REGION Network 46: FIT-508 LOW / HIGH
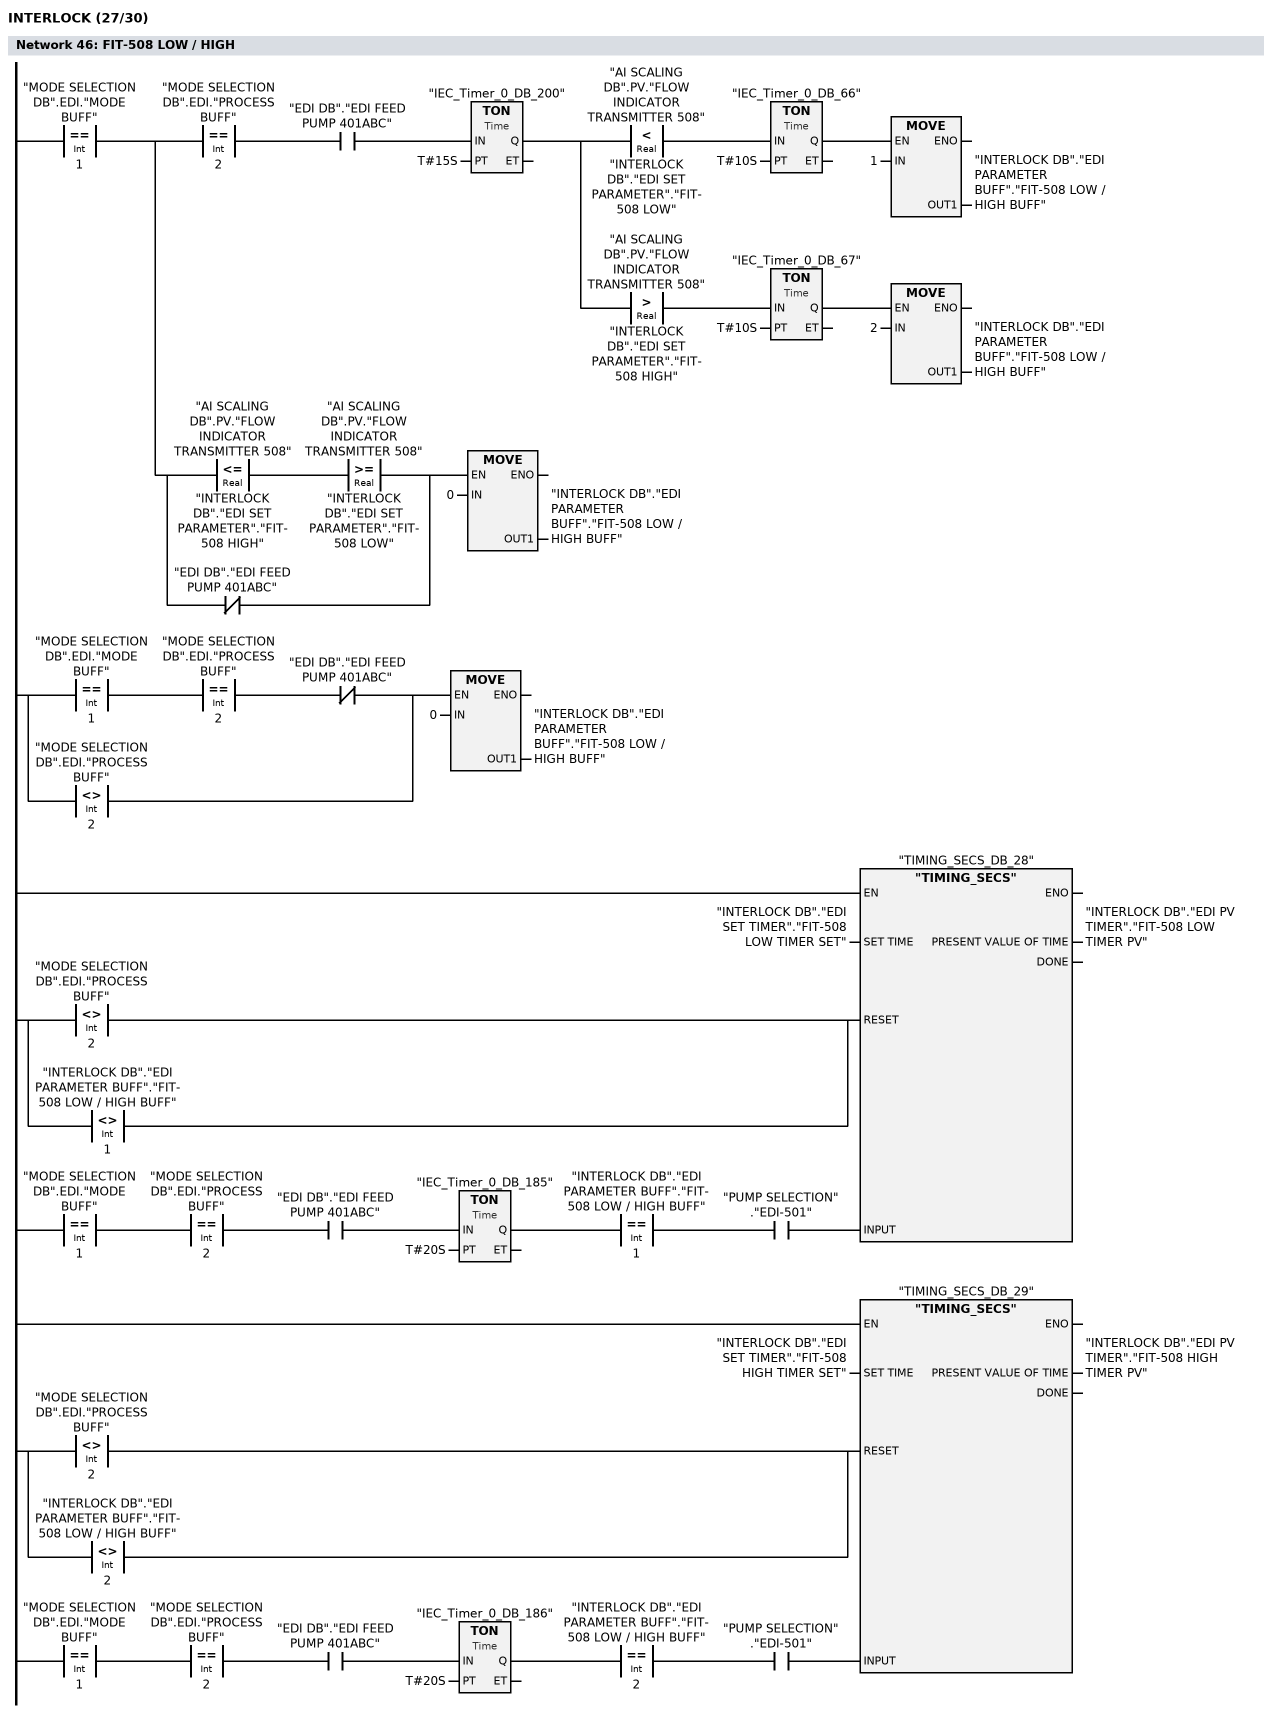
   RUNG wire#powerrail
      { S7_Templates := "SrcType := Int" } EQ_Contact(in1 := "MODE SELECTION DB".EDI."MODE BUFF", in2 := 1)
      wire#w1
      { S7_Templates := "SrcType := Int" } EQ_Contact(in1 := "MODE SELECTION DB".EDI."PROCESS BUFF", in2 := 2)
      Contact( "EDI DB"."EDI FEED PUMP 401ABC" )
      { S7_Templates := "time_type := Time" } "IEC_Timer_0_DB_200".TON(pt := T#15S, et =>)
      wire#w2
      { S7_Templates := "SrcType := Real" } LT_Contact(in1 := "AI SCALING DB".PV."FLOW INDICATOR TRANSMITTER 508", in2 := "INTERLOCK DB"."EDI SET PARAMETER"."FIT-508 LOW")
      { S7_Templates := "time_type := Time" } "IEC_Timer_0_DB_66".TON(pt := T#10S, et =>)
      Move(in := 1, out1 => "INTERLOCK DB"."EDI PARAMETER BUFF"."FIT-508 LOW / HIGH BUFF")
   END_RUNG
   RUNG wire#w2
      { S7_Templates := "SrcType := Real" } GT_Contact(in1 := "AI SCALING DB".PV."FLOW INDICATOR TRANSMITTER 508", in2 := "INTERLOCK DB"."EDI SET PARAMETER"."FIT-508 HIGH")
      { S7_Templates := "time_type := Time" } "IEC_Timer_0_DB_67".TON(pt := T#10S, et =>)
      Move(in := 2, out1 => "INTERLOCK DB"."EDI PARAMETER BUFF"."FIT-508 LOW / HIGH BUFF")
   END_RUNG
   RUNG wire#w1
      { S7_Templates := "SrcType := Real" } LE_Contact(in1 := "AI SCALING DB".PV."FLOW INDICATOR TRANSMITTER 508", in2 := "INTERLOCK DB"."EDI SET PARAMETER"."FIT-508 HIGH")
      { S7_Templates := "SrcType := Real" } GE_Contact(in1 := "AI SCALING DB".PV."FLOW INDICATOR TRANSMITTER 508", in2 := "INTERLOCK DB"."EDI SET PARAMETER"."FIT-508 LOW")
      wire#w3
      Move(in := 0, out1 => "INTERLOCK DB"."EDI PARAMETER BUFF"."FIT-508 LOW / HIGH BUFF")
   END_RUNG
   RUNG wire#w1
      I_Contact( "EDI DB"."EDI FEED PUMP 401ABC" )
   END_RUNG wire#w3
   RUNG wire#powerrail
      { S7_Templates := "SrcType := Int" } EQ_Contact(in1 := "MODE SELECTION DB".EDI."MODE BUFF", in2 := 1)
      { S7_Templates := "SrcType := Int" } EQ_Contact(in1 := "MODE SELECTION DB".EDI."PROCESS BUFF", in2 := 2)
      I_Contact( "EDI DB"."EDI FEED PUMP 401ABC" )
      wire#w4
      Move(in := 0, out1 => "INTERLOCK DB"."EDI PARAMETER BUFF"."FIT-508 LOW / HIGH BUFF")
   END_RUNG
   RUNG wire#powerrail
      { S7_Templates := "SrcType := Int" } NE_Contact(in1 := "MODE SELECTION DB".EDI."PROCESS BUFF", in2 := 2)
   END_RUNG wire#w4
   RUNG wire#powerrail
      "TIMING_SECS_DB_28"(RESET := wire#w5, INPUT := wire#w6, "SET TIME" := "INTERLOCK DB"."EDI SET TIMER"."FIT-508 LOW TIMER SET", "PRESENT VALUE OF TIME" => "INTERLOCK DB"."EDI PV TIMER"."FIT-508 LOW TIMER PV", DONE =>)
   END_RUNG
   RUNG wire#powerrail
      { S7_Templates := "SrcType := Int" } NE_Contact(in1 := "MODE SELECTION DB".EDI."PROCESS BUFF", in2 := 2)
   END_RUNG wire#w5
   RUNG wire#powerrail
      { S7_Templates := "SrcType := Int" } NE_Contact(in1 := "INTERLOCK DB"."EDI PARAMETER BUFF"."FIT-508 LOW / HIGH BUFF", in2 := 1)
   END_RUNG wire#w5
   RUNG wire#powerrail
      { S7_Templates := "SrcType := Int" } EQ_Contact(in1 := "MODE SELECTION DB".EDI."MODE BUFF", in2 := 1)
      { S7_Templates := "SrcType := Int" } EQ_Contact(in1 := "MODE SELECTION DB".EDI."PROCESS BUFF", in2 := 2)
      Contact( "EDI DB"."EDI FEED PUMP 401ABC" )
      { S7_Templates := "time_type := Time" } "IEC_Timer_0_DB_185".TON(pt := T#20S, et =>)
      { S7_Templates := "SrcType := Int" } EQ_Contact(in1 := "INTERLOCK DB"."EDI PARAMETER BUFF"."FIT-508 LOW / HIGH BUFF", in2 := 1)
      Contact( "PUMP SELECTION"."EDI-501" )
   END_RUNG wire#w6
   RUNG wire#powerrail
      "TIMING_SECS_DB_29"(RESET := wire#w7, INPUT := wire#w8, "SET TIME" := "INTERLOCK DB"."EDI SET TIMER"."FIT-508 HIGH TIMER SET", "PRESENT VALUE OF TIME" => "INTERLOCK DB"."EDI PV TIMER"."FIT-508 HIGH TIMER PV", DONE =>)
   END_RUNG
   RUNG wire#powerrail
      { S7_Templates := "SrcType := Int" } NE_Contact(in1 := "MODE SELECTION DB".EDI."PROCESS BUFF", in2 := 2)
   END_RUNG wire#w7
   RUNG wire#powerrail
      { S7_Templates := "SrcType := Int" } NE_Contact(in1 := "INTERLOCK DB"."EDI PARAMETER BUFF"."FIT-508 LOW / HIGH BUFF", in2 := 2)
   END_RUNG wire#w7
   RUNG wire#powerrail
      { S7_Templates := "SrcType := Int" } EQ_Contact(in1 := "MODE SELECTION DB".EDI."MODE BUFF", in2 := 1)
      { S7_Templates := "SrcType := Int" } EQ_Contact(in1 := "MODE SELECTION DB".EDI."PROCESS BUFF", in2 := 2)
      Contact( "EDI DB"."EDI FEED PUMP 401ABC" )
      { S7_Templates := "time_type := Time" } "IEC_Timer_0_DB_186".TON(pt := T#20S, et =>)
      { S7_Templates := "SrcType := Int" } EQ_Contact(in1 := "INTERLOCK DB"."EDI PARAMETER BUFF"."FIT-508 LOW / HIGH BUFF", in2 := 2)
      Contact( "PUMP SELECTION"."EDI-501" )
   END_RUNG wire#w8
   // the same network as SCL:
   #_w1 := "MODE SELECTION DB".EDI."MODE BUFF" = 1;
   "IEC_Timer_0_DB_200".TON(IN := #_w1 AND ("MODE SELECTION DB".EDI."PROCESS BUFF" = 2) AND "EDI DB"."EDI FEED PUMP 401ABC",
                           PT := T#15S);
   "IEC_Timer_0_DB_66".TON(IN := "IEC_Timer_0_DB_200".Q AND ("AI SCALING DB".PV."FLOW INDICATOR TRANSMITTER 508" < "INTERLOCK DB"."EDI SET PARAMETER"."FIT-508 LOW"),
                           PT := T#10S);
   IF "IEC_Timer_0_DB_66".Q THEN "INTERLOCK DB"."EDI PARAMETER BUFF"."FIT-508 LOW / HIGH BUFF" := 1; END_IF;
   "IEC_Timer_0_DB_67".TON(IN := "IEC_Timer_0_DB_200".Q AND ("AI SCALING DB".PV."FLOW INDICATOR TRANSMITTER 508" > "INTERLOCK DB"."EDI SET PARAMETER"."FIT-508 HIGH"),
                           PT := T#10S);
   IF "IEC_Timer_0_DB_67".Q THEN "INTERLOCK DB"."EDI PARAMETER BUFF"."FIT-508 LOW / HIGH BUFF" := 2; END_IF;
   IF #_w1 AND ((("AI SCALING DB".PV."FLOW INDICATOR TRANSMITTER 508" <= "INTERLOCK DB"."EDI SET PARAMETER"."FIT-508 HIGH") AND ("AI SCALING DB".PV."FLOW INDICATOR TRANSMITTER 508" >= "INTERLOCK DB"."EDI SET PARAMETER"."FIT-508 LOW")) OR NOT "EDI DB"."EDI FEED PUMP 401ABC") THEN
       "INTERLOCK DB"."EDI PARAMETER BUFF"."FIT-508 LOW / HIGH BUFF" := 0;
   END_IF;
   IF (("MODE SELECTION DB".EDI."MODE BUFF" = 1) AND ("MODE SELECTION DB".EDI."PROCESS BUFF" = 2) AND NOT "EDI DB"."EDI FEED PUMP 401ABC") OR ("MODE SELECTION DB".EDI."PROCESS BUFF" <> 2) THEN
       "INTERLOCK DB"."EDI PARAMETER BUFF"."FIT-508 LOW / HIGH BUFF" := 0;
   END_IF;
   "IEC_Timer_0_DB_185".TON(IN := ("MODE SELECTION DB".EDI."MODE BUFF" = 1) AND ("MODE SELECTION DB".EDI."PROCESS BUFF" = 2) AND "EDI DB"."EDI FEED PUMP 401ABC",
                           PT := T#20S);
   "TIMING_SECS_DB_28"("SET TIME" := "INTERLOCK DB"."EDI SET TIMER"."FIT-508 LOW TIMER SET",   // "TIMING_SECS"
                       RESET := ("MODE SELECTION DB".EDI."PROCESS BUFF" <> 2) OR ("INTERLOCK DB"."EDI PARAMETER BUFF"."FIT-508 LOW / HIGH BUFF" <> 1),
                       INPUT := "IEC_Timer_0_DB_185".Q AND ("INTERLOCK DB"."EDI PARAMETER BUFF"."FIT-508 LOW / HIGH BUFF" = 1) AND "PUMP SELECTION"."EDI-501",
                       "PRESENT VALUE OF TIME" => "INTERLOCK DB"."EDI PV TIMER"."FIT-508 LOW TIMER PV");
   "IEC_Timer_0_DB_186".TON(IN := ("MODE SELECTION DB".EDI."MODE BUFF" = 1) AND ("MODE SELECTION DB".EDI."PROCESS BUFF" = 2) AND "EDI DB"."EDI FEED PUMP 401ABC",
                           PT := T#20S);
   "TIMING_SECS_DB_29"("SET TIME" := "INTERLOCK DB"."EDI SET TIMER"."FIT-508 HIGH TIMER SET",   // "TIMING_SECS"
                       RESET := ("MODE SELECTION DB".EDI."PROCESS BUFF" <> 2) OR ("INTERLOCK DB"."EDI PARAMETER BUFF"."FIT-508 LOW / HIGH BUFF" <> 2),
                       INPUT := "IEC_Timer_0_DB_186".Q AND ("INTERLOCK DB"."EDI PARAMETER BUFF"."FIT-508 LOW / HIGH BUFF" = 2) AND "PUMP SELECTION"."EDI-501",
                       "PRESENT VALUE OF TIME" => "INTERLOCK DB"."EDI PV TIMER"."FIT-508 HIGH TIMER PV");
END_REGION

REGION Network 47: pH-501 - LOW / High
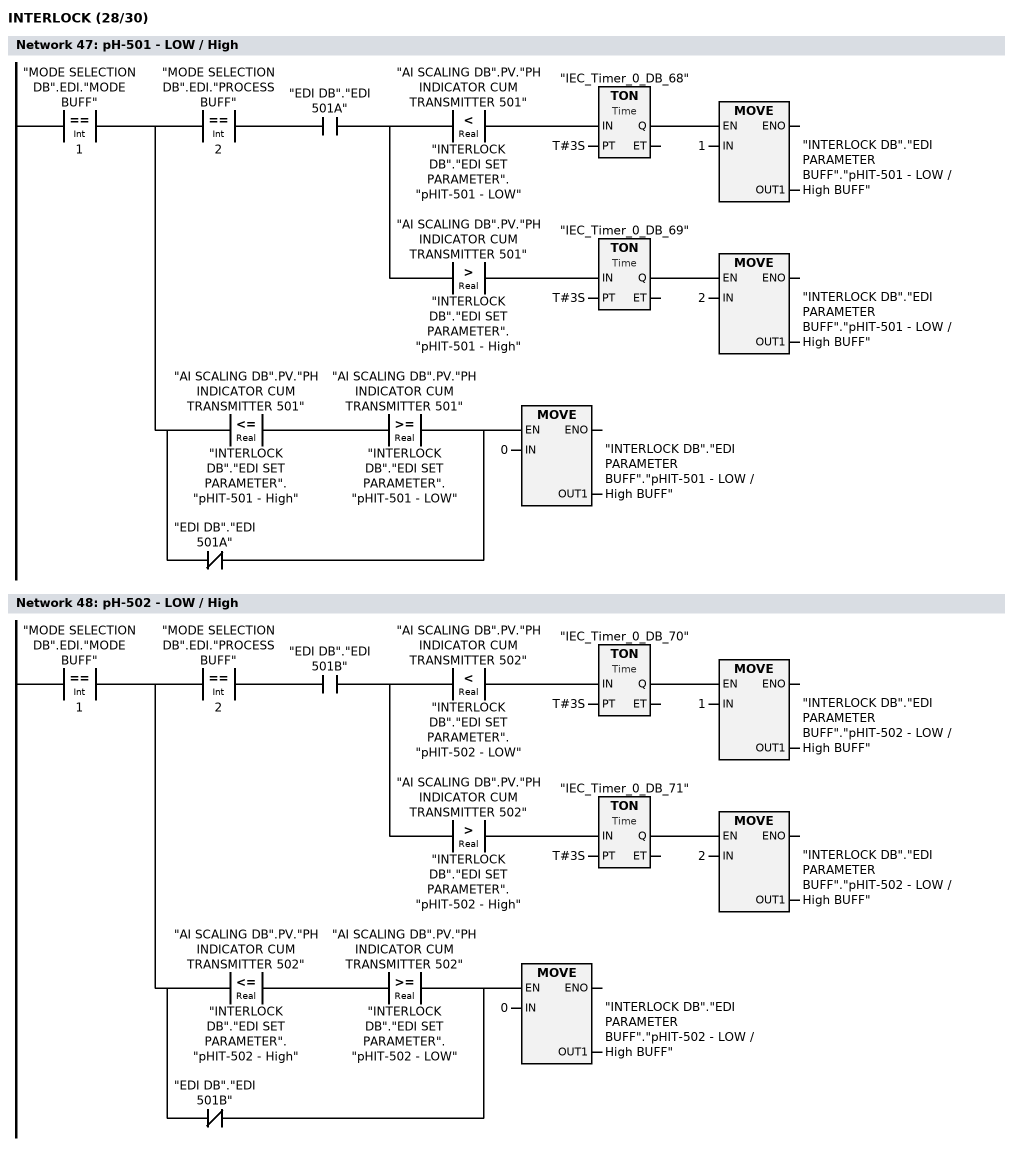
   RUNG wire#powerrail
      { S7_Templates := "SrcType := Int" } EQ_Contact(in1 := "MODE SELECTION DB".EDI."MODE BUFF", in2 := 1)
      wire#w1
      { S7_Templates := "SrcType := Int" } EQ_Contact(in1 := "MODE SELECTION DB".EDI."PROCESS BUFF", in2 := 2)
      Contact( "EDI DB"."EDI 501A" )
      wire#w2
      { S7_Templates := "SrcType := Real" } LT_Contact(in1 := "AI SCALING DB".PV."PH INDICATOR CUM TRANSMITTER 501", in2 := "INTERLOCK DB"."EDI SET PARAMETER"."pHIT-501 - LOW")
      { S7_Templates := "time_type := Time" } "IEC_Timer_0_DB_68".TON(pt := T#3S, et =>)
      Move(in := 1, out1 => "INTERLOCK DB"."EDI PARAMETER BUFF"."pHIT-501 - LOW / High BUFF")
   END_RUNG
   RUNG wire#w2
      { S7_Templates := "SrcType := Real" } GT_Contact(in1 := "AI SCALING DB".PV."PH INDICATOR CUM TRANSMITTER 501", in2 := "INTERLOCK DB"."EDI SET PARAMETER"."pHIT-501 - High")
      { S7_Templates := "time_type := Time" } "IEC_Timer_0_DB_69".TON(pt := T#3S, et =>)
      Move(in := 2, out1 => "INTERLOCK DB"."EDI PARAMETER BUFF"."pHIT-501 - LOW / High BUFF")
   END_RUNG
   RUNG wire#w1
      { S7_Templates := "SrcType := Real" } LE_Contact(in1 := "AI SCALING DB".PV."PH INDICATOR CUM TRANSMITTER 501", in2 := "INTERLOCK DB"."EDI SET PARAMETER"."pHIT-501 - High")
      { S7_Templates := "SrcType := Real" } GE_Contact(in1 := "AI SCALING DB".PV."PH INDICATOR CUM TRANSMITTER 501", in2 := "INTERLOCK DB"."EDI SET PARAMETER"."pHIT-501 - LOW")
      wire#w3
      Move(in := 0, out1 => "INTERLOCK DB"."EDI PARAMETER BUFF"."pHIT-501 - LOW / High BUFF")
   END_RUNG
   RUNG wire#w1
      I_Contact( "EDI DB"."EDI 501A" )
   END_RUNG wire#w3
   // the same network as SCL:
   #_w1 := "MODE SELECTION DB".EDI."MODE BUFF" = 1;
   #_w2 := #_w1 AND ("MODE SELECTION DB".EDI."PROCESS BUFF" = 2) AND "EDI DB"."EDI 501A";
   "IEC_Timer_0_DB_68".TON(IN := #_w2 AND ("AI SCALING DB".PV."PH INDICATOR CUM TRANSMITTER 501" < "INTERLOCK DB"."EDI SET PARAMETER"."pHIT-501 - LOW"),
                           PT := T#3S);
   IF "IEC_Timer_0_DB_68".Q THEN
       "INTERLOCK DB"."EDI PARAMETER BUFF"."pHIT-501 - LOW / High BUFF" := 1;
   END_IF;
   "IEC_Timer_0_DB_69".TON(IN := #_w2 AND ("AI SCALING DB".PV."PH INDICATOR CUM TRANSMITTER 501" > "INTERLOCK DB"."EDI SET PARAMETER"."pHIT-501 - High"),
                           PT := T#3S);
   IF "IEC_Timer_0_DB_69".Q THEN
       "INTERLOCK DB"."EDI PARAMETER BUFF"."pHIT-501 - LOW / High BUFF" := 2;
   END_IF;
   IF #_w1 AND ((("AI SCALING DB".PV."PH INDICATOR CUM TRANSMITTER 501" <= "INTERLOCK DB"."EDI SET PARAMETER"."pHIT-501 - High") AND ("AI SCALING DB".PV."PH INDICATOR CUM TRANSMITTER 501" >= "INTERLOCK DB"."EDI SET PARAMETER"."pHIT-501 - LOW")) OR NOT "EDI DB"."EDI 501A") THEN
       "INTERLOCK DB"."EDI PARAMETER BUFF"."pHIT-501 - LOW / High BUFF" := 0;
   END_IF;
END_REGION

REGION Network 48: pH-502 - LOW / High
   RUNG wire#powerrail
      { S7_Templates := "SrcType := Int" } EQ_Contact(in1 := "MODE SELECTION DB".EDI."MODE BUFF", in2 := 1)
      wire#w1
      { S7_Templates := "SrcType := Int" } EQ_Contact(in1 := "MODE SELECTION DB".EDI."PROCESS BUFF", in2 := 2)
      Contact( "EDI DB"."EDI 501B" )
      wire#w2
      { S7_Templates := "SrcType := Real" } LT_Contact(in1 := "AI SCALING DB".PV."PH INDICATOR CUM TRANSMITTER 502", in2 := "INTERLOCK DB"."EDI SET PARAMETER"."pHIT-502 - LOW")
      { S7_Templates := "time_type := Time" } "IEC_Timer_0_DB_70".TON(pt := T#3S, et =>)
      Move(in := 1, out1 => "INTERLOCK DB"."EDI PARAMETER BUFF"."pHIT-502 - LOW / High BUFF")
   END_RUNG
   RUNG wire#w2
      { S7_Templates := "SrcType := Real" } GT_Contact(in1 := "AI SCALING DB".PV."PH INDICATOR CUM TRANSMITTER 502", in2 := "INTERLOCK DB"."EDI SET PARAMETER"."pHIT-502 - High")
      { S7_Templates := "time_type := Time" } "IEC_Timer_0_DB_71".TON(pt := T#3S, et =>)
      Move(in := 2, out1 => "INTERLOCK DB"."EDI PARAMETER BUFF"."pHIT-502 - LOW / High BUFF")
   END_RUNG
   RUNG wire#w1
      { S7_Templates := "SrcType := Real" } LE_Contact(in1 := "AI SCALING DB".PV."PH INDICATOR CUM TRANSMITTER 502", in2 := "INTERLOCK DB"."EDI SET PARAMETER"."pHIT-502 - High")
      { S7_Templates := "SrcType := Real" } GE_Contact(in1 := "AI SCALING DB".PV."PH INDICATOR CUM TRANSMITTER 502", in2 := "INTERLOCK DB"."EDI SET PARAMETER"."pHIT-502 - LOW")
      wire#w3
      Move(in := 0, out1 => "INTERLOCK DB"."EDI PARAMETER BUFF"."pHIT-502 - LOW / High BUFF")
   END_RUNG
   RUNG wire#w1
      I_Contact( "EDI DB"."EDI 501B" )
   END_RUNG wire#w3
   // the same network as SCL:
   #_w1 := "MODE SELECTION DB".EDI."MODE BUFF" = 1;
   #_w2 := #_w1 AND ("MODE SELECTION DB".EDI."PROCESS BUFF" = 2) AND "EDI DB"."EDI 501B";
   "IEC_Timer_0_DB_70".TON(IN := #_w2 AND ("AI SCALING DB".PV."PH INDICATOR CUM TRANSMITTER 502" < "INTERLOCK DB"."EDI SET PARAMETER"."pHIT-502 - LOW"),
                           PT := T#3S);
   IF "IEC_Timer_0_DB_70".Q THEN
       "INTERLOCK DB"."EDI PARAMETER BUFF"."pHIT-502 - LOW / High BUFF" := 1;
   END_IF;
   "IEC_Timer_0_DB_71".TON(IN := #_w2 AND ("AI SCALING DB".PV."PH INDICATOR CUM TRANSMITTER 502" > "INTERLOCK DB"."EDI SET PARAMETER"."pHIT-502 - High"),
                           PT := T#3S);
   IF "IEC_Timer_0_DB_71".Q THEN
       "INTERLOCK DB"."EDI PARAMETER BUFF"."pHIT-502 - LOW / High BUFF" := 2;
   END_IF;
   IF #_w1 AND ((("AI SCALING DB".PV."PH INDICATOR CUM TRANSMITTER 502" <= "INTERLOCK DB"."EDI SET PARAMETER"."pHIT-502 - High") AND ("AI SCALING DB".PV."PH INDICATOR CUM TRANSMITTER 502" >= "INTERLOCK DB"."EDI SET PARAMETER"."pHIT-502 - LOW")) OR NOT "EDI DB"."EDI 501B") THEN
       "INTERLOCK DB"."EDI PARAMETER BUFF"."pHIT-502 - LOW / High BUFF" := 0;
   END_IF;
END_REGION

REGION Network 49: RIT-501 HIGH
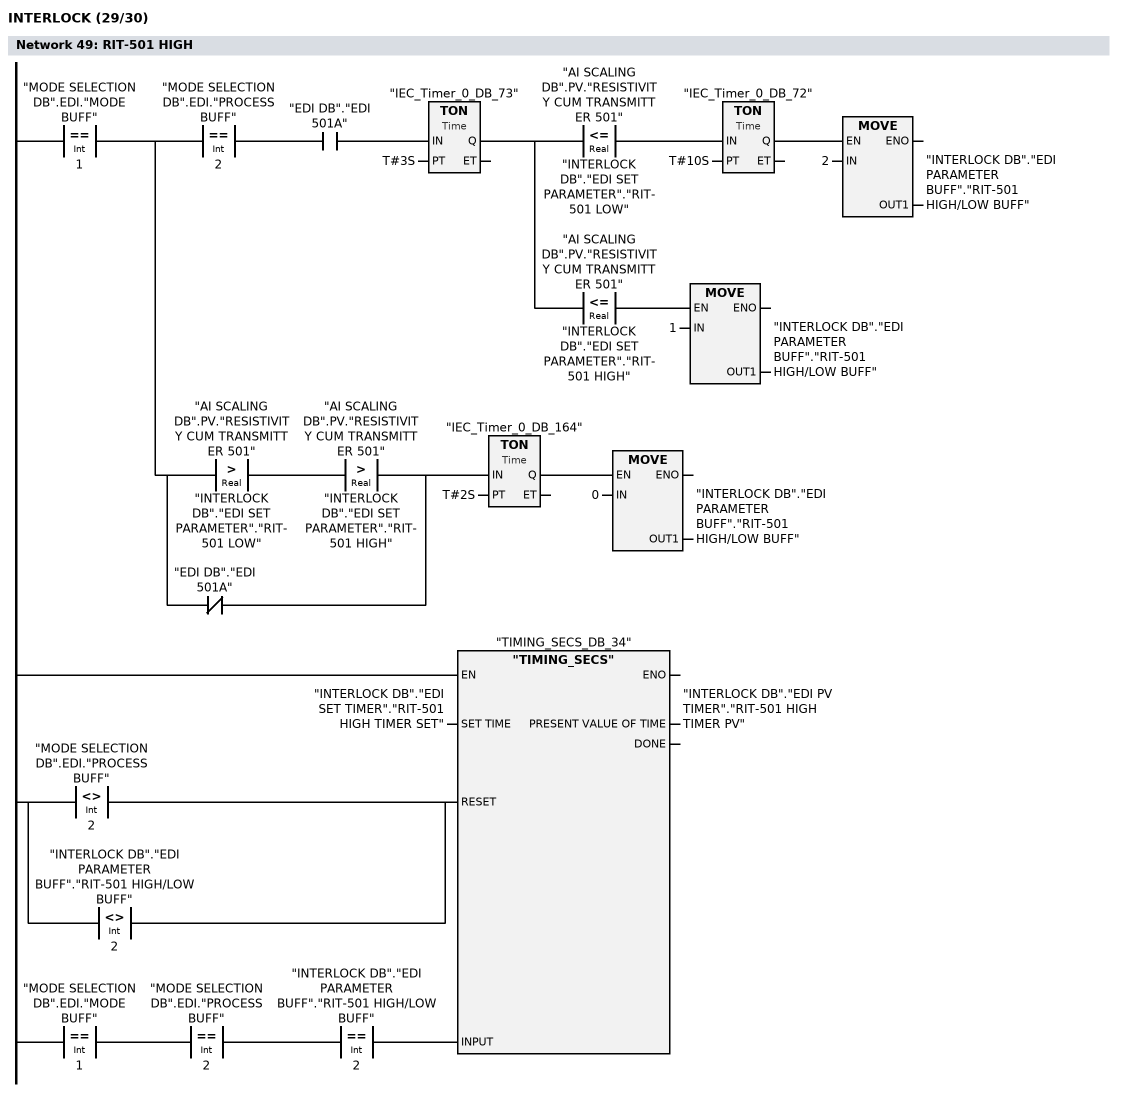
   RUNG wire#powerrail
      { S7_Templates := "SrcType := Int" } EQ_Contact(in1 := "MODE SELECTION DB".EDI."MODE BUFF", in2 := 1)
      wire#w1
      { S7_Templates := "SrcType := Int" } EQ_Contact(in1 := "MODE SELECTION DB".EDI."PROCESS BUFF", in2 := 2)
      Contact( "EDI DB"."EDI 501A" )
      { S7_Templates := "time_type := Time" } "IEC_Timer_0_DB_73".TON(pt := T#3S, et =>)
      wire#w2
      { S7_Templates := "SrcType := Real" } LE_Contact(in1 := "AI SCALING DB".PV."RESISTIVITY CUM TRANSMITTER 501", in2 := "INTERLOCK DB"."EDI SET PARAMETER"."RIT-501 LOW")
      { S7_Templates := "time_type := Time" } "IEC_Timer_0_DB_72".TON(pt := T#10S, et =>)
      Move(in := 2, out1 => "INTERLOCK DB"."EDI PARAMETER BUFF"."RIT-501 HIGH/LOW BUFF")
   END_RUNG
   RUNG wire#w2
      { S7_Templates := "SrcType := Real" } LE_Contact(in1 := "AI SCALING DB".PV."RESISTIVITY CUM TRANSMITTER 501", in2 := "INTERLOCK DB"."EDI SET PARAMETER"."RIT-501 HIGH")
      Move(in := 1, out1 => "INTERLOCK DB"."EDI PARAMETER BUFF"."RIT-501 HIGH/LOW BUFF")
   END_RUNG
   RUNG wire#w1
      { S7_Templates := "SrcType := Real" } GT_Contact(in1 := "AI SCALING DB".PV."RESISTIVITY CUM TRANSMITTER 501", in2 := "INTERLOCK DB"."EDI SET PARAMETER"."RIT-501 LOW")
      { S7_Templates := "SrcType := Real" } GT_Contact(in1 := "AI SCALING DB".PV."RESISTIVITY CUM TRANSMITTER 501", in2 := "INTERLOCK DB"."EDI SET PARAMETER"."RIT-501 HIGH")
      wire#w3
      { S7_Templates := "time_type := Time" } "IEC_Timer_0_DB_164".TON(pt := T#2S, et =>)
      Move(in := 0, out1 => "INTERLOCK DB"."EDI PARAMETER BUFF"."RIT-501 HIGH/LOW BUFF")
   END_RUNG
   RUNG wire#w1
      I_Contact( "EDI DB"."EDI 501A" )
   END_RUNG wire#w3
   RUNG wire#powerrail
      "TIMING_SECS_DB_34"(RESET := wire#w4, INPUT := wire#w5, "SET TIME" := "INTERLOCK DB"."EDI SET TIMER"."RIT-501 HIGH TIMER SET", "PRESENT VALUE OF TIME" => "INTERLOCK DB"."EDI PV TIMER"."RIT-501 HIGH TIMER PV", DONE =>)
   END_RUNG
   RUNG wire#powerrail
      { S7_Templates := "SrcType := Int" } NE_Contact(in1 := "MODE SELECTION DB".EDI."PROCESS BUFF", in2 := 2)
   END_RUNG wire#w4
   RUNG wire#powerrail
      { S7_Templates := "SrcType := Int" } NE_Contact(in1 := "INTERLOCK DB"."EDI PARAMETER BUFF"."RIT-501 HIGH/LOW BUFF", in2 := 2)
   END_RUNG wire#w4
   RUNG wire#powerrail
      { S7_Templates := "SrcType := Int" } EQ_Contact(in1 := "MODE SELECTION DB".EDI."MODE BUFF", in2 := 1)
      { S7_Templates := "SrcType := Int" } EQ_Contact(in1 := "MODE SELECTION DB".EDI."PROCESS BUFF", in2 := 2)
      { S7_Templates := "SrcType := Int" } EQ_Contact(in1 := "INTERLOCK DB"."EDI PARAMETER BUFF"."RIT-501 HIGH/LOW BUFF", in2 := 2)
   END_RUNG wire#w5
   // the same network as SCL:
   #_w1 := "MODE SELECTION DB".EDI."MODE BUFF" = 1;
   "IEC_Timer_0_DB_73".TON(IN := #_w1 AND ("MODE SELECTION DB".EDI."PROCESS BUFF" = 2) AND "EDI DB"."EDI 501A",
                           PT := T#3S);
   "IEC_Timer_0_DB_72".TON(IN := "IEC_Timer_0_DB_73".Q AND ("AI SCALING DB".PV."RESISTIVITY CUM TRANSMITTER 501" <= "INTERLOCK DB"."EDI SET PARAMETER"."RIT-501 LOW"),
                           PT := T#10S);
   IF "IEC_Timer_0_DB_72".Q THEN "INTERLOCK DB"."EDI PARAMETER BUFF"."RIT-501 HIGH/LOW BUFF" := 2; END_IF;
   IF "IEC_Timer_0_DB_73".Q AND ("AI SCALING DB".PV."RESISTIVITY CUM TRANSMITTER 501" <= "INTERLOCK DB"."EDI SET PARAMETER"."RIT-501 HIGH") THEN
       "INTERLOCK DB"."EDI PARAMETER BUFF"."RIT-501 HIGH/LOW BUFF" := 1;
   END_IF;
   "IEC_Timer_0_DB_164".TON(IN := #_w1 AND ((("AI SCALING DB".PV."RESISTIVITY CUM TRANSMITTER 501" > "INTERLOCK DB"."EDI SET PARAMETER"."RIT-501 LOW") AND ("AI SCALING DB".PV."RESISTIVITY CUM TRANSMITTER 501" > "INTERLOCK DB"."EDI SET PARAMETER"."RIT-501 HIGH")) OR NOT "EDI DB"."EDI 501A"),
                           PT := T#2S);
   IF "IEC_Timer_0_DB_164".Q THEN "INTERLOCK DB"."EDI PARAMETER BUFF"."RIT-501 HIGH/LOW BUFF" := 0; END_IF;
   "TIMING_SECS_DB_34"("SET TIME" := "INTERLOCK DB"."EDI SET TIMER"."RIT-501 HIGH TIMER SET",   // "TIMING_SECS"
                       RESET := ("MODE SELECTION DB".EDI."PROCESS BUFF" <> 2) OR ("INTERLOCK DB"."EDI PARAMETER BUFF"."RIT-501 HIGH/LOW BUFF" <> 2),
                       INPUT := ("MODE SELECTION DB".EDI."MODE BUFF" = 1) AND ("MODE SELECTION DB".EDI."PROCESS BUFF" = 2) AND ("INTERLOCK DB"."EDI PARAMETER BUFF"."RIT-501 HIGH/LOW BUFF" = 2),
                       "PRESENT VALUE OF TIME" => "INTERLOCK DB"."EDI PV TIMER"."RIT-501 HIGH TIMER PV");
END_REGION

REGION Network 50: RIT-502 HIGH
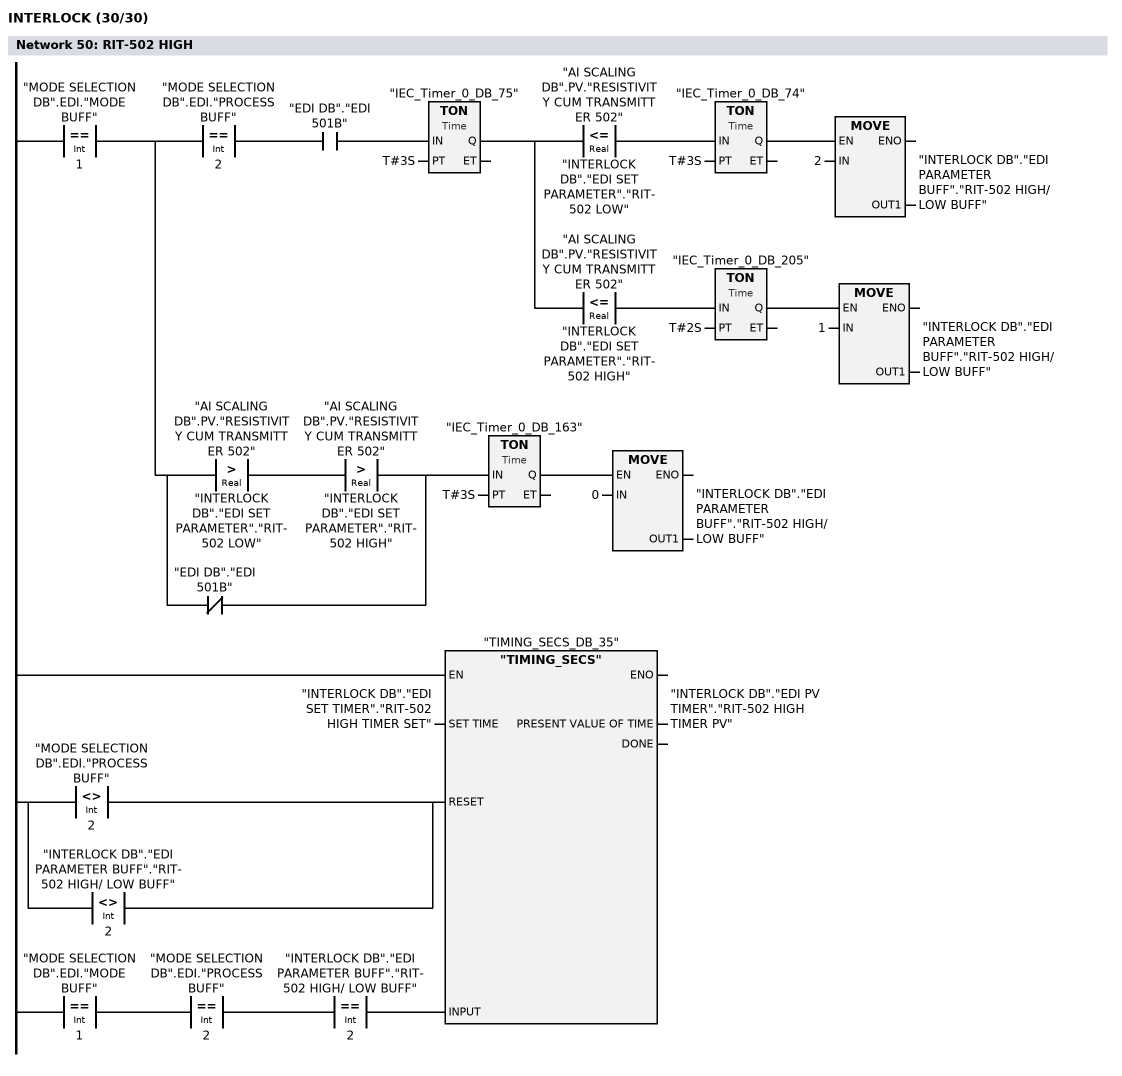
   RUNG wire#powerrail
      { S7_Templates := "SrcType := Int" } EQ_Contact(in1 := "MODE SELECTION DB".EDI."MODE BUFF", in2 := 1)
      wire#w1
      { S7_Templates := "SrcType := Int" } EQ_Contact(in1 := "MODE SELECTION DB".EDI."PROCESS BUFF", in2 := 2)
      Contact( "EDI DB"."EDI 501B" )
      { S7_Templates := "time_type := Time" } "IEC_Timer_0_DB_75".TON(pt := T#3S, et =>)
      wire#w2
      { S7_Templates := "SrcType := Real" } LE_Contact(in1 := "AI SCALING DB".PV."RESISTIVITY CUM TRANSMITTER 502", in2 := "INTERLOCK DB"."EDI SET PARAMETER"."RIT-502 LOW")
      { S7_Templates := "time_type := Time" } "IEC_Timer_0_DB_74".TON(pt := T#3S, et =>)
      Move(in := 2, out1 => "INTERLOCK DB"."EDI PARAMETER BUFF"."RIT-502 HIGH/ LOW BUFF")
   END_RUNG
   RUNG wire#w2
      { S7_Templates := "SrcType := Real" } LE_Contact(in1 := "AI SCALING DB".PV."RESISTIVITY CUM TRANSMITTER 502", in2 := "INTERLOCK DB"."EDI SET PARAMETER"."RIT-502 HIGH")
      { S7_Templates := "time_type := Time" } "IEC_Timer_0_DB_205".TON(pt := T#2S, et =>)
      Move(in := 1, out1 => "INTERLOCK DB"."EDI PARAMETER BUFF"."RIT-502 HIGH/ LOW BUFF")
   END_RUNG
   RUNG wire#w1
      { S7_Templates := "SrcType := Real" } GT_Contact(in1 := "AI SCALING DB".PV."RESISTIVITY CUM TRANSMITTER 502", in2 := "INTERLOCK DB"."EDI SET PARAMETER"."RIT-502 LOW")
      { S7_Templates := "SrcType := Real" } GT_Contact(in1 := "AI SCALING DB".PV."RESISTIVITY CUM TRANSMITTER 502", in2 := "INTERLOCK DB"."EDI SET PARAMETER"."RIT-502 HIGH")
      wire#w3
      { S7_Templates := "time_type := Time" } "IEC_Timer_0_DB_163".TON(pt := T#3S, et =>)
      Move(in := 0, out1 => "INTERLOCK DB"."EDI PARAMETER BUFF"."RIT-502 HIGH/ LOW BUFF")
   END_RUNG
   RUNG wire#w1
      I_Contact( "EDI DB"."EDI 501B" )
   END_RUNG wire#w3
   RUNG wire#powerrail
      "TIMING_SECS_DB_35"(RESET := wire#w4, INPUT := wire#w5, "SET TIME" := "INTERLOCK DB"."EDI SET TIMER"."RIT-502 HIGH TIMER SET", "PRESENT VALUE OF TIME" => "INTERLOCK DB"."EDI PV TIMER"."RIT-502 HIGH TIMER PV", DONE =>)
   END_RUNG
   RUNG wire#powerrail
      { S7_Templates := "SrcType := Int" } NE_Contact(in1 := "MODE SELECTION DB".EDI."PROCESS BUFF", in2 := 2)
   END_RUNG wire#w4
   RUNG wire#powerrail
      { S7_Templates := "SrcType := Int" } NE_Contact(in1 := "INTERLOCK DB"."EDI PARAMETER BUFF"."RIT-502 HIGH/ LOW BUFF", in2 := 2)
   END_RUNG wire#w4
   RUNG wire#powerrail
      { S7_Templates := "SrcType := Int" } EQ_Contact(in1 := "MODE SELECTION DB".EDI."MODE BUFF", in2 := 1)
      { S7_Templates := "SrcType := Int" } EQ_Contact(in1 := "MODE SELECTION DB".EDI."PROCESS BUFF", in2 := 2)
      { S7_Templates := "SrcType := Int" } EQ_Contact(in1 := "INTERLOCK DB"."EDI PARAMETER BUFF"."RIT-502 HIGH/ LOW BUFF", in2 := 2)
   END_RUNG wire#w5
   // the same network as SCL:
   #_w1 := "MODE SELECTION DB".EDI."MODE BUFF" = 1;
   "IEC_Timer_0_DB_75".TON(IN := #_w1 AND ("MODE SELECTION DB".EDI."PROCESS BUFF" = 2) AND "EDI DB"."EDI 501B",
                           PT := T#3S);
   "IEC_Timer_0_DB_74".TON(IN := "IEC_Timer_0_DB_75".Q AND ("AI SCALING DB".PV."RESISTIVITY CUM TRANSMITTER 502" <= "INTERLOCK DB"."EDI SET PARAMETER"."RIT-502 LOW"),
                           PT := T#3S);
   IF "IEC_Timer_0_DB_74".Q THEN "INTERLOCK DB"."EDI PARAMETER BUFF"."RIT-502 HIGH/ LOW BUFF" := 2; END_IF;
   "IEC_Timer_0_DB_205".TON(IN := "IEC_Timer_0_DB_75".Q AND ("AI SCALING DB".PV."RESISTIVITY CUM TRANSMITTER 502" <= "INTERLOCK DB"."EDI SET PARAMETER"."RIT-502 HIGH"),
                           PT := T#2S);
   IF "IEC_Timer_0_DB_205".Q THEN "INTERLOCK DB"."EDI PARAMETER BUFF"."RIT-502 HIGH/ LOW BUFF" := 1; END_IF;
   "IEC_Timer_0_DB_163".TON(IN := #_w1 AND ((("AI SCALING DB".PV."RESISTIVITY CUM TRANSMITTER 502" > "INTERLOCK DB"."EDI SET PARAMETER"."RIT-502 LOW") AND ("AI SCALING DB".PV."RESISTIVITY CUM TRANSMITTER 502" > "INTERLOCK DB"."EDI SET PARAMETER"."RIT-502 HIGH")) OR NOT "EDI DB"."EDI 501B"),
                           PT := T#3S);
   IF "IEC_Timer_0_DB_163".Q THEN "INTERLOCK DB"."EDI PARAMETER BUFF"."RIT-502 HIGH/ LOW BUFF" := 0; END_IF;
   "TIMING_SECS_DB_35"("SET TIME" := "INTERLOCK DB"."EDI SET TIMER"."RIT-502 HIGH TIMER SET",   // "TIMING_SECS"
                       RESET := ("MODE SELECTION DB".EDI."PROCESS BUFF" <> 2) OR ("INTERLOCK DB"."EDI PARAMETER BUFF"."RIT-502 HIGH/ LOW BUFF" <> 2),
                       INPUT := ("MODE SELECTION DB".EDI."MODE BUFF" = 1) AND ("MODE SELECTION DB".EDI."PROCESS BUFF" = 2) AND ("INTERLOCK DB"."EDI PARAMETER BUFF"."RIT-502 HIGH/ LOW BUFF" = 2),
                       "PRESENT VALUE OF TIME" => "INTERLOCK DB"."EDI PV TIMER"."RIT-502 HIGH TIMER PV");
END_REGION
END_FUNCTION

FUNCTION_BLOCK "TIMING_SECS"   // FB3, LAD
{ S7_Optimized_Access := 'TRUE' }
// stored: MemoryReserve 100, SetENOAutomatically false
   VAR_INPUT
      "SET TIME" : Int;
      RESET : Bool;
      INPUT : Bool;
   END_VAR
   VAR_OUTPUT
      "PRESENT VALUE OF TIME" : Int;
      DONE : Bool;
   END_VAR
   VAR
      "TIMER 1" { S7_SetPoint := 'True'} : IEC_TIMER;
   END_VAR
   VAR RETAIN
      "COUNTER1 1" { S7_SetPoint := 'True'} : IEC_COUNTER;
   END_VAR
   VAR_TEMP   // added for the SCL form of the ladder/FBD networks
      _w1 : Bool;
      _w2 : Bool;
   END_VAR
BEGIN

REGION Network 1
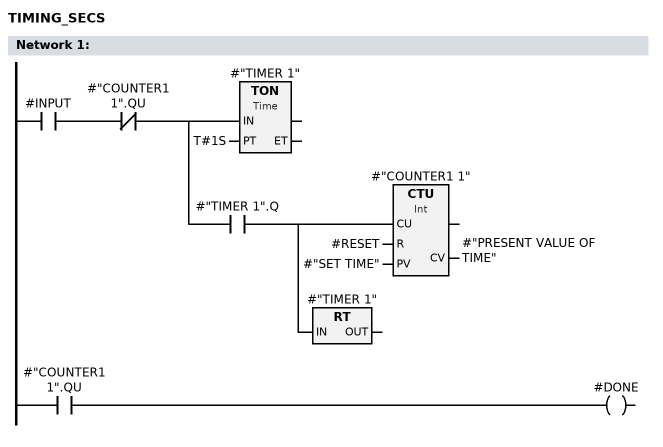
   RUNG wire#powerrail
      Contact( #INPUT )
      I_Contact( #"COUNTER1 1".QU )
      wire#w1
      { S7_Templates := "time_type := Time" } #"TIMER 1".TON(pt := T#1S, et =>)
   END_RUNG
   RUNG wire#w1
      Contact( #"TIMER 1".Q )
      wire#w2
      { S7_Templates := "value_type := Int" } #"COUNTER1 1".CTU(r := #RESET, pv := #"SET TIME", cv => #"PRESENT VALUE OF TIME")
   END_RUNG
   RUNG wire#w2
      RT_Coil( #"TIMER 1" )
   END_RUNG
   RUNG wire#powerrail
      Contact( #"COUNTER1 1".QU )
      Coil( #DONE )
   END_RUNG
   // the same network as SCL:
   #_w1 := #INPUT AND NOT #"COUNTER1 1".QU;
   #"TIMER 1".TON(IN := #_w1, PT := T#1S);
   #_w2 := #_w1 AND #"TIMER 1".Q;
   #"COUNTER1 1".CTU(CU := #_w2, R := #RESET, PV := #"SET TIME", CV => #"PRESENT VALUE OF TIME");
   IF #_w2 THEN RESET_TIMER(#"TIMER 1"); END_IF;
   #DONE := #"COUNTER1 1".QU;
END_REGION
END_FUNCTION_BLOCK

FUNCTION "AO SCALING" : Void   // FC13, LAD
{ S7_Optimized_Access := 'TRUE' }
// stored: SetENOAutomatically false
BEGIN

REGION Network 1: VFD P-502A
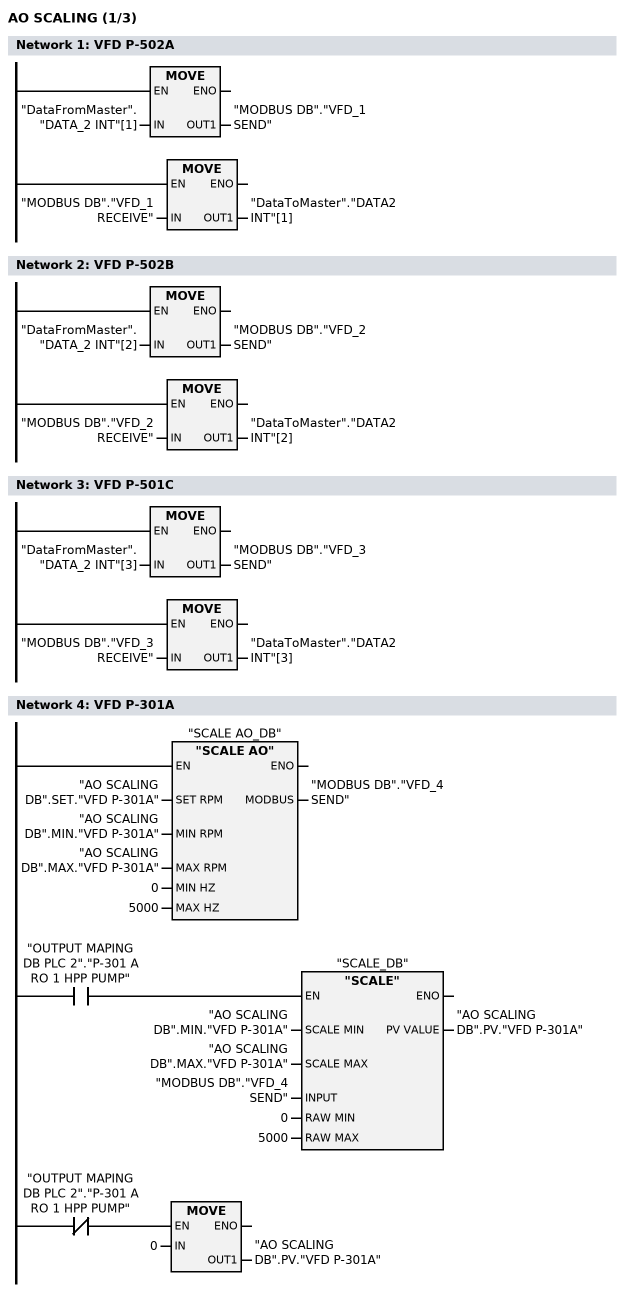
   RUNG wire#powerrail
      Move(in := "DataFromMaster"."DATA_2 INT"[1], out1 => "MODBUS DB"."VFD_1 SEND")
   END_RUNG
   RUNG wire#powerrail
      Move(in := "MODBUS DB"."VFD_1 RECEIVE", out1 => "DataToMaster"."DATA2 INT"[1])
   END_RUNG
   // the same network as SCL:
   "MODBUS DB"."VFD_1 SEND" := "DataFromMaster"."DATA_2 INT"[1];
   "DataToMaster"."DATA2 INT"[1] := "MODBUS DB"."VFD_1 RECEIVE";
END_REGION

REGION Network 2: VFD P-502B
   RUNG wire#powerrail
      Move(in := "DataFromMaster"."DATA_2 INT"[2], out1 => "MODBUS DB"."VFD_2 SEND")
   END_RUNG
   RUNG wire#powerrail
      Move(in := "MODBUS DB"."VFD_2 RECEIVE", out1 => "DataToMaster"."DATA2 INT"[2])
   END_RUNG
   // the same network as SCL:
   "MODBUS DB"."VFD_2 SEND" := "DataFromMaster"."DATA_2 INT"[2];
   "DataToMaster"."DATA2 INT"[2] := "MODBUS DB"."VFD_2 RECEIVE";
END_REGION

REGION Network 3: VFD P-501C
   RUNG wire#powerrail
      Move(in := "DataFromMaster"."DATA_2 INT"[3], out1 => "MODBUS DB"."VFD_3 SEND")
   END_RUNG
   RUNG wire#powerrail
      Move(in := "MODBUS DB"."VFD_3 RECEIVE", out1 => "DataToMaster"."DATA2 INT"[3])
   END_RUNG
   // the same network as SCL:
   "MODBUS DB"."VFD_3 SEND" := "DataFromMaster"."DATA_2 INT"[3];
   "DataToMaster"."DATA2 INT"[3] := "MODBUS DB"."VFD_3 RECEIVE";
END_REGION

REGION Network 4: VFD P-301A
   RUNG wire#powerrail
      "SCALE AO_DB"("SET RPM" := "AO SCALING DB".SET."VFD P-301A", "MIN RPM" := "AO SCALING DB".MIN."VFD P-301A", "MAX RPM" := "AO SCALING DB".MAX."VFD P-301A", "MIN HZ" := 0, "MAX HZ" := 5000, MODBUS => "MODBUS DB"."VFD_4 SEND")
   END_RUNG
   RUNG wire#powerrail
      Contact( "OUTPUT MAPING DB PLC 2"."P-301 A RO 1 HPP PUMP" )
      "SCALE_DB"("SCALE MIN" := "AO SCALING DB".MIN."VFD P-301A", "SCALE MAX" := "AO SCALING DB".MAX."VFD P-301A", INPUT := "MODBUS DB"."VFD_4 SEND", "RAW MIN" := 0, "RAW MAX" := 5000, "PV VALUE" => "AO SCALING DB".PV."VFD P-301A")
   END_RUNG
   RUNG wire#powerrail
      I_Contact( "OUTPUT MAPING DB PLC 2"."P-301 A RO 1 HPP PUMP" )
      Move(in := 0, out1 => "AO SCALING DB".PV."VFD P-301A")
   END_RUNG
   // the same network as SCL:
   "SCALE AO_DB"("SET RPM" := "AO SCALING DB".SET."VFD P-301A",   // "SCALE AO"
                 "MIN RPM" := "AO SCALING DB".MIN."VFD P-301A",
                 "MAX RPM" := "AO SCALING DB".MAX."VFD P-301A",
                 "MIN HZ" := 0,
                 "MAX HZ" := 5000,
                 MODBUS => "MODBUS DB"."VFD_4 SEND");
   IF "OUTPUT MAPING DB PLC 2"."P-301 A RO 1 HPP PUMP" THEN
       "SCALE_DB"("SCALE MIN" := "AO SCALING DB".MIN."VFD P-301A",   // "SCALE"
                  "SCALE MAX" := "AO SCALING DB".MAX."VFD P-301A",
                  INPUT := "MODBUS DB"."VFD_4 SEND",
                  "RAW MIN" := 0,
                  "RAW MAX" := 5000,
                  "PV VALUE" => "AO SCALING DB".PV."VFD P-301A");
   END_IF;
   IF NOT "OUTPUT MAPING DB PLC 2"."P-301 A RO 1 HPP PUMP" THEN "AO SCALING DB".PV."VFD P-301A" := 0; END_IF;
END_REGION

REGION Network 5: VFD P-301B
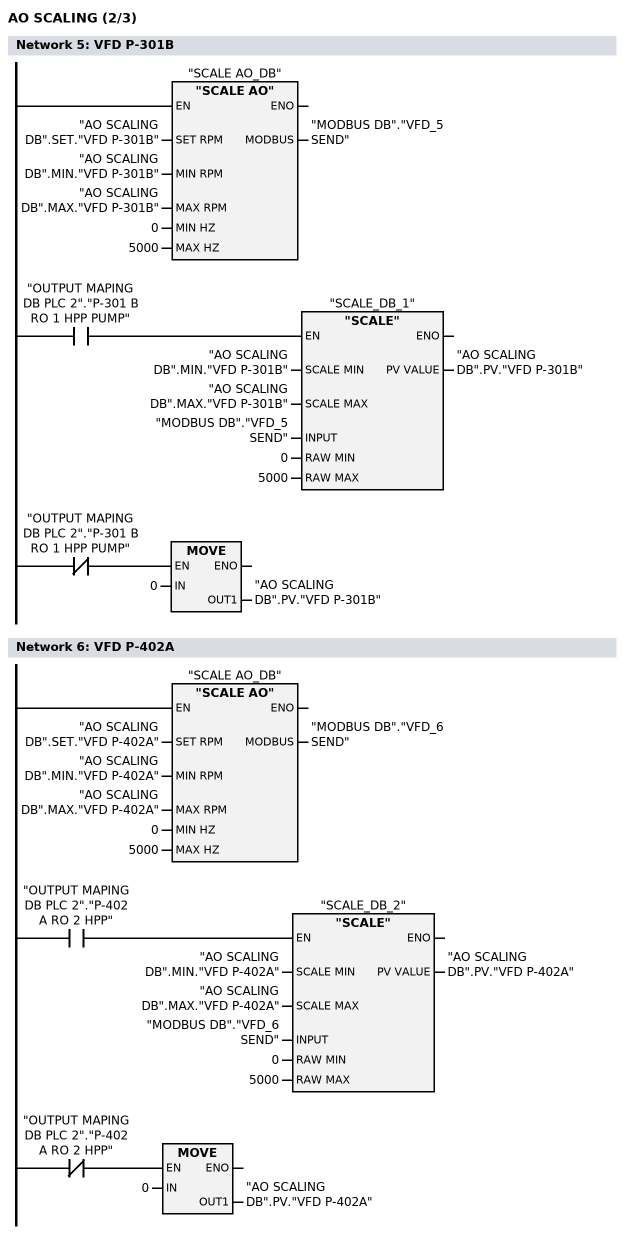
   RUNG wire#powerrail
      "SCALE AO_DB"("SET RPM" := "AO SCALING DB".SET."VFD P-301B", "MIN RPM" := "AO SCALING DB".MIN."VFD P-301B", "MAX RPM" := "AO SCALING DB".MAX."VFD P-301B", "MIN HZ" := 0, "MAX HZ" := 5000, MODBUS => "MODBUS DB"."VFD_5 SEND")
   END_RUNG
   RUNG wire#powerrail
      Contact( "OUTPUT MAPING DB PLC 2"."P-301 B RO 1 HPP PUMP" )
      "SCALE_DB_1"("SCALE MIN" := "AO SCALING DB".MIN."VFD P-301B", "SCALE MAX" := "AO SCALING DB".MAX."VFD P-301B", INPUT := "MODBUS DB"."VFD_5 SEND", "RAW MIN" := 0, "RAW MAX" := 5000, "PV VALUE" => "AO SCALING DB".PV."VFD P-301B")
   END_RUNG
   RUNG wire#powerrail
      I_Contact( "OUTPUT MAPING DB PLC 2"."P-301 B RO 1 HPP PUMP" )
      Move(in := 0, out1 => "AO SCALING DB".PV."VFD P-301B")
   END_RUNG
   // the same network as SCL:
   "SCALE AO_DB"("SET RPM" := "AO SCALING DB".SET."VFD P-301B",   // "SCALE AO"
                 "MIN RPM" := "AO SCALING DB".MIN."VFD P-301B",
                 "MAX RPM" := "AO SCALING DB".MAX."VFD P-301B",
                 "MIN HZ" := 0,
                 "MAX HZ" := 5000,
                 MODBUS => "MODBUS DB"."VFD_5 SEND");
   IF "OUTPUT MAPING DB PLC 2"."P-301 B RO 1 HPP PUMP" THEN
       "SCALE_DB_1"("SCALE MIN" := "AO SCALING DB".MIN."VFD P-301B",   // "SCALE"
                    "SCALE MAX" := "AO SCALING DB".MAX."VFD P-301B",
                    INPUT := "MODBUS DB"."VFD_5 SEND",
                    "RAW MIN" := 0,
                    "RAW MAX" := 5000,
                    "PV VALUE" => "AO SCALING DB".PV."VFD P-301B");
   END_IF;
   IF NOT "OUTPUT MAPING DB PLC 2"."P-301 B RO 1 HPP PUMP" THEN "AO SCALING DB".PV."VFD P-301B" := 0; END_IF;
END_REGION

REGION Network 6: VFD P-402A
   RUNG wire#powerrail
      "SCALE AO_DB"("SET RPM" := "AO SCALING DB".SET."VFD P-402A", "MIN RPM" := "AO SCALING DB".MIN."VFD P-402A", "MAX RPM" := "AO SCALING DB".MAX."VFD P-402A", "MIN HZ" := 0, "MAX HZ" := 5000, MODBUS => "MODBUS DB"."VFD_6 SEND")
   END_RUNG
   RUNG wire#powerrail
      Contact( "OUTPUT MAPING DB PLC 2"."P-402  A RO 2 HPP" )
      "SCALE_DB_2"("SCALE MIN" := "AO SCALING DB".MIN."VFD P-402A", "SCALE MAX" := "AO SCALING DB".MAX."VFD P-402A", INPUT := "MODBUS DB"."VFD_6 SEND", "RAW MIN" := 0, "RAW MAX" := 5000, "PV VALUE" => "AO SCALING DB".PV."VFD P-402A")
   END_RUNG
   RUNG wire#powerrail
      I_Contact( "OUTPUT MAPING DB PLC 2"."P-402  A RO 2 HPP" )
      Move(in := 0, out1 => "AO SCALING DB".PV."VFD P-402A")
   END_RUNG
   // the same network as SCL:
   "SCALE AO_DB"("SET RPM" := "AO SCALING DB".SET."VFD P-402A",   // "SCALE AO"
                 "MIN RPM" := "AO SCALING DB".MIN."VFD P-402A",
                 "MAX RPM" := "AO SCALING DB".MAX."VFD P-402A",
                 "MIN HZ" := 0,
                 "MAX HZ" := 5000,
                 MODBUS => "MODBUS DB"."VFD_6 SEND");
   IF "OUTPUT MAPING DB PLC 2"."P-402  A RO 2 HPP" THEN
       "SCALE_DB_2"("SCALE MIN" := "AO SCALING DB".MIN."VFD P-402A",   // "SCALE"
                    "SCALE MAX" := "AO SCALING DB".MAX."VFD P-402A",
                    INPUT := "MODBUS DB"."VFD_6 SEND",
                    "RAW MIN" := 0,
                    "RAW MAX" := 5000,
                    "PV VALUE" => "AO SCALING DB".PV."VFD P-402A");
   END_IF;
   IF NOT "OUTPUT MAPING DB PLC 2"."P-402  A RO 2 HPP" THEN "AO SCALING DB".PV."VFD P-402A" := 0; END_IF;
END_REGION

REGION Network 7: VFD P-402B
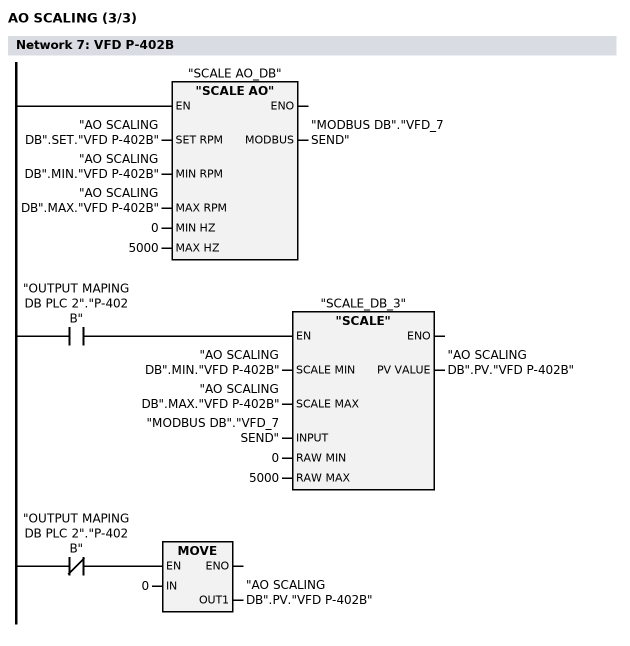
   RUNG wire#powerrail
      "SCALE AO_DB"("SET RPM" := "AO SCALING DB".SET."VFD P-402B", "MIN RPM" := "AO SCALING DB".MIN."VFD P-402B", "MAX RPM" := "AO SCALING DB".MAX."VFD P-402B", "MIN HZ" := 0, "MAX HZ" := 5000, MODBUS => "MODBUS DB"."VFD_7 SEND")
   END_RUNG
   RUNG wire#powerrail
      Contact( "OUTPUT MAPING DB PLC 2"."P-402 B" )
      "SCALE_DB_3"("SCALE MIN" := "AO SCALING DB".MIN."VFD P-402B", "SCALE MAX" := "AO SCALING DB".MAX."VFD P-402B", INPUT := "MODBUS DB"."VFD_7 SEND", "RAW MIN" := 0, "RAW MAX" := 5000, "PV VALUE" => "AO SCALING DB".PV."VFD P-402B")
   END_RUNG
   RUNG wire#powerrail
      I_Contact( "OUTPUT MAPING DB PLC 2"."P-402 B" )
      Move(in := 0, out1 => "AO SCALING DB".PV."VFD P-402B")
   END_RUNG
   // the same network as SCL:
   "SCALE AO_DB"("SET RPM" := "AO SCALING DB".SET."VFD P-402B",   // "SCALE AO"
                 "MIN RPM" := "AO SCALING DB".MIN."VFD P-402B",
                 "MAX RPM" := "AO SCALING DB".MAX."VFD P-402B",
                 "MIN HZ" := 0,
                 "MAX HZ" := 5000,
                 MODBUS => "MODBUS DB"."VFD_7 SEND");
   IF "OUTPUT MAPING DB PLC 2"."P-402 B" THEN
       "SCALE_DB_3"("SCALE MIN" := "AO SCALING DB".MIN."VFD P-402B",   // "SCALE"
                    "SCALE MAX" := "AO SCALING DB".MAX."VFD P-402B",
                    INPUT := "MODBUS DB"."VFD_7 SEND",
                    "RAW MIN" := 0,
                    "RAW MAX" := 5000,
                    "PV VALUE" => "AO SCALING DB".PV."VFD P-402B");
   END_IF;
   IF NOT "OUTPUT MAPING DB PLC 2"."P-402 B" THEN "AO SCALING DB".PV."VFD P-402B" := 0; END_IF;
END_REGION
END_FUNCTION

FUNCTION_BLOCK "SCALE AO"   // FB5, LAD
{ S7_Optimized_Access := 'TRUE' }
// stored: MemoryReserve 100, SetENOAutomatically false
   VAR_INPUT
      "SET RPM" : Real;
      "MIN RPM" : Real;
      "MAX RPM" : Real;
      "MIN HZ" : Int;
      "MAX HZ" : Int;
   END_VAR
   VAR_OUTPUT
      MODBUS : Int;
   END_VAR
   VAR_TEMP
      NOM : Real;
   END_VAR
BEGIN

REGION Network 1
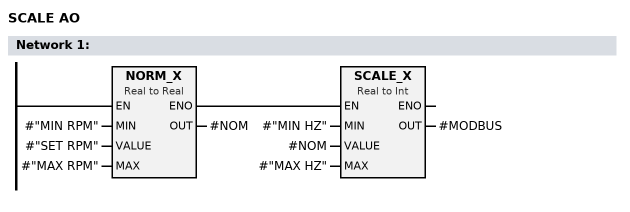
   RUNG wire#powerrail
      { S7_Templates := "[SrcType := Real, DestType := Real]" } Normalize(min := #"MIN RPM", value := #"SET RPM", max := #"MAX RPM", out => #NOM)
      { S7_Templates := "[SrcType := Real, DestType := Int]" } Scale(min := #"MIN HZ", value := #NOM, max := #"MAX HZ", out => #MODBUS)
   END_RUNG
   // the same network as SCL:
   #NOM := NORM_X(MIN := #"MIN RPM", VALUE := #"SET RPM", MAX := #"MAX RPM");
   #MODBUS := SCALE_X(MIN := #"MIN HZ", VALUE := #NOM, MAX := #"MAX HZ");
END_REGION
END_FUNCTION_BLOCK

FUNCTION "AUTO_SUBOUTPUT" : Void   // FC9, LAD
{ S7_Optimized_Access := 'TRUE' }
// stored: SetENOAutomatically false
BEGIN

REGION Network 1: P-202 A RO 1 FEED PUMP
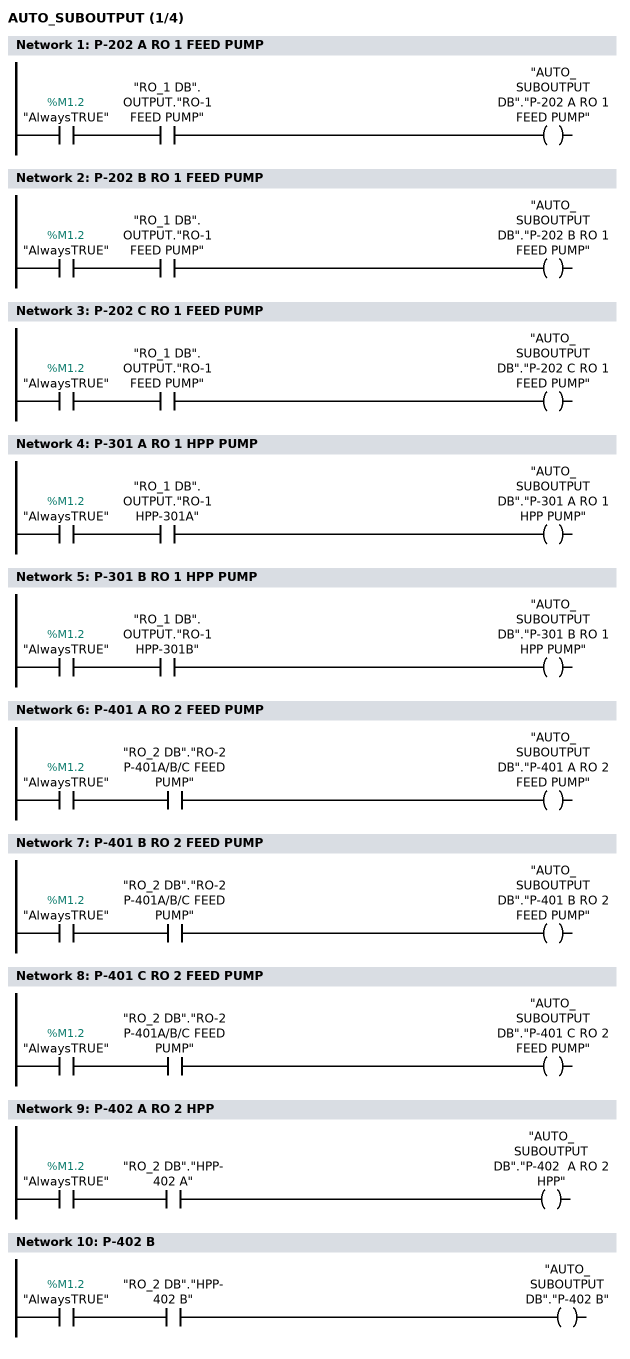
   RUNG wire#powerrail
      Contact( "AlwaysTRUE" )
      Contact( "RO_1 DB".OUTPUT."RO-1 FEED PUMP" )
      Coil( "AUTO_SUBOUTPUT DB"."P-202 A RO 1 FEED PUMP" )
   END_RUNG
   // the same network as SCL:
   "AUTO_SUBOUTPUT DB"."P-202 A RO 1 FEED PUMP" := "AlwaysTRUE" AND "RO_1 DB".OUTPUT."RO-1 FEED PUMP";
END_REGION

REGION Network 2: P-202 B RO 1 FEED PUMP
   RUNG wire#powerrail
      Contact( "AlwaysTRUE" )
      Contact( "RO_1 DB".OUTPUT."RO-1 FEED PUMP" )
      Coil( "AUTO_SUBOUTPUT DB"."P-202 B RO 1 FEED PUMP" )
   END_RUNG
   // the same network as SCL:
   "AUTO_SUBOUTPUT DB"."P-202 B RO 1 FEED PUMP" := "AlwaysTRUE" AND "RO_1 DB".OUTPUT."RO-1 FEED PUMP";
END_REGION

REGION Network 3: P-202 C RO 1 FEED PUMP
   RUNG wire#powerrail
      Contact( "AlwaysTRUE" )
      Contact( "RO_1 DB".OUTPUT."RO-1 FEED PUMP" )
      Coil( "AUTO_SUBOUTPUT DB"."P-202 C RO 1 FEED PUMP" )
   END_RUNG
   // the same network as SCL:
   "AUTO_SUBOUTPUT DB"."P-202 C RO 1 FEED PUMP" := "AlwaysTRUE" AND "RO_1 DB".OUTPUT."RO-1 FEED PUMP";
END_REGION

REGION Network 4: P-301 A RO 1 HPP PUMP
   RUNG wire#powerrail
      Contact( "AlwaysTRUE" )
      Contact( "RO_1 DB".OUTPUT."RO-1 HPP-301A" )
      Coil( "AUTO_SUBOUTPUT DB"."P-301 A RO 1 HPP PUMP" )
   END_RUNG
   // the same network as SCL:
   "AUTO_SUBOUTPUT DB"."P-301 A RO 1 HPP PUMP" := "AlwaysTRUE" AND "RO_1 DB".OUTPUT."RO-1 HPP-301A";
END_REGION

REGION Network 5: P-301 B RO 1 HPP PUMP
   RUNG wire#powerrail
      Contact( "AlwaysTRUE" )
      Contact( "RO_1 DB".OUTPUT."RO-1 HPP-301B" )
      Coil( "AUTO_SUBOUTPUT DB"."P-301 B RO 1 HPP PUMP" )
   END_RUNG
   // the same network as SCL:
   "AUTO_SUBOUTPUT DB"."P-301 B RO 1 HPP PUMP" := "AlwaysTRUE" AND "RO_1 DB".OUTPUT."RO-1 HPP-301B";
END_REGION

REGION Network 6: P-401 A RO 2 FEED PUMP
   RUNG wire#powerrail
      Contact( "AlwaysTRUE" )
      Contact( "RO_2 DB"."RO-2 P-401A/B/C FEED PUMP" )
      Coil( "AUTO_SUBOUTPUT DB"."P-401 A RO 2 FEED PUMP" )
   END_RUNG
   // the same network as SCL:
   "AUTO_SUBOUTPUT DB"."P-401 A RO 2 FEED PUMP" := "AlwaysTRUE" AND "RO_2 DB"."RO-2 P-401A/B/C FEED PUMP";
END_REGION

REGION Network 7: P-401 B RO 2 FEED PUMP
   RUNG wire#powerrail
      Contact( "AlwaysTRUE" )
      Contact( "RO_2 DB"."RO-2 P-401A/B/C FEED PUMP" )
      Coil( "AUTO_SUBOUTPUT DB"."P-401 B RO 2 FEED PUMP" )
   END_RUNG
   // the same network as SCL:
   "AUTO_SUBOUTPUT DB"."P-401 B RO 2 FEED PUMP" := "AlwaysTRUE" AND "RO_2 DB"."RO-2 P-401A/B/C FEED PUMP";
END_REGION

REGION Network 8: P-401 C RO 2 FEED PUMP
   RUNG wire#powerrail
      Contact( "AlwaysTRUE" )
      Contact( "RO_2 DB"."RO-2 P-401A/B/C FEED PUMP" )
      Coil( "AUTO_SUBOUTPUT DB"."P-401 C RO 2 FEED PUMP" )
   END_RUNG
   // the same network as SCL:
   "AUTO_SUBOUTPUT DB"."P-401 C RO 2 FEED PUMP" := "AlwaysTRUE" AND "RO_2 DB"."RO-2 P-401A/B/C FEED PUMP";
END_REGION

REGION Network 9: P-402 A RO 2 HPP
   RUNG wire#powerrail
      Contact( "AlwaysTRUE" )
      Contact( "RO_2 DB"."HPP-402 A" )
      Coil( "AUTO_SUBOUTPUT DB"."P-402  A RO 2 HPP" )
   END_RUNG
   // the same network as SCL:
   "AUTO_SUBOUTPUT DB"."P-402  A RO 2 HPP" := "AlwaysTRUE" AND "RO_2 DB"."HPP-402 A";
END_REGION

REGION Network 10: P-402 B
   RUNG wire#powerrail
      Contact( "AlwaysTRUE" )
      Contact( "RO_2 DB"."HPP-402 B" )
      Coil( "AUTO_SUBOUTPUT DB"."P-402 B" )
   END_RUNG
   // the same network as SCL:
   "AUTO_SUBOUTPUT DB"."P-402 B" := "AlwaysTRUE" AND "RO_2 DB"."HPP-402 B";
END_REGION

REGION Network 11: P-501 A EDI FEED PUMP
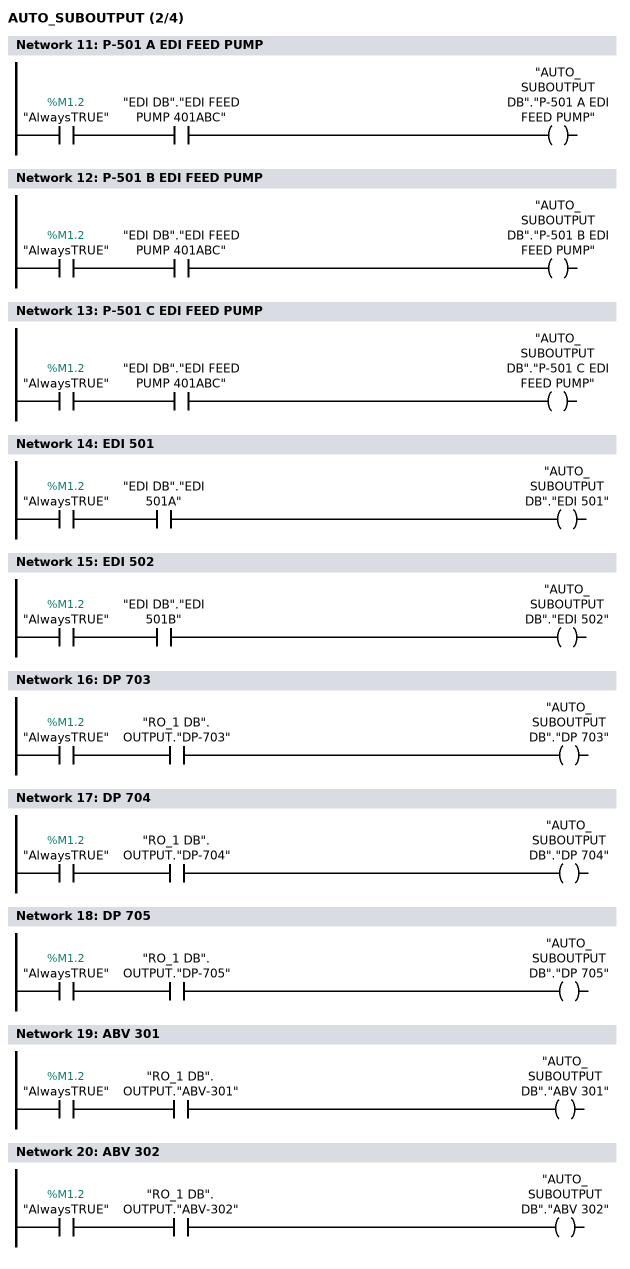
   RUNG wire#powerrail
      Contact( "AlwaysTRUE" )
      Contact( "EDI DB"."EDI FEED PUMP 401ABC" )
      Coil( "AUTO_SUBOUTPUT DB"."P-501 A EDI FEED PUMP" )
   END_RUNG
   // the same network as SCL:
   "AUTO_SUBOUTPUT DB"."P-501 A EDI FEED PUMP" := "AlwaysTRUE" AND "EDI DB"."EDI FEED PUMP 401ABC";
END_REGION

REGION Network 12: P-501 B EDI FEED PUMP
   RUNG wire#powerrail
      Contact( "AlwaysTRUE" )
      Contact( "EDI DB"."EDI FEED PUMP 401ABC" )
      Coil( "AUTO_SUBOUTPUT DB"."P-501 B EDI FEED PUMP" )
   END_RUNG
   // the same network as SCL:
   "AUTO_SUBOUTPUT DB"."P-501 B EDI FEED PUMP" := "AlwaysTRUE" AND "EDI DB"."EDI FEED PUMP 401ABC";
END_REGION

REGION Network 13: P-501 C EDI FEED PUMP
   RUNG wire#powerrail
      Contact( "AlwaysTRUE" )
      Contact( "EDI DB"."EDI FEED PUMP 401ABC" )
      Coil( "AUTO_SUBOUTPUT DB"."P-501 C EDI FEED PUMP" )
   END_RUNG
   // the same network as SCL:
   "AUTO_SUBOUTPUT DB"."P-501 C EDI FEED PUMP" := "AlwaysTRUE" AND "EDI DB"."EDI FEED PUMP 401ABC";
END_REGION

REGION Network 14: EDI 501
   RUNG wire#powerrail
      Contact( "AlwaysTRUE" )
      Contact( "EDI DB"."EDI 501A" )
      Coil( "AUTO_SUBOUTPUT DB"."EDI 501" )
   END_RUNG
   // the same network as SCL:
   "AUTO_SUBOUTPUT DB"."EDI 501" := "AlwaysTRUE" AND "EDI DB"."EDI 501A";
END_REGION

REGION Network 15: EDI 502
   RUNG wire#powerrail
      Contact( "AlwaysTRUE" )
      Contact( "EDI DB"."EDI 501B" )
      Coil( "AUTO_SUBOUTPUT DB"."EDI 502" )
   END_RUNG
   // the same network as SCL:
   "AUTO_SUBOUTPUT DB"."EDI 502" := "AlwaysTRUE" AND "EDI DB"."EDI 501B";
END_REGION

REGION Network 16: DP 703
   RUNG wire#powerrail
      Contact( "AlwaysTRUE" )
      Contact( "RO_1 DB".OUTPUT."DP-703" )
      Coil( "AUTO_SUBOUTPUT DB"."DP 703" )
   END_RUNG
   // the same network as SCL:
   "AUTO_SUBOUTPUT DB"."DP 703" := "AlwaysTRUE" AND "RO_1 DB".OUTPUT."DP-703";
END_REGION

REGION Network 17: DP 704
   RUNG wire#powerrail
      Contact( "AlwaysTRUE" )
      Contact( "RO_1 DB".OUTPUT."DP-704" )
      Coil( "AUTO_SUBOUTPUT DB"."DP 704" )
   END_RUNG
   // the same network as SCL:
   "AUTO_SUBOUTPUT DB"."DP 704" := "AlwaysTRUE" AND "RO_1 DB".OUTPUT."DP-704";
END_REGION

REGION Network 18: DP 705
   RUNG wire#powerrail
      Contact( "AlwaysTRUE" )
      Contact( "RO_1 DB".OUTPUT."DP-705" )
      Coil( "AUTO_SUBOUTPUT DB"."DP 705" )
   END_RUNG
   // the same network as SCL:
   "AUTO_SUBOUTPUT DB"."DP 705" := "AlwaysTRUE" AND "RO_1 DB".OUTPUT."DP-705";
END_REGION

REGION Network 19: ABV 301
   RUNG wire#powerrail
      Contact( "AlwaysTRUE" )
      Contact( "RO_1 DB".OUTPUT."ABV-301" )
      Coil( "AUTO_SUBOUTPUT DB"."ABV 301" )
   END_RUNG
   // the same network as SCL:
   "AUTO_SUBOUTPUT DB"."ABV 301" := "AlwaysTRUE" AND "RO_1 DB".OUTPUT."ABV-301";
END_REGION

REGION Network 20: ABV 302
   RUNG wire#powerrail
      Contact( "AlwaysTRUE" )
      Contact( "RO_1 DB".OUTPUT."ABV-302" )
      Coil( "AUTO_SUBOUTPUT DB"."ABV 302" )
   END_RUNG
   // the same network as SCL:
   "AUTO_SUBOUTPUT DB"."ABV 302" := "AlwaysTRUE" AND "RO_1 DB".OUTPUT."ABV-302";
END_REGION

REGION Network 21: AGLV-301
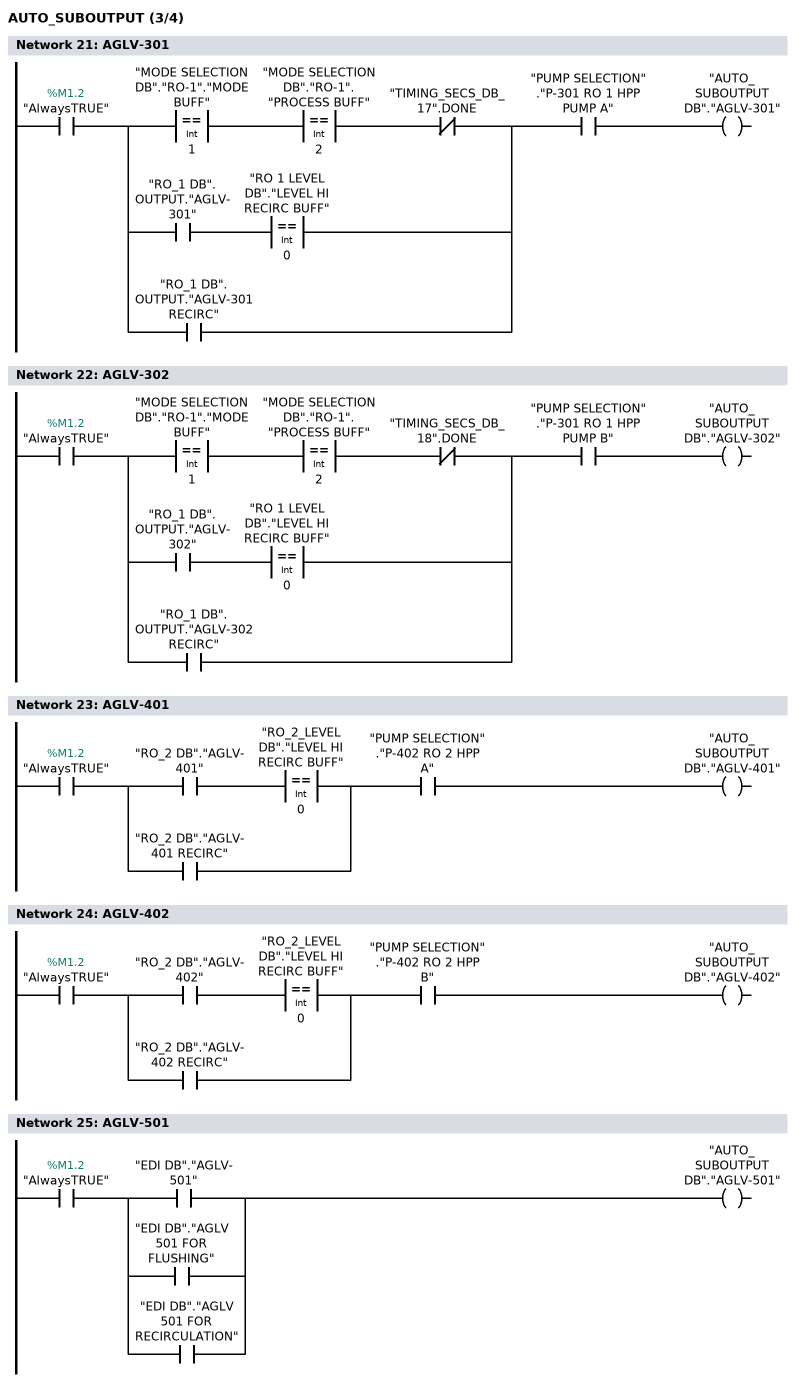
   RUNG wire#powerrail
      Contact( "AlwaysTRUE" )
      wire#w1
      { S7_Templates := "SrcType := Int" } EQ_Contact(in1 := "MODE SELECTION DB"."RO-1"."MODE BUFF", in2 := 1)
      { S7_Templates := "SrcType := Int" } EQ_Contact(in1 := "MODE SELECTION DB"."RO-1"."PROCESS BUFF", in2 := 2)
      I_Contact( "TIMING_SECS_DB_17".DONE )
      wire#w2
      Contact( "PUMP SELECTION"."P-301 RO 1 HPP PUMP A" )
      Coil( "AUTO_SUBOUTPUT DB"."AGLV-301" )
   END_RUNG
   RUNG wire#w1
      Contact( "RO_1 DB".OUTPUT."AGLV-301" )
      { S7_Templates := "SrcType := Int" } EQ_Contact(in1 := "RO 1 LEVEL DB"."LEVEL HI RECIRC BUFF", in2 := 0)
   END_RUNG wire#w2
   RUNG wire#w1
      Contact( "RO_1 DB".OUTPUT."AGLV-301 RECIRC" )
   END_RUNG wire#w2
   // the same network as SCL:
   "AUTO_SUBOUTPUT DB"."AGLV-301" := "AlwaysTRUE" AND ((("MODE SELECTION DB"."RO-1"."MODE BUFF" = 1) AND ("MODE SELECTION DB"."RO-1"."PROCESS BUFF" = 2) AND NOT "TIMING_SECS_DB_17".DONE) OR ("RO_1 DB".OUTPUT."AGLV-301" AND ("RO 1 LEVEL DB"."LEVEL HI RECIRC BUFF" = 0)) OR "RO_1 DB".OUTPUT."AGLV-301 RECIRC") AND "PUMP SELECTION"."P-301 RO 1 HPP PUMP A";
END_REGION

REGION Network 22: AGLV-302
   RUNG wire#powerrail
      Contact( "AlwaysTRUE" )
      wire#w1
      { S7_Templates := "SrcType := Int" } EQ_Contact(in1 := "MODE SELECTION DB"."RO-1"."MODE BUFF", in2 := 1)
      { S7_Templates := "SrcType := Int" } EQ_Contact(in1 := "MODE SELECTION DB"."RO-1"."PROCESS BUFF", in2 := 2)
      I_Contact( "TIMING_SECS_DB_18".DONE )
      wire#w2
      Contact( "PUMP SELECTION"."P-301 RO 1 HPP PUMP B" )
      Coil( "AUTO_SUBOUTPUT DB"."AGLV-302" )
   END_RUNG
   RUNG wire#w1
      Contact( "RO_1 DB".OUTPUT."AGLV-302" )
      { S7_Templates := "SrcType := Int" } EQ_Contact(in1 := "RO 1 LEVEL DB"."LEVEL HI RECIRC BUFF", in2 := 0)
   END_RUNG wire#w2
   RUNG wire#w1
      Contact( "RO_1 DB".OUTPUT."AGLV-302 RECIRC" )
   END_RUNG wire#w2
   // the same network as SCL:
   "AUTO_SUBOUTPUT DB"."AGLV-302" := "AlwaysTRUE" AND ((("MODE SELECTION DB"."RO-1"."MODE BUFF" = 1) AND ("MODE SELECTION DB"."RO-1"."PROCESS BUFF" = 2) AND NOT "TIMING_SECS_DB_18".DONE) OR ("RO_1 DB".OUTPUT."AGLV-302" AND ("RO 1 LEVEL DB"."LEVEL HI RECIRC BUFF" = 0)) OR "RO_1 DB".OUTPUT."AGLV-302 RECIRC") AND "PUMP SELECTION"."P-301 RO 1 HPP PUMP B";
END_REGION

REGION Network 23: AGLV-401
   RUNG wire#powerrail
      Contact( "AlwaysTRUE" )
      wire#w1
      Contact( "RO_2 DB"."AGLV-401" )
      { S7_Templates := "SrcType := Int" } EQ_Contact(in1 := "RO_2_LEVEL DB"."LEVEL HI RECIRC BUFF", in2 := 0)
      wire#w2
      Contact( "PUMP SELECTION"."P-402 RO 2 HPP A" )
      Coil( "AUTO_SUBOUTPUT DB"."AGLV-401" )
   END_RUNG
   RUNG wire#w1
      Contact( "RO_2 DB"."AGLV-401 RECIRC" )
   END_RUNG wire#w2
   // the same network as SCL:
   "AUTO_SUBOUTPUT DB"."AGLV-401" := "AlwaysTRUE" AND (("RO_2 DB"."AGLV-401" AND ("RO_2_LEVEL DB"."LEVEL HI RECIRC BUFF" = 0)) OR "RO_2 DB"."AGLV-401 RECIRC") AND "PUMP SELECTION"."P-402 RO 2 HPP A";
END_REGION

REGION Network 24: AGLV-402
   RUNG wire#powerrail
      Contact( "AlwaysTRUE" )
      wire#w1
      Contact( "RO_2 DB"."AGLV-402" )
      { S7_Templates := "SrcType := Int" } EQ_Contact(in1 := "RO_2_LEVEL DB"."LEVEL HI RECIRC BUFF", in2 := 0)
      wire#w2
      Contact( "PUMP SELECTION"."P-402 RO 2 HPP B" )
      Coil( "AUTO_SUBOUTPUT DB"."AGLV-402" )
   END_RUNG
   RUNG wire#w1
      Contact( "RO_2 DB"."AGLV-402 RECIRC" )
   END_RUNG wire#w2
   // the same network as SCL:
   "AUTO_SUBOUTPUT DB"."AGLV-402" := "AlwaysTRUE" AND (("RO_2 DB"."AGLV-402" AND ("RO_2_LEVEL DB"."LEVEL HI RECIRC BUFF" = 0)) OR "RO_2 DB"."AGLV-402 RECIRC") AND "PUMP SELECTION"."P-402 RO 2 HPP B";
END_REGION

REGION Network 25: AGLV-501
   RUNG wire#powerrail
      Contact( "AlwaysTRUE" )
      wire#w1
      Contact( "EDI DB"."AGLV-501" )
      wire#w2
      Coil( "AUTO_SUBOUTPUT DB"."AGLV-501" )
   END_RUNG
   RUNG wire#w1
      Contact( "EDI DB"."AGLV 501 FOR FLUSHING" )
   END_RUNG wire#w2
   RUNG wire#w1
      Contact( "EDI DB"."AGLV 501 FOR RECIRCULATION" )
   END_RUNG wire#w2
   // the same network as SCL:
   "AUTO_SUBOUTPUT DB"."AGLV-501" := "AlwaysTRUE" AND ("EDI DB"."AGLV-501" OR "EDI DB"."AGLV 501 FOR FLUSHING" OR "EDI DB"."AGLV 501 FOR RECIRCULATION");
END_REGION

REGION Network 26: AGLV-502
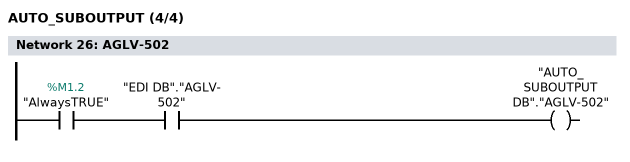
   RUNG wire#powerrail
      Contact( "AlwaysTRUE" )
      Contact( "EDI DB"."AGLV-502" )
      Coil( "AUTO_SUBOUTPUT DB"."AGLV-502" )
   END_RUNG
   // the same network as SCL:
   "AUTO_SUBOUTPUT DB"."AGLV-502" := "AlwaysTRUE" AND "EDI DB"."AGLV-502";
END_REGION
END_FUNCTION

FUNCTION "RO_1" : Void   // FC10, LAD
{ S7_Optimized_Access := 'TRUE' }
// stored: SetENOAutomatically false
   VAR_TEMP   // added for the SCL form of the ladder/FBD networks
      _w1 : Bool;
      _w2 : Bool;
      _w3 : Bool;
   END_VAR
BEGIN

REGION Network 1: ABV-301/ ABV-302
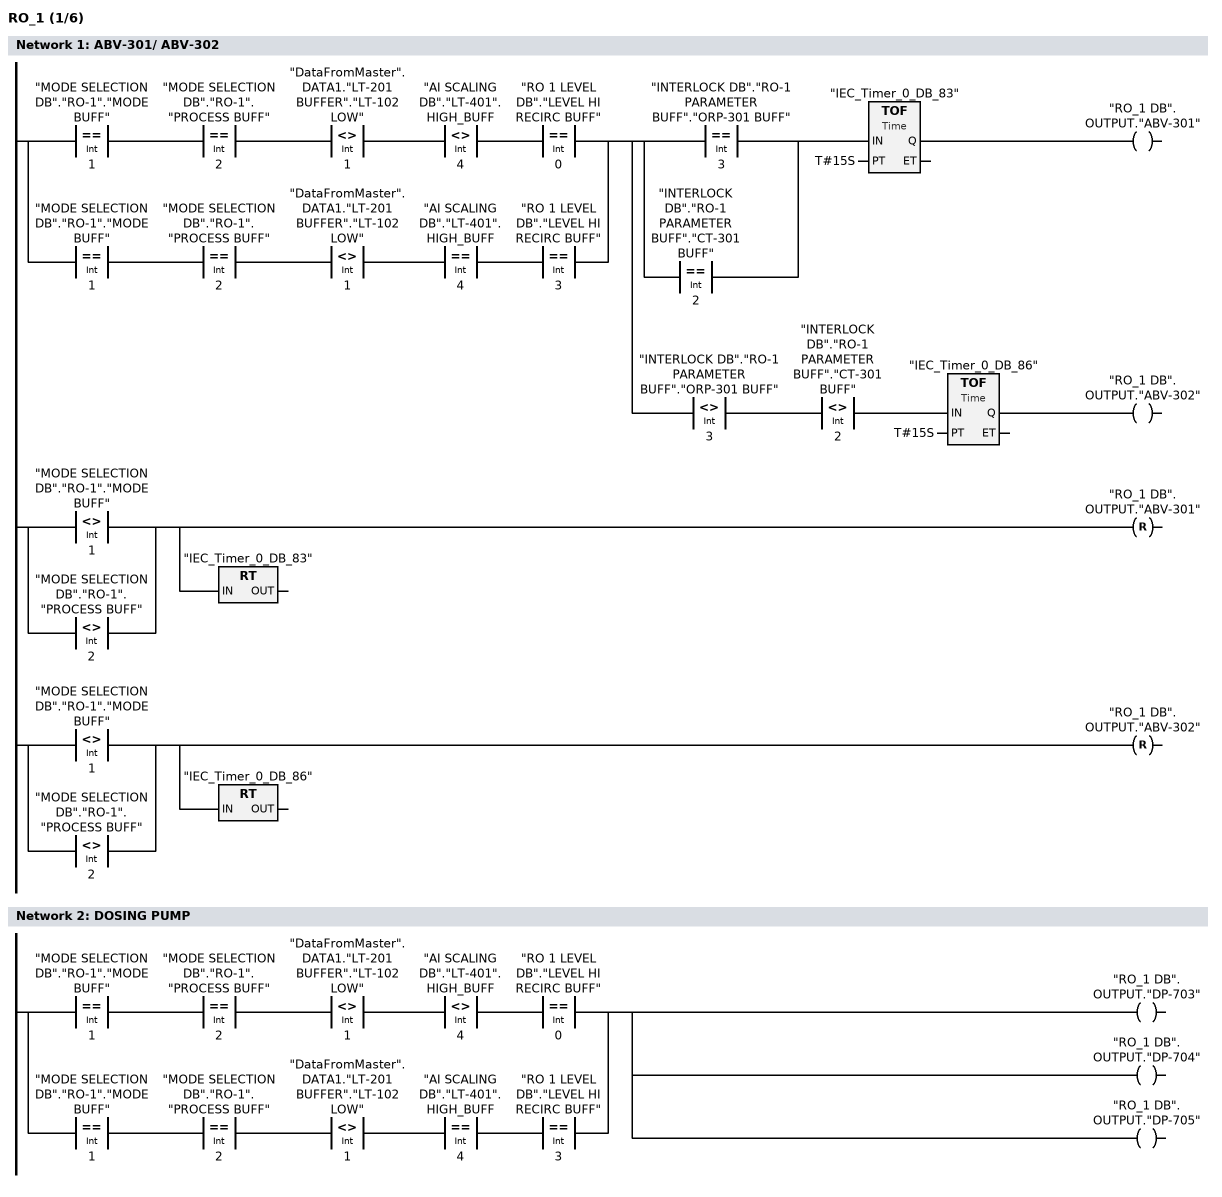
   RUNG wire#powerrail
      { S7_Templates := "SrcType := Int" } EQ_Contact(in1 := "MODE SELECTION DB"."RO-1"."MODE BUFF", in2 := 1)
      { S7_Templates := "SrcType := Int" } EQ_Contact(in1 := "MODE SELECTION DB"."RO-1"."PROCESS BUFF", in2 := 2)
      { S7_Templates := "SrcType := Int" } NE_Contact(in1 := "DataFromMaster".DATA1."LT-201 BUFFER"."LT-102 LOW", in2 := 1)
      { S7_Templates := "SrcType := Int" } NE_Contact(in1 := "AI SCALING DB"."LT-401".HIGH_BUFF, in2 := 4)
      { S7_Templates := "SrcType := Int" } EQ_Contact(in1 := "RO 1 LEVEL DB"."LEVEL HI RECIRC BUFF", in2 := 0)
      wire#w1
      { S7_Templates := "SrcType := Int" } EQ_Contact(in1 := "INTERLOCK DB"."RO-1 PARAMETER BUFF"."ORP-301 BUFF", in2 := 3)
      wire#w2
      { S7_Templates := "time_type := Time" } "IEC_Timer_0_DB_83".TOF(pt := T#15S, et =>)
      Coil( "RO_1 DB".OUTPUT."ABV-301" )
   END_RUNG
   RUNG wire#powerrail
      { S7_Templates := "SrcType := Int" } EQ_Contact(in1 := "MODE SELECTION DB"."RO-1"."MODE BUFF", in2 := 1)
      { S7_Templates := "SrcType := Int" } EQ_Contact(in1 := "MODE SELECTION DB"."RO-1"."PROCESS BUFF", in2 := 2)
      { S7_Templates := "SrcType := Int" } NE_Contact(in1 := "DataFromMaster".DATA1."LT-201 BUFFER"."LT-102 LOW", in2 := 1)
      { S7_Templates := "SrcType := Int" } EQ_Contact(in1 := "AI SCALING DB"."LT-401".HIGH_BUFF, in2 := 4)
      { S7_Templates := "SrcType := Int" } EQ_Contact(in1 := "RO 1 LEVEL DB"."LEVEL HI RECIRC BUFF", in2 := 3)
   END_RUNG wire#w1
   RUNG wire#w1
      { S7_Templates := "SrcType := Int" } EQ_Contact(in1 := "INTERLOCK DB"."RO-1 PARAMETER BUFF"."CT-301 BUFF", in2 := 2)
   END_RUNG wire#w2
   RUNG wire#w1
      { S7_Templates := "SrcType := Int" } NE_Contact(in1 := "INTERLOCK DB"."RO-1 PARAMETER BUFF"."ORP-301 BUFF", in2 := 3)
      { S7_Templates := "SrcType := Int" } NE_Contact(in1 := "INTERLOCK DB"."RO-1 PARAMETER BUFF"."CT-301 BUFF", in2 := 2)
      { S7_Templates := "time_type := Time" } "IEC_Timer_0_DB_86".TOF(pt := T#15S, et =>)
      Coil( "RO_1 DB".OUTPUT."ABV-302" )
   END_RUNG
   RUNG wire#powerrail
      { S7_Templates := "SrcType := Int" } NE_Contact(in1 := "MODE SELECTION DB"."RO-1"."MODE BUFF", in2 := 1)
      wire#w3
      R_Coil( "RO_1 DB".OUTPUT."ABV-301" )
   END_RUNG
   RUNG wire#powerrail
      { S7_Templates := "SrcType := Int" } NE_Contact(in1 := "MODE SELECTION DB"."RO-1"."PROCESS BUFF", in2 := 2)
   END_RUNG wire#w3
   RUNG wire#w3
      RT_Coil( "IEC_Timer_0_DB_83" )
   END_RUNG
   RUNG wire#powerrail
      { S7_Templates := "SrcType := Int" } NE_Contact(in1 := "MODE SELECTION DB"."RO-1"."MODE BUFF", in2 := 1)
      wire#w4
      R_Coil( "RO_1 DB".OUTPUT."ABV-302" )
   END_RUNG
   RUNG wire#powerrail
      { S7_Templates := "SrcType := Int" } NE_Contact(in1 := "MODE SELECTION DB"."RO-1"."PROCESS BUFF", in2 := 2)
   END_RUNG wire#w4
   RUNG wire#w4
      RT_Coil( "IEC_Timer_0_DB_86" )
   END_RUNG
   // the same network as SCL:
   #_w1 := (("MODE SELECTION DB"."RO-1"."MODE BUFF" = 1) AND ("MODE SELECTION DB"."RO-1"."PROCESS BUFF" = 2) AND ("DataFromMaster".DATA1."LT-201 BUFFER"."LT-102 LOW" <> 1) AND ("AI SCALING DB"."LT-401".HIGH_BUFF <> 4) AND ("RO 1 LEVEL DB"."LEVEL HI RECIRC BUFF" = 0)) OR (("MODE SELECTION DB"."RO-1"."MODE BUFF" = 1) AND ("MODE SELECTION DB"."RO-1"."PROCESS BUFF" = 2) AND ("DataFromMaster".DATA1."LT-201 BUFFER"."LT-102 LOW" <> 1) AND ("AI SCALING DB"."LT-401".HIGH_BUFF = 4) AND ("RO 1 LEVEL DB"."LEVEL HI RECIRC BUFF" = 3));
   "IEC_Timer_0_DB_83".TOF(IN := #_w1 AND (("INTERLOCK DB"."RO-1 PARAMETER BUFF"."ORP-301 BUFF" = 3) OR ("INTERLOCK DB"."RO-1 PARAMETER BUFF"."CT-301 BUFF" = 2)),
                           PT := T#15S);
   "RO_1 DB".OUTPUT."ABV-301" := "IEC_Timer_0_DB_83".Q;
   "IEC_Timer_0_DB_86".TOF(IN := #_w1 AND ("INTERLOCK DB"."RO-1 PARAMETER BUFF"."ORP-301 BUFF" <> 3) AND ("INTERLOCK DB"."RO-1 PARAMETER BUFF"."CT-301 BUFF" <> 2),
                           PT := T#15S);
   "RO_1 DB".OUTPUT."ABV-302" := "IEC_Timer_0_DB_86".Q;
   #_w2 := ("MODE SELECTION DB"."RO-1"."MODE BUFF" <> 1) OR ("MODE SELECTION DB"."RO-1"."PROCESS BUFF" <> 2);
   IF #_w2 THEN
       "RO_1 DB".OUTPUT."ABV-301" := FALSE;
       RESET_TIMER("IEC_Timer_0_DB_83");
   END_IF;
   #_w3 := ("MODE SELECTION DB"."RO-1"."MODE BUFF" <> 1) OR ("MODE SELECTION DB"."RO-1"."PROCESS BUFF" <> 2);
   IF #_w3 THEN
       "RO_1 DB".OUTPUT."ABV-302" := FALSE;
       RESET_TIMER("IEC_Timer_0_DB_86");
   END_IF;
END_REGION

REGION Network 2: DOSING PUMP
   RUNG wire#powerrail
      { S7_Templates := "SrcType := Int" } EQ_Contact(in1 := "MODE SELECTION DB"."RO-1"."MODE BUFF", in2 := 1)
      { S7_Templates := "SrcType := Int" } EQ_Contact(in1 := "MODE SELECTION DB"."RO-1"."PROCESS BUFF", in2 := 2)
      { S7_Templates := "SrcType := Int" } NE_Contact(in1 := "DataFromMaster".DATA1."LT-201 BUFFER"."LT-102 LOW", in2 := 1)
      { S7_Templates := "SrcType := Int" } NE_Contact(in1 := "AI SCALING DB"."LT-401".HIGH_BUFF, in2 := 4)
      { S7_Templates := "SrcType := Int" } EQ_Contact(in1 := "RO 1 LEVEL DB"."LEVEL HI RECIRC BUFF", in2 := 0)
      wire#w1
      Coil( "RO_1 DB".OUTPUT."DP-703" )
   END_RUNG
   RUNG wire#powerrail
      { S7_Templates := "SrcType := Int" } EQ_Contact(in1 := "MODE SELECTION DB"."RO-1"."MODE BUFF", in2 := 1)
      { S7_Templates := "SrcType := Int" } EQ_Contact(in1 := "MODE SELECTION DB"."RO-1"."PROCESS BUFF", in2 := 2)
      { S7_Templates := "SrcType := Int" } NE_Contact(in1 := "DataFromMaster".DATA1."LT-201 BUFFER"."LT-102 LOW", in2 := 1)
      { S7_Templates := "SrcType := Int" } EQ_Contact(in1 := "AI SCALING DB"."LT-401".HIGH_BUFF, in2 := 4)
      { S7_Templates := "SrcType := Int" } EQ_Contact(in1 := "RO 1 LEVEL DB"."LEVEL HI RECIRC BUFF", in2 := 3)
   END_RUNG wire#w1
   RUNG wire#w1
      Coil( "RO_1 DB".OUTPUT."DP-704" )
   END_RUNG
   RUNG wire#w1
      Coil( "RO_1 DB".OUTPUT."DP-705" )
   END_RUNG
   // the same network as SCL:
   "RO_1 DB".OUTPUT."DP-703" := (("MODE SELECTION DB"."RO-1"."MODE BUFF" = 1) AND ("MODE SELECTION DB"."RO-1"."PROCESS BUFF" = 2) AND ("DataFromMaster".DATA1."LT-201 BUFFER"."LT-102 LOW" <> 1) AND ("AI SCALING DB"."LT-401".HIGH_BUFF <> 4) AND ("RO 1 LEVEL DB"."LEVEL HI RECIRC BUFF" = 0)) OR (("MODE SELECTION DB"."RO-1"."MODE BUFF" = 1) AND ("MODE SELECTION DB"."RO-1"."PROCESS BUFF" = 2) AND ("DataFromMaster".DATA1."LT-201 BUFFER"."LT-102 LOW" <> 1) AND ("AI SCALING DB"."LT-401".HIGH_BUFF = 4) AND ("RO 1 LEVEL DB"."LEVEL HI RECIRC BUFF" = 3));
   "RO_1 DB".OUTPUT."DP-704" := "RO_1 DB".OUTPUT."DP-703";
   "RO_1 DB".OUTPUT."DP-705" := "RO_1 DB".OUTPUT."DP-703";
END_REGION

REGION Network 3: RO-1 FEED PUMP
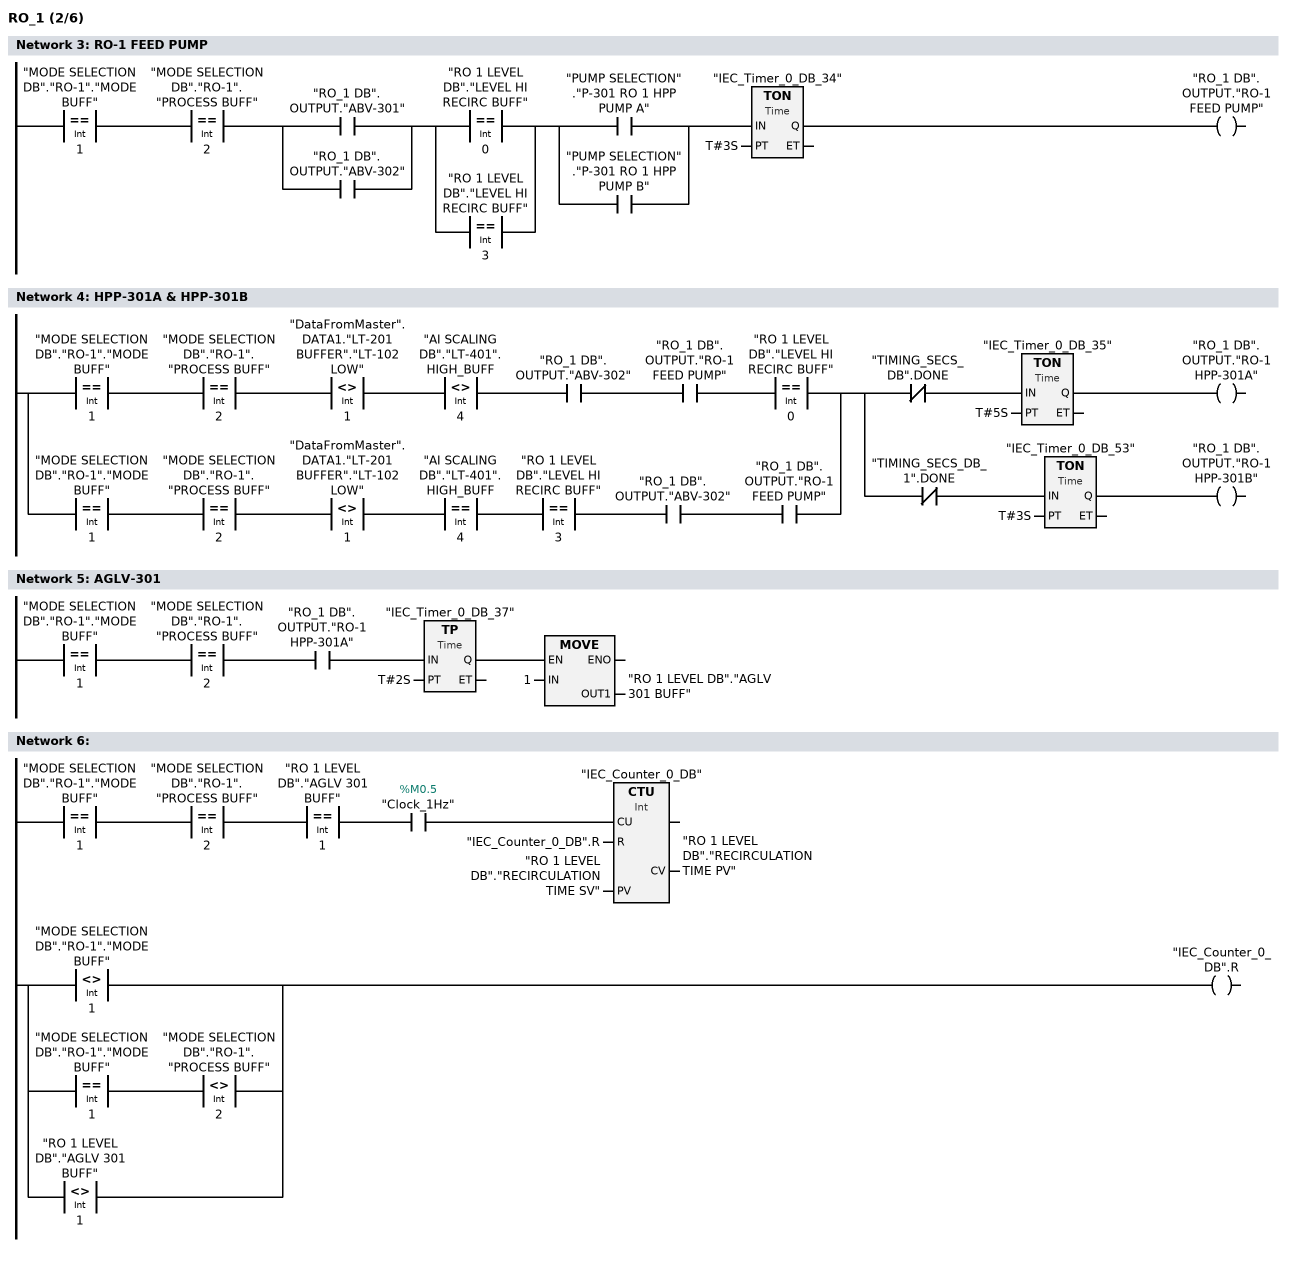
   RUNG wire#powerrail
      { S7_Templates := "SrcType := Int" } EQ_Contact(in1 := "MODE SELECTION DB"."RO-1"."MODE BUFF", in2 := 1)
      { S7_Templates := "SrcType := Int" } EQ_Contact(in1 := "MODE SELECTION DB"."RO-1"."PROCESS BUFF", in2 := 2)
      wire#w1
      Contact( "RO_1 DB".OUTPUT."ABV-301" )
      wire#w2
      { S7_Templates := "SrcType := Int" } EQ_Contact(in1 := "RO 1 LEVEL DB"."LEVEL HI RECIRC BUFF", in2 := 0)
      wire#w3
      Contact( "PUMP SELECTION"."P-301 RO 1 HPP PUMP A" )
      wire#w4
      { S7_Templates := "time_type := Time" } "IEC_Timer_0_DB_34".TON(pt := T#3S, et =>)
      Coil( "RO_1 DB".OUTPUT."RO-1 FEED PUMP" )
   END_RUNG
   RUNG wire#w1
      Contact( "RO_1 DB".OUTPUT."ABV-302" )
   END_RUNG wire#w2
   RUNG wire#w2
      { S7_Templates := "SrcType := Int" } EQ_Contact(in1 := "RO 1 LEVEL DB"."LEVEL HI RECIRC BUFF", in2 := 3)
   END_RUNG wire#w3
   RUNG wire#w3
      Contact( "PUMP SELECTION"."P-301 RO 1 HPP PUMP B" )
   END_RUNG wire#w4
   // the same network as SCL:
   "IEC_Timer_0_DB_34".TON(IN := ("MODE SELECTION DB"."RO-1"."MODE BUFF" = 1) AND ("MODE SELECTION DB"."RO-1"."PROCESS BUFF" = 2) AND ("RO_1 DB".OUTPUT."ABV-301" OR "RO_1 DB".OUTPUT."ABV-302") AND (("RO 1 LEVEL DB"."LEVEL HI RECIRC BUFF" = 0) OR ("RO 1 LEVEL DB"."LEVEL HI RECIRC BUFF" = 3)) AND ("PUMP SELECTION"."P-301 RO 1 HPP PUMP A" OR "PUMP SELECTION"."P-301 RO 1 HPP PUMP B"),
                           PT := T#3S);
   "RO_1 DB".OUTPUT."RO-1 FEED PUMP" := "IEC_Timer_0_DB_34".Q;
END_REGION

REGION Network 4: HPP-301A & HPP-301B
   RUNG wire#powerrail
      { S7_Templates := "SrcType := Int" } EQ_Contact(in1 := "MODE SELECTION DB"."RO-1"."MODE BUFF", in2 := 1)
      { S7_Templates := "SrcType := Int" } EQ_Contact(in1 := "MODE SELECTION DB"."RO-1"."PROCESS BUFF", in2 := 2)
      { S7_Templates := "SrcType := Int" } NE_Contact(in1 := "DataFromMaster".DATA1."LT-201 BUFFER"."LT-102 LOW", in2 := 1)
      { S7_Templates := "SrcType := Int" } NE_Contact(in1 := "AI SCALING DB"."LT-401".HIGH_BUFF, in2 := 4)
      Contact( "RO_1 DB".OUTPUT."ABV-302" )
      Contact( "RO_1 DB".OUTPUT."RO-1 FEED PUMP" )
      { S7_Templates := "SrcType := Int" } EQ_Contact(in1 := "RO 1 LEVEL DB"."LEVEL HI RECIRC BUFF", in2 := 0)
      wire#w1
      I_Contact( "TIMING_SECS_DB".DONE )
      { S7_Templates := "time_type := Time" } "IEC_Timer_0_DB_35".TON(pt := T#5S, et =>)
      Coil( "RO_1 DB".OUTPUT."RO-1 HPP-301A" )
   END_RUNG
   RUNG wire#powerrail
      { S7_Templates := "SrcType := Int" } EQ_Contact(in1 := "MODE SELECTION DB"."RO-1"."MODE BUFF", in2 := 1)
      { S7_Templates := "SrcType := Int" } EQ_Contact(in1 := "MODE SELECTION DB"."RO-1"."PROCESS BUFF", in2 := 2)
      { S7_Templates := "SrcType := Int" } NE_Contact(in1 := "DataFromMaster".DATA1."LT-201 BUFFER"."LT-102 LOW", in2 := 1)
      { S7_Templates := "SrcType := Int" } EQ_Contact(in1 := "AI SCALING DB"."LT-401".HIGH_BUFF, in2 := 4)
      { S7_Templates := "SrcType := Int" } EQ_Contact(in1 := "RO 1 LEVEL DB"."LEVEL HI RECIRC BUFF", in2 := 3)
      Contact( "RO_1 DB".OUTPUT."ABV-302" )
      Contact( "RO_1 DB".OUTPUT."RO-1 FEED PUMP" )
   END_RUNG wire#w1
   RUNG wire#w1
      I_Contact( "TIMING_SECS_DB_1".DONE )
      { S7_Templates := "time_type := Time" } "IEC_Timer_0_DB_53".TON(pt := T#3S, et =>)
      Coil( "RO_1 DB".OUTPUT."RO-1 HPP-301B" )
   END_RUNG
   // the same network as SCL:
   #_w1 := (("MODE SELECTION DB"."RO-1"."MODE BUFF" = 1) AND ("MODE SELECTION DB"."RO-1"."PROCESS BUFF" = 2) AND ("DataFromMaster".DATA1."LT-201 BUFFER"."LT-102 LOW" <> 1) AND ("AI SCALING DB"."LT-401".HIGH_BUFF <> 4) AND "RO_1 DB".OUTPUT."ABV-302" AND "RO_1 DB".OUTPUT."RO-1 FEED PUMP" AND ("RO 1 LEVEL DB"."LEVEL HI RECIRC BUFF" = 0)) OR (("MODE SELECTION DB"."RO-1"."MODE BUFF" = 1) AND ("MODE SELECTION DB"."RO-1"."PROCESS BUFF" = 2) AND ("DataFromMaster".DATA1."LT-201 BUFFER"."LT-102 LOW" <> 1) AND ("AI SCALING DB"."LT-401".HIGH_BUFF = 4) AND ("RO 1 LEVEL DB"."LEVEL HI RECIRC BUFF" = 3) AND "RO_1 DB".OUTPUT."ABV-302" AND "RO_1 DB".OUTPUT."RO-1 FEED PUMP");
   "IEC_Timer_0_DB_35".TON(IN := #_w1 AND NOT "TIMING_SECS_DB".DONE, PT := T#5S);
   "RO_1 DB".OUTPUT."RO-1 HPP-301A" := "IEC_Timer_0_DB_35".Q;
   "IEC_Timer_0_DB_53".TON(IN := #_w1 AND NOT "TIMING_SECS_DB_1".DONE, PT := T#3S);
   "RO_1 DB".OUTPUT."RO-1 HPP-301B" := "IEC_Timer_0_DB_53".Q;
END_REGION

REGION Network 5: AGLV-301
   RUNG wire#powerrail
      { S7_Templates := "SrcType := Int" } EQ_Contact(in1 := "MODE SELECTION DB"."RO-1"."MODE BUFF", in2 := 1)
      { S7_Templates := "SrcType := Int" } EQ_Contact(in1 := "MODE SELECTION DB"."RO-1"."PROCESS BUFF", in2 := 2)
      Contact( "RO_1 DB".OUTPUT."RO-1 HPP-301A" )
      { S7_Templates := "time_type := Time" } "IEC_Timer_0_DB_37".TP(pt := T#2S, et =>)
      Move(in := 1, out1 => "RO 1 LEVEL DB"."AGLV 301 BUFF")
   END_RUNG
   // the same network as SCL:
   "IEC_Timer_0_DB_37".TP(IN := ("MODE SELECTION DB"."RO-1"."MODE BUFF" = 1) AND ("MODE SELECTION DB"."RO-1"."PROCESS BUFF" = 2) AND "RO_1 DB".OUTPUT."RO-1 HPP-301A",
                          PT := T#2S);
   IF "IEC_Timer_0_DB_37".Q THEN "RO 1 LEVEL DB"."AGLV 301 BUFF" := 1; END_IF;
END_REGION

REGION Network 6
   RUNG wire#powerrail
      { S7_Templates := "SrcType := Int" } EQ_Contact(in1 := "MODE SELECTION DB"."RO-1"."MODE BUFF", in2 := 1)
      { S7_Templates := "SrcType := Int" } EQ_Contact(in1 := "MODE SELECTION DB"."RO-1"."PROCESS BUFF", in2 := 2)
      { S7_Templates := "SrcType := Int" } EQ_Contact(in1 := "RO 1 LEVEL DB"."AGLV 301 BUFF", in2 := 1)
      Contact( "Clock_1Hz" )
      { S7_Templates := "value_type := Int" } "IEC_Counter_0_DB".CTU(r := "IEC_Counter_0_DB".R, pv := "RO 1 LEVEL DB"."RECIRCULATION TIME SV", cv => "RO 1 LEVEL DB"."RECIRCULATION TIME PV")
   END_RUNG
   RUNG wire#powerrail
      { S7_Templates := "SrcType := Int" } NE_Contact(in1 := "MODE SELECTION DB"."RO-1"."MODE BUFF", in2 := 1)
      wire#w1
      Coil( "IEC_Counter_0_DB".R )
   END_RUNG
   RUNG wire#powerrail
      { S7_Templates := "SrcType := Int" } EQ_Contact(in1 := "MODE SELECTION DB"."RO-1"."MODE BUFF", in2 := 1)
      { S7_Templates := "SrcType := Int" } NE_Contact(in1 := "MODE SELECTION DB"."RO-1"."PROCESS BUFF", in2 := 2)
   END_RUNG wire#w1
   RUNG wire#powerrail
      { S7_Templates := "SrcType := Int" } NE_Contact(in1 := "RO 1 LEVEL DB"."AGLV 301 BUFF", in2 := 1)
   END_RUNG wire#w1
   // the same network as SCL:
   "IEC_Counter_0_DB".CTU(CU := ("MODE SELECTION DB"."RO-1"."MODE BUFF" = 1) AND ("MODE SELECTION DB"."RO-1"."PROCESS BUFF" = 2) AND ("RO 1 LEVEL DB"."AGLV 301 BUFF" = 1) AND "Clock_1Hz",
                          R := "IEC_Counter_0_DB".R,
                          PV := "RO 1 LEVEL DB"."RECIRCULATION TIME SV",
                          CV => "RO 1 LEVEL DB"."RECIRCULATION TIME PV");
   "IEC_Counter_0_DB".R := ("MODE SELECTION DB"."RO-1"."MODE BUFF" <> 1) OR (("MODE SELECTION DB"."RO-1"."MODE BUFF" = 1) AND ("MODE SELECTION DB"."RO-1"."PROCESS BUFF" <> 2)) OR ("RO 1 LEVEL DB"."AGLV 301 BUFF" <> 1);
END_REGION

REGION Network 7
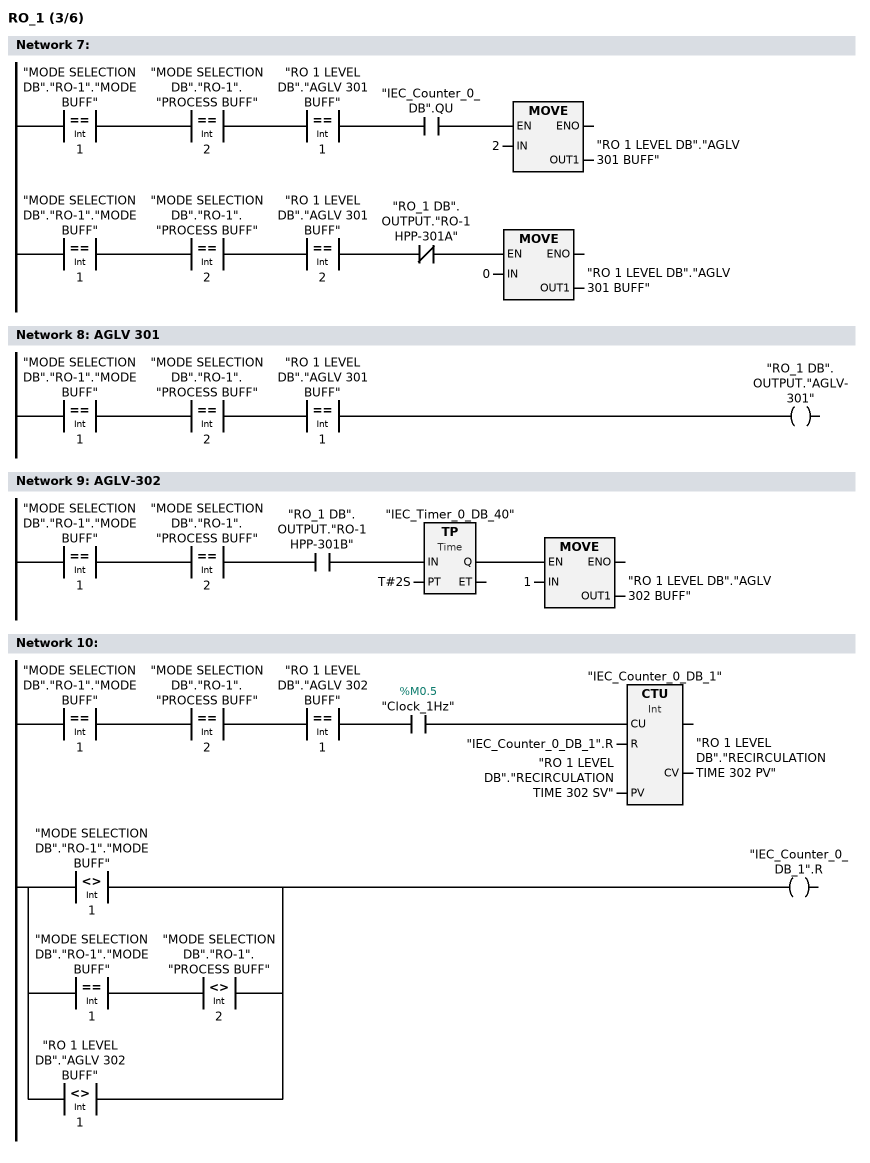
   RUNG wire#powerrail
      { S7_Templates := "SrcType := Int" } EQ_Contact(in1 := "MODE SELECTION DB"."RO-1"."MODE BUFF", in2 := 1)
      { S7_Templates := "SrcType := Int" } EQ_Contact(in1 := "MODE SELECTION DB"."RO-1"."PROCESS BUFF", in2 := 2)
      { S7_Templates := "SrcType := Int" } EQ_Contact(in1 := "RO 1 LEVEL DB"."AGLV 301 BUFF", in2 := 1)
      Contact( "IEC_Counter_0_DB".QU )
      Move(in := 2, out1 => "RO 1 LEVEL DB"."AGLV 301 BUFF")
   END_RUNG
   RUNG wire#powerrail
      { S7_Templates := "SrcType := Int" } EQ_Contact(in1 := "MODE SELECTION DB"."RO-1"."MODE BUFF", in2 := 1)
      { S7_Templates := "SrcType := Int" } EQ_Contact(in1 := "MODE SELECTION DB"."RO-1"."PROCESS BUFF", in2 := 2)
      { S7_Templates := "SrcType := Int" } EQ_Contact(in1 := "RO 1 LEVEL DB"."AGLV 301 BUFF", in2 := 2)
      I_Contact( "RO_1 DB".OUTPUT."RO-1 HPP-301A" )
      Move(in := 0, out1 => "RO 1 LEVEL DB"."AGLV 301 BUFF")
   END_RUNG
   // the same network as SCL:
   IF ("MODE SELECTION DB"."RO-1"."MODE BUFF" = 1) AND ("MODE SELECTION DB"."RO-1"."PROCESS BUFF" = 2) AND ("RO 1 LEVEL DB"."AGLV 301 BUFF" = 1) AND "IEC_Counter_0_DB".QU THEN
       "RO 1 LEVEL DB"."AGLV 301 BUFF" := 2;
   END_IF;
   IF ("MODE SELECTION DB"."RO-1"."MODE BUFF" = 1) AND ("MODE SELECTION DB"."RO-1"."PROCESS BUFF" = 2) AND ("RO 1 LEVEL DB"."AGLV 301 BUFF" = 2) AND NOT "RO_1 DB".OUTPUT."RO-1 HPP-301A" THEN
       "RO 1 LEVEL DB"."AGLV 301 BUFF" := 0;
   END_IF;
END_REGION

REGION Network 8: AGLV 301
   RUNG wire#powerrail
      { S7_Templates := "SrcType := Int" } EQ_Contact(in1 := "MODE SELECTION DB"."RO-1"."MODE BUFF", in2 := 1)
      { S7_Templates := "SrcType := Int" } EQ_Contact(in1 := "MODE SELECTION DB"."RO-1"."PROCESS BUFF", in2 := 2)
      { S7_Templates := "SrcType := Int" } EQ_Contact(in1 := "RO 1 LEVEL DB"."AGLV 301 BUFF", in2 := 1)
      Coil( "RO_1 DB".OUTPUT."AGLV-301" )
   END_RUNG
   // the same network as SCL:
   "RO_1 DB".OUTPUT."AGLV-301" := ("MODE SELECTION DB"."RO-1"."MODE BUFF" = 1) AND ("MODE SELECTION DB"."RO-1"."PROCESS BUFF" = 2) AND ("RO 1 LEVEL DB"."AGLV 301 BUFF" = 1);
END_REGION

REGION Network 9: AGLV-302
   RUNG wire#powerrail
      { S7_Templates := "SrcType := Int" } EQ_Contact(in1 := "MODE SELECTION DB"."RO-1"."MODE BUFF", in2 := 1)
      { S7_Templates := "SrcType := Int" } EQ_Contact(in1 := "MODE SELECTION DB"."RO-1"."PROCESS BUFF", in2 := 2)
      Contact( "RO_1 DB".OUTPUT."RO-1 HPP-301B" )
      { S7_Templates := "time_type := Time" } "IEC_Timer_0_DB_40".TP(pt := T#2S, et =>)
      Move(in := 1, out1 => "RO 1 LEVEL DB"."AGLV 302 BUFF")
   END_RUNG
   // the same network as SCL:
   "IEC_Timer_0_DB_40".TP(IN := ("MODE SELECTION DB"."RO-1"."MODE BUFF" = 1) AND ("MODE SELECTION DB"."RO-1"."PROCESS BUFF" = 2) AND "RO_1 DB".OUTPUT."RO-1 HPP-301B",
                          PT := T#2S);
   IF "IEC_Timer_0_DB_40".Q THEN "RO 1 LEVEL DB"."AGLV 302 BUFF" := 1; END_IF;
END_REGION

REGION Network 10
   RUNG wire#powerrail
      { S7_Templates := "SrcType := Int" } EQ_Contact(in1 := "MODE SELECTION DB"."RO-1"."MODE BUFF", in2 := 1)
      { S7_Templates := "SrcType := Int" } EQ_Contact(in1 := "MODE SELECTION DB"."RO-1"."PROCESS BUFF", in2 := 2)
      { S7_Templates := "SrcType := Int" } EQ_Contact(in1 := "RO 1 LEVEL DB"."AGLV 302 BUFF", in2 := 1)
      Contact( "Clock_1Hz" )
      { S7_Templates := "value_type := Int" } "IEC_Counter_0_DB_1".CTU(r := "IEC_Counter_0_DB_1".R, pv := "RO 1 LEVEL DB"."RECIRCULATION TIME 302 SV", cv => "RO 1 LEVEL DB"."RECIRCULATION TIME 302 PV")
   END_RUNG
   RUNG wire#powerrail
      { S7_Templates := "SrcType := Int" } NE_Contact(in1 := "MODE SELECTION DB"."RO-1"."MODE BUFF", in2 := 1)
      wire#w1
      Coil( "IEC_Counter_0_DB_1".R )
   END_RUNG
   RUNG wire#powerrail
      { S7_Templates := "SrcType := Int" } EQ_Contact(in1 := "MODE SELECTION DB"."RO-1"."MODE BUFF", in2 := 1)
      { S7_Templates := "SrcType := Int" } NE_Contact(in1 := "MODE SELECTION DB"."RO-1"."PROCESS BUFF", in2 := 2)
   END_RUNG wire#w1
   RUNG wire#powerrail
      { S7_Templates := "SrcType := Int" } NE_Contact(in1 := "RO 1 LEVEL DB"."AGLV 302 BUFF", in2 := 1)
   END_RUNG wire#w1
   // the same network as SCL:
   "IEC_Counter_0_DB_1".CTU(CU := ("MODE SELECTION DB"."RO-1"."MODE BUFF" = 1) AND ("MODE SELECTION DB"."RO-1"."PROCESS BUFF" = 2) AND ("RO 1 LEVEL DB"."AGLV 302 BUFF" = 1) AND "Clock_1Hz",
                           R := "IEC_Counter_0_DB_1".R,
                           PV := "RO 1 LEVEL DB"."RECIRCULATION TIME 302 SV",
                           CV => "RO 1 LEVEL DB"."RECIRCULATION TIME 302 PV");
   "IEC_Counter_0_DB_1".R := ("MODE SELECTION DB"."RO-1"."MODE BUFF" <> 1) OR (("MODE SELECTION DB"."RO-1"."MODE BUFF" = 1) AND ("MODE SELECTION DB"."RO-1"."PROCESS BUFF" <> 2)) OR ("RO 1 LEVEL DB"."AGLV 302 BUFF" <> 1);
END_REGION

REGION Network 11
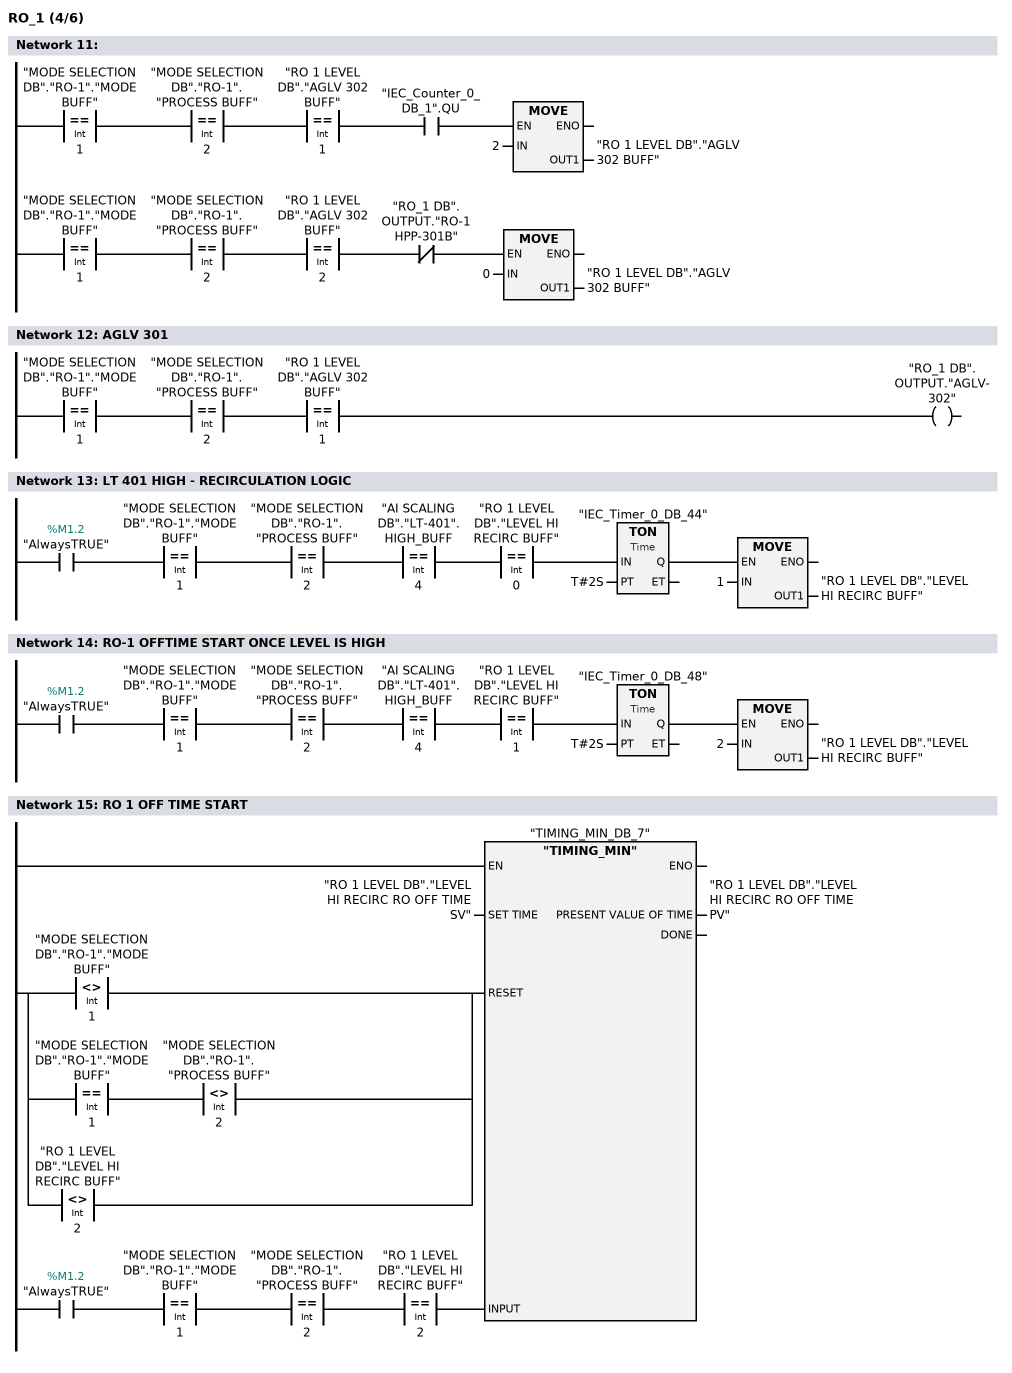
   RUNG wire#powerrail
      { S7_Templates := "SrcType := Int" } EQ_Contact(in1 := "MODE SELECTION DB"."RO-1"."MODE BUFF", in2 := 1)
      { S7_Templates := "SrcType := Int" } EQ_Contact(in1 := "MODE SELECTION DB"."RO-1"."PROCESS BUFF", in2 := 2)
      { S7_Templates := "SrcType := Int" } EQ_Contact(in1 := "RO 1 LEVEL DB"."AGLV 302 BUFF", in2 := 1)
      Contact( "IEC_Counter_0_DB_1".QU )
      Move(in := 2, out1 => "RO 1 LEVEL DB"."AGLV 302 BUFF")
   END_RUNG
   RUNG wire#powerrail
      { S7_Templates := "SrcType := Int" } EQ_Contact(in1 := "MODE SELECTION DB"."RO-1"."MODE BUFF", in2 := 1)
      { S7_Templates := "SrcType := Int" } EQ_Contact(in1 := "MODE SELECTION DB"."RO-1"."PROCESS BUFF", in2 := 2)
      { S7_Templates := "SrcType := Int" } EQ_Contact(in1 := "RO 1 LEVEL DB"."AGLV 302 BUFF", in2 := 2)
      I_Contact( "RO_1 DB".OUTPUT."RO-1 HPP-301B" )
      Move(in := 0, out1 => "RO 1 LEVEL DB"."AGLV 302 BUFF")
   END_RUNG
   // the same network as SCL:
   IF ("MODE SELECTION DB"."RO-1"."MODE BUFF" = 1) AND ("MODE SELECTION DB"."RO-1"."PROCESS BUFF" = 2) AND ("RO 1 LEVEL DB"."AGLV 302 BUFF" = 1) AND "IEC_Counter_0_DB_1".QU THEN
       "RO 1 LEVEL DB"."AGLV 302 BUFF" := 2;
   END_IF;
   IF ("MODE SELECTION DB"."RO-1"."MODE BUFF" = 1) AND ("MODE SELECTION DB"."RO-1"."PROCESS BUFF" = 2) AND ("RO 1 LEVEL DB"."AGLV 302 BUFF" = 2) AND NOT "RO_1 DB".OUTPUT."RO-1 HPP-301B" THEN
       "RO 1 LEVEL DB"."AGLV 302 BUFF" := 0;
   END_IF;
END_REGION

REGION Network 12: AGLV 301
   RUNG wire#powerrail
      { S7_Templates := "SrcType := Int" } EQ_Contact(in1 := "MODE SELECTION DB"."RO-1"."MODE BUFF", in2 := 1)
      { S7_Templates := "SrcType := Int" } EQ_Contact(in1 := "MODE SELECTION DB"."RO-1"."PROCESS BUFF", in2 := 2)
      { S7_Templates := "SrcType := Int" } EQ_Contact(in1 := "RO 1 LEVEL DB"."AGLV 302 BUFF", in2 := 1)
      Coil( "RO_1 DB".OUTPUT."AGLV-302" )
   END_RUNG
   // the same network as SCL:
   "RO_1 DB".OUTPUT."AGLV-302" := ("MODE SELECTION DB"."RO-1"."MODE BUFF" = 1) AND ("MODE SELECTION DB"."RO-1"."PROCESS BUFF" = 2) AND ("RO 1 LEVEL DB"."AGLV 302 BUFF" = 1);
END_REGION

REGION Network 13: LT 401 HIGH - RECIRCULATION LOGIC
   RUNG wire#powerrail
      Contact( "AlwaysTRUE" )
      { S7_Templates := "SrcType := Int" } EQ_Contact(in1 := "MODE SELECTION DB"."RO-1"."MODE BUFF", in2 := 1)
      { S7_Templates := "SrcType := Int" } EQ_Contact(in1 := "MODE SELECTION DB"."RO-1"."PROCESS BUFF", in2 := 2)
      { S7_Templates := "SrcType := Int" } EQ_Contact(in1 := "AI SCALING DB"."LT-401".HIGH_BUFF, in2 := 4)
      { S7_Templates := "SrcType := Int" } EQ_Contact(in1 := "RO 1 LEVEL DB"."LEVEL HI RECIRC BUFF", in2 := 0)
      { S7_Templates := "time_type := Time" } "IEC_Timer_0_DB_44".TON(pt := T#2S, et =>)
      Move(in := 1, out1 => "RO 1 LEVEL DB"."LEVEL HI RECIRC BUFF")
   END_RUNG
   // the same network as SCL:
   "IEC_Timer_0_DB_44".TON(IN := "AlwaysTRUE" AND ("MODE SELECTION DB"."RO-1"."MODE BUFF" = 1) AND ("MODE SELECTION DB"."RO-1"."PROCESS BUFF" = 2) AND ("AI SCALING DB"."LT-401".HIGH_BUFF = 4) AND ("RO 1 LEVEL DB"."LEVEL HI RECIRC BUFF" = 0),
                           PT := T#2S);
   IF "IEC_Timer_0_DB_44".Q THEN "RO 1 LEVEL DB"."LEVEL HI RECIRC BUFF" := 1; END_IF;
END_REGION

REGION Network 14: RO-1 OFFTIME START ONCE LEVEL IS HIGH
   RUNG wire#powerrail
      Contact( "AlwaysTRUE" )
      { S7_Templates := "SrcType := Int" } EQ_Contact(in1 := "MODE SELECTION DB"."RO-1"."MODE BUFF", in2 := 1)
      { S7_Templates := "SrcType := Int" } EQ_Contact(in1 := "MODE SELECTION DB"."RO-1"."PROCESS BUFF", in2 := 2)
      { S7_Templates := "SrcType := Int" } EQ_Contact(in1 := "AI SCALING DB"."LT-401".HIGH_BUFF, in2 := 4)
      { S7_Templates := "SrcType := Int" } EQ_Contact(in1 := "RO 1 LEVEL DB"."LEVEL HI RECIRC BUFF", in2 := 1)
      { S7_Templates := "time_type := Time" } "IEC_Timer_0_DB_48".TON(pt := T#2S, et =>)
      Move(in := 2, out1 => "RO 1 LEVEL DB"."LEVEL HI RECIRC BUFF")
   END_RUNG
   // the same network as SCL:
   "IEC_Timer_0_DB_48".TON(IN := "AlwaysTRUE" AND ("MODE SELECTION DB"."RO-1"."MODE BUFF" = 1) AND ("MODE SELECTION DB"."RO-1"."PROCESS BUFF" = 2) AND ("AI SCALING DB"."LT-401".HIGH_BUFF = 4) AND ("RO 1 LEVEL DB"."LEVEL HI RECIRC BUFF" = 1),
                           PT := T#2S);
   IF "IEC_Timer_0_DB_48".Q THEN "RO 1 LEVEL DB"."LEVEL HI RECIRC BUFF" := 2; END_IF;
END_REGION

REGION Network 15: RO 1 OFF TIME START
   RUNG wire#powerrail
      "TIMING_MIN_DB_7"(RESET := wire#w1, INPUT := wire#w2, "SET TIME" := "RO 1 LEVEL DB"."LEVEL HI RECIRC RO OFF TIME SV", "PRESENT VALUE OF TIME" => "RO 1 LEVEL DB"."LEVEL HI RECIRC RO OFF TIME PV", DONE =>)
   END_RUNG
   RUNG wire#powerrail
      { S7_Templates := "SrcType := Int" } NE_Contact(in1 := "MODE SELECTION DB"."RO-1"."MODE BUFF", in2 := 1)
   END_RUNG wire#w1
   RUNG wire#powerrail
      { S7_Templates := "SrcType := Int" } EQ_Contact(in1 := "MODE SELECTION DB"."RO-1"."MODE BUFF", in2 := 1)
      { S7_Templates := "SrcType := Int" } NE_Contact(in1 := "MODE SELECTION DB"."RO-1"."PROCESS BUFF", in2 := 2)
   END_RUNG wire#w1
   RUNG wire#powerrail
      { S7_Templates := "SrcType := Int" } NE_Contact(in1 := "RO 1 LEVEL DB"."LEVEL HI RECIRC BUFF", in2 := 2)
   END_RUNG wire#w1
   RUNG wire#powerrail
      Contact( "AlwaysTRUE" )
      { S7_Templates := "SrcType := Int" } EQ_Contact(in1 := "MODE SELECTION DB"."RO-1"."MODE BUFF", in2 := 1)
      { S7_Templates := "SrcType := Int" } EQ_Contact(in1 := "MODE SELECTION DB"."RO-1"."PROCESS BUFF", in2 := 2)
      { S7_Templates := "SrcType := Int" } EQ_Contact(in1 := "RO 1 LEVEL DB"."LEVEL HI RECIRC BUFF", in2 := 2)
   END_RUNG wire#w2
   // the same network as SCL:
   "TIMING_MIN_DB_7"("SET TIME" := "RO 1 LEVEL DB"."LEVEL HI RECIRC RO OFF TIME SV",   // "TIMING_MIN"
                     RESET := ("MODE SELECTION DB"."RO-1"."MODE BUFF" <> 1) OR (("MODE SELECTION DB"."RO-1"."MODE BUFF" = 1) AND ("MODE SELECTION DB"."RO-1"."PROCESS BUFF" <> 2)) OR ("RO 1 LEVEL DB"."LEVEL HI RECIRC BUFF" <> 2),
                     INPUT := "AlwaysTRUE" AND ("MODE SELECTION DB"."RO-1"."MODE BUFF" = 1) AND ("MODE SELECTION DB"."RO-1"."PROCESS BUFF" = 2) AND ("RO 1 LEVEL DB"."LEVEL HI RECIRC BUFF" = 2),
                     "PRESENT VALUE OF TIME" => "RO 1 LEVEL DB"."LEVEL HI RECIRC RO OFF TIME PV");
END_REGION

REGION Network 16: RO 1 RECIRCULATION START AFTER OFF TIME OVER
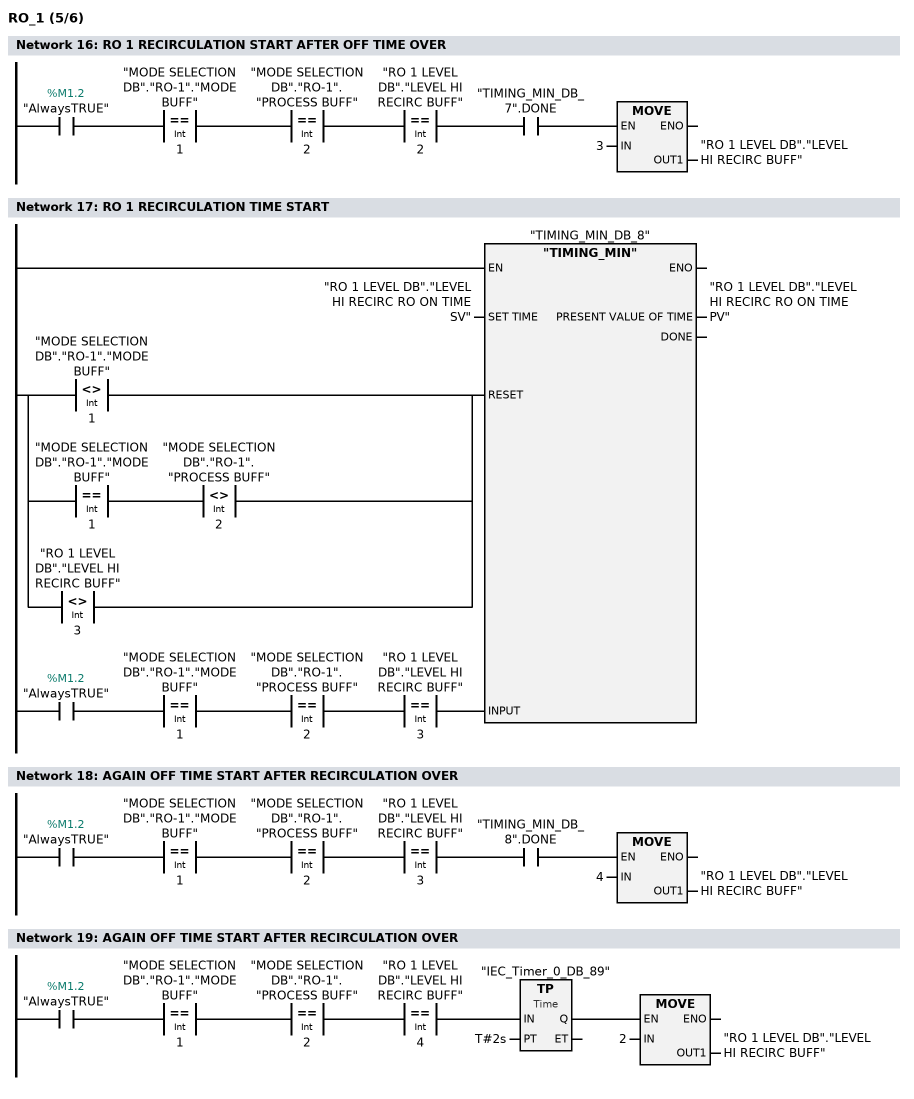
   RUNG wire#powerrail
      Contact( "AlwaysTRUE" )
      { S7_Templates := "SrcType := Int" } EQ_Contact(in1 := "MODE SELECTION DB"."RO-1"."MODE BUFF", in2 := 1)
      { S7_Templates := "SrcType := Int" } EQ_Contact(in1 := "MODE SELECTION DB"."RO-1"."PROCESS BUFF", in2 := 2)
      { S7_Templates := "SrcType := Int" } EQ_Contact(in1 := "RO 1 LEVEL DB"."LEVEL HI RECIRC BUFF", in2 := 2)
      Contact( "TIMING_MIN_DB_7".DONE )
      Move(in := 3, out1 => "RO 1 LEVEL DB"."LEVEL HI RECIRC BUFF")
   END_RUNG
   // the same network as SCL:
   IF "AlwaysTRUE" AND ("MODE SELECTION DB"."RO-1"."MODE BUFF" = 1) AND ("MODE SELECTION DB"."RO-1"."PROCESS BUFF" = 2) AND ("RO 1 LEVEL DB"."LEVEL HI RECIRC BUFF" = 2) AND "TIMING_MIN_DB_7".DONE THEN
       "RO 1 LEVEL DB"."LEVEL HI RECIRC BUFF" := 3;
   END_IF;
END_REGION

REGION Network 17: RO 1 RECIRCULATION TIME START
   RUNG wire#powerrail
      "TIMING_MIN_DB_8"(RESET := wire#w1, INPUT := wire#w2, "SET TIME" := "RO 1 LEVEL DB"."LEVEL HI RECIRC RO ON TIME SV", "PRESENT VALUE OF TIME" => "RO 1 LEVEL DB"."LEVEL HI RECIRC RO ON TIME PV", DONE =>)
   END_RUNG
   RUNG wire#powerrail
      { S7_Templates := "SrcType := Int" } NE_Contact(in1 := "MODE SELECTION DB"."RO-1"."MODE BUFF", in2 := 1)
   END_RUNG wire#w1
   RUNG wire#powerrail
      { S7_Templates := "SrcType := Int" } EQ_Contact(in1 := "MODE SELECTION DB"."RO-1"."MODE BUFF", in2 := 1)
      { S7_Templates := "SrcType := Int" } NE_Contact(in1 := "MODE SELECTION DB"."RO-1"."PROCESS BUFF", in2 := 2)
   END_RUNG wire#w1
   RUNG wire#powerrail
      { S7_Templates := "SrcType := Int" } NE_Contact(in1 := "RO 1 LEVEL DB"."LEVEL HI RECIRC BUFF", in2 := 3)
   END_RUNG wire#w1
   RUNG wire#powerrail
      Contact( "AlwaysTRUE" )
      { S7_Templates := "SrcType := Int" } EQ_Contact(in1 := "MODE SELECTION DB"."RO-1"."MODE BUFF", in2 := 1)
      { S7_Templates := "SrcType := Int" } EQ_Contact(in1 := "MODE SELECTION DB"."RO-1"."PROCESS BUFF", in2 := 2)
      { S7_Templates := "SrcType := Int" } EQ_Contact(in1 := "RO 1 LEVEL DB"."LEVEL HI RECIRC BUFF", in2 := 3)
   END_RUNG wire#w2
   // the same network as SCL:
   "TIMING_MIN_DB_8"("SET TIME" := "RO 1 LEVEL DB"."LEVEL HI RECIRC RO ON TIME SV",   // "TIMING_MIN"
                     RESET := ("MODE SELECTION DB"."RO-1"."MODE BUFF" <> 1) OR (("MODE SELECTION DB"."RO-1"."MODE BUFF" = 1) AND ("MODE SELECTION DB"."RO-1"."PROCESS BUFF" <> 2)) OR ("RO 1 LEVEL DB"."LEVEL HI RECIRC BUFF" <> 3),
                     INPUT := "AlwaysTRUE" AND ("MODE SELECTION DB"."RO-1"."MODE BUFF" = 1) AND ("MODE SELECTION DB"."RO-1"."PROCESS BUFF" = 2) AND ("RO 1 LEVEL DB"."LEVEL HI RECIRC BUFF" = 3),
                     "PRESENT VALUE OF TIME" => "RO 1 LEVEL DB"."LEVEL HI RECIRC RO ON TIME PV");
END_REGION

REGION Network 18: AGAIN OFF TIME START AFTER RECIRCULATION OVER
   RUNG wire#powerrail
      Contact( "AlwaysTRUE" )
      { S7_Templates := "SrcType := Int" } EQ_Contact(in1 := "MODE SELECTION DB"."RO-1"."MODE BUFF", in2 := 1)
      { S7_Templates := "SrcType := Int" } EQ_Contact(in1 := "MODE SELECTION DB"."RO-1"."PROCESS BUFF", in2 := 2)
      { S7_Templates := "SrcType := Int" } EQ_Contact(in1 := "RO 1 LEVEL DB"."LEVEL HI RECIRC BUFF", in2 := 3)
      Contact( "TIMING_MIN_DB_8".DONE )
      Move(in := 4, out1 => "RO 1 LEVEL DB"."LEVEL HI RECIRC BUFF")
   END_RUNG
   // the same network as SCL:
   IF "AlwaysTRUE" AND ("MODE SELECTION DB"."RO-1"."MODE BUFF" = 1) AND ("MODE SELECTION DB"."RO-1"."PROCESS BUFF" = 2) AND ("RO 1 LEVEL DB"."LEVEL HI RECIRC BUFF" = 3) AND "TIMING_MIN_DB_8".DONE THEN
       "RO 1 LEVEL DB"."LEVEL HI RECIRC BUFF" := 4;
   END_IF;
END_REGION

REGION Network 19: AGAIN OFF TIME START AFTER RECIRCULATION OVER
   RUNG wire#powerrail
      Contact( "AlwaysTRUE" )
      { S7_Templates := "SrcType := Int" } EQ_Contact(in1 := "MODE SELECTION DB"."RO-1"."MODE BUFF", in2 := 1)
      { S7_Templates := "SrcType := Int" } EQ_Contact(in1 := "MODE SELECTION DB"."RO-1"."PROCESS BUFF", in2 := 2)
      { S7_Templates := "SrcType := Int" } EQ_Contact(in1 := "RO 1 LEVEL DB"."LEVEL HI RECIRC BUFF", in2 := 4)
      { S7_Templates := "time_type := Time" } "IEC_Timer_0_DB_89".TP(pt := T#2s, et =>)
      Move(in := 2, out1 => "RO 1 LEVEL DB"."LEVEL HI RECIRC BUFF")
   END_RUNG
   // the same network as SCL:
   "IEC_Timer_0_DB_89".TP(IN := "AlwaysTRUE" AND ("MODE SELECTION DB"."RO-1"."MODE BUFF" = 1) AND ("MODE SELECTION DB"."RO-1"."PROCESS BUFF" = 2) AND ("RO 1 LEVEL DB"."LEVEL HI RECIRC BUFF" = 4),
                          PT := T#2s);
   IF "IEC_Timer_0_DB_89".Q THEN "RO 1 LEVEL DB"."LEVEL HI RECIRC BUFF" := 2; END_IF;
END_REGION

REGION Network 20: REcirculation stop when level is normal
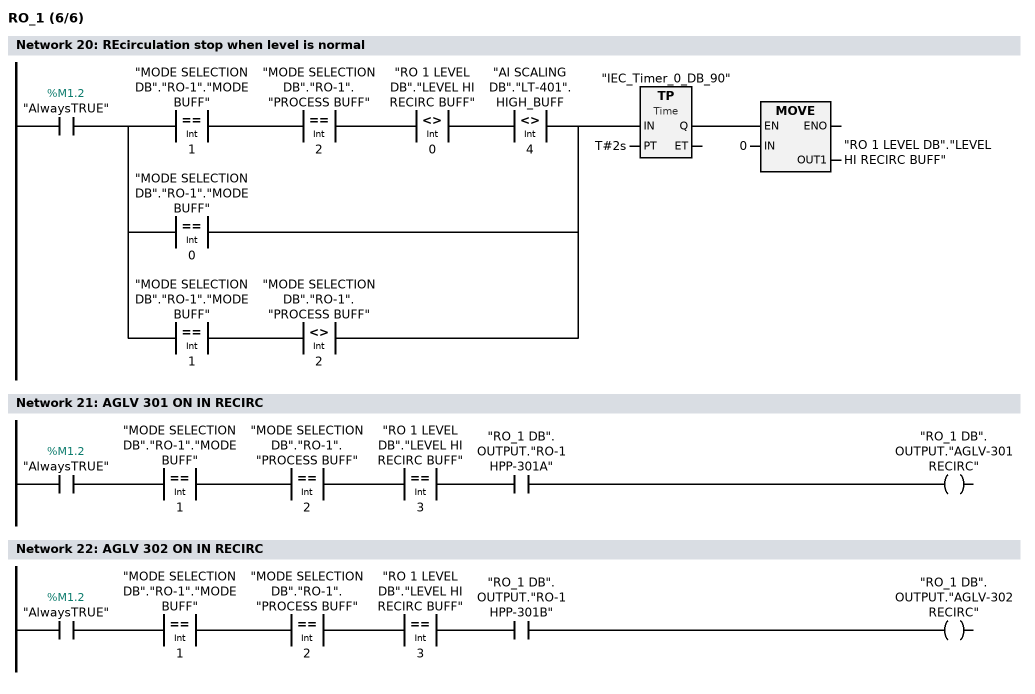
   RUNG wire#powerrail
      Contact( "AlwaysTRUE" )
      wire#w1
      { S7_Templates := "SrcType := Int" } EQ_Contact(in1 := "MODE SELECTION DB"."RO-1"."MODE BUFF", in2 := 1)
      { S7_Templates := "SrcType := Int" } EQ_Contact(in1 := "MODE SELECTION DB"."RO-1"."PROCESS BUFF", in2 := 2)
      { S7_Templates := "SrcType := Int" } NE_Contact(in1 := "RO 1 LEVEL DB"."LEVEL HI RECIRC BUFF", in2 := 0)
      { S7_Templates := "SrcType := Int" } NE_Contact(in1 := "AI SCALING DB"."LT-401".HIGH_BUFF, in2 := 4)
      wire#w2
      { S7_Templates := "time_type := Time" } "IEC_Timer_0_DB_90".TP(pt := T#2s, et =>)
      Move(in := 0, out1 => "RO 1 LEVEL DB"."LEVEL HI RECIRC BUFF")
   END_RUNG
   RUNG wire#w1
      { S7_Templates := "SrcType := Int" } EQ_Contact(in1 := "MODE SELECTION DB"."RO-1"."MODE BUFF", in2 := 0)
   END_RUNG wire#w2
   RUNG wire#w1
      { S7_Templates := "SrcType := Int" } EQ_Contact(in1 := "MODE SELECTION DB"."RO-1"."MODE BUFF", in2 := 1)
      { S7_Templates := "SrcType := Int" } NE_Contact(in1 := "MODE SELECTION DB"."RO-1"."PROCESS BUFF", in2 := 2)
   END_RUNG wire#w2
   // the same network as SCL:
   "IEC_Timer_0_DB_90".TP(IN := "AlwaysTRUE" AND ((("MODE SELECTION DB"."RO-1"."MODE BUFF" = 1) AND ("MODE SELECTION DB"."RO-1"."PROCESS BUFF" = 2) AND ("RO 1 LEVEL DB"."LEVEL HI RECIRC BUFF" <> 0) AND ("AI SCALING DB"."LT-401".HIGH_BUFF <> 4)) OR ("MODE SELECTION DB"."RO-1"."MODE BUFF" = 0) OR (("MODE SELECTION DB"."RO-1"."MODE BUFF" = 1) AND ("MODE SELECTION DB"."RO-1"."PROCESS BUFF" <> 2))),
                          PT := T#2s);
   IF "IEC_Timer_0_DB_90".Q THEN "RO 1 LEVEL DB"."LEVEL HI RECIRC BUFF" := 0; END_IF;
END_REGION

REGION Network 21: AGLV 301 ON IN RECIRC
   RUNG wire#powerrail
      Contact( "AlwaysTRUE" )
      { S7_Templates := "SrcType := Int" } EQ_Contact(in1 := "MODE SELECTION DB"."RO-1"."MODE BUFF", in2 := 1)
      { S7_Templates := "SrcType := Int" } EQ_Contact(in1 := "MODE SELECTION DB"."RO-1"."PROCESS BUFF", in2 := 2)
      { S7_Templates := "SrcType := Int" } EQ_Contact(in1 := "RO 1 LEVEL DB"."LEVEL HI RECIRC BUFF", in2 := 3)
      Contact( "RO_1 DB".OUTPUT."RO-1 HPP-301A" )
      Coil( "RO_1 DB".OUTPUT."AGLV-301 RECIRC" )
   END_RUNG
   // the same network as SCL:
   "RO_1 DB".OUTPUT."AGLV-301 RECIRC" := "AlwaysTRUE" AND ("MODE SELECTION DB"."RO-1"."MODE BUFF" = 1) AND ("MODE SELECTION DB"."RO-1"."PROCESS BUFF" = 2) AND ("RO 1 LEVEL DB"."LEVEL HI RECIRC BUFF" = 3) AND "RO_1 DB".OUTPUT."RO-1 HPP-301A";
END_REGION

REGION Network 22: AGLV 302 ON IN RECIRC
   RUNG wire#powerrail
      Contact( "AlwaysTRUE" )
      { S7_Templates := "SrcType := Int" } EQ_Contact(in1 := "MODE SELECTION DB"."RO-1"."MODE BUFF", in2 := 1)
      { S7_Templates := "SrcType := Int" } EQ_Contact(in1 := "MODE SELECTION DB"."RO-1"."PROCESS BUFF", in2 := 2)
      { S7_Templates := "SrcType := Int" } EQ_Contact(in1 := "RO 1 LEVEL DB"."LEVEL HI RECIRC BUFF", in2 := 3)
      Contact( "RO_1 DB".OUTPUT."RO-1 HPP-301B" )
      Coil( "RO_1 DB".OUTPUT."AGLV-302 RECIRC" )
   END_RUNG
   // the same network as SCL:
   "RO_1 DB".OUTPUT."AGLV-302 RECIRC" := "AlwaysTRUE" AND ("MODE SELECTION DB"."RO-1"."MODE BUFF" = 1) AND ("MODE SELECTION DB"."RO-1"."PROCESS BUFF" = 2) AND ("RO 1 LEVEL DB"."LEVEL HI RECIRC BUFF" = 3) AND "RO_1 DB".OUTPUT."RO-1 HPP-301B";
END_REGION
END_FUNCTION

FUNCTION "RO_2" : Void   // FC11, LAD
{ S7_Optimized_Access := 'TRUE' }
// stored: SetENOAutomatically false
   VAR_TEMP   // added for the SCL form of the ladder/FBD networks
      _w1 : Bool;
   END_VAR
BEGIN

REGION Network 1: FEED PUMP
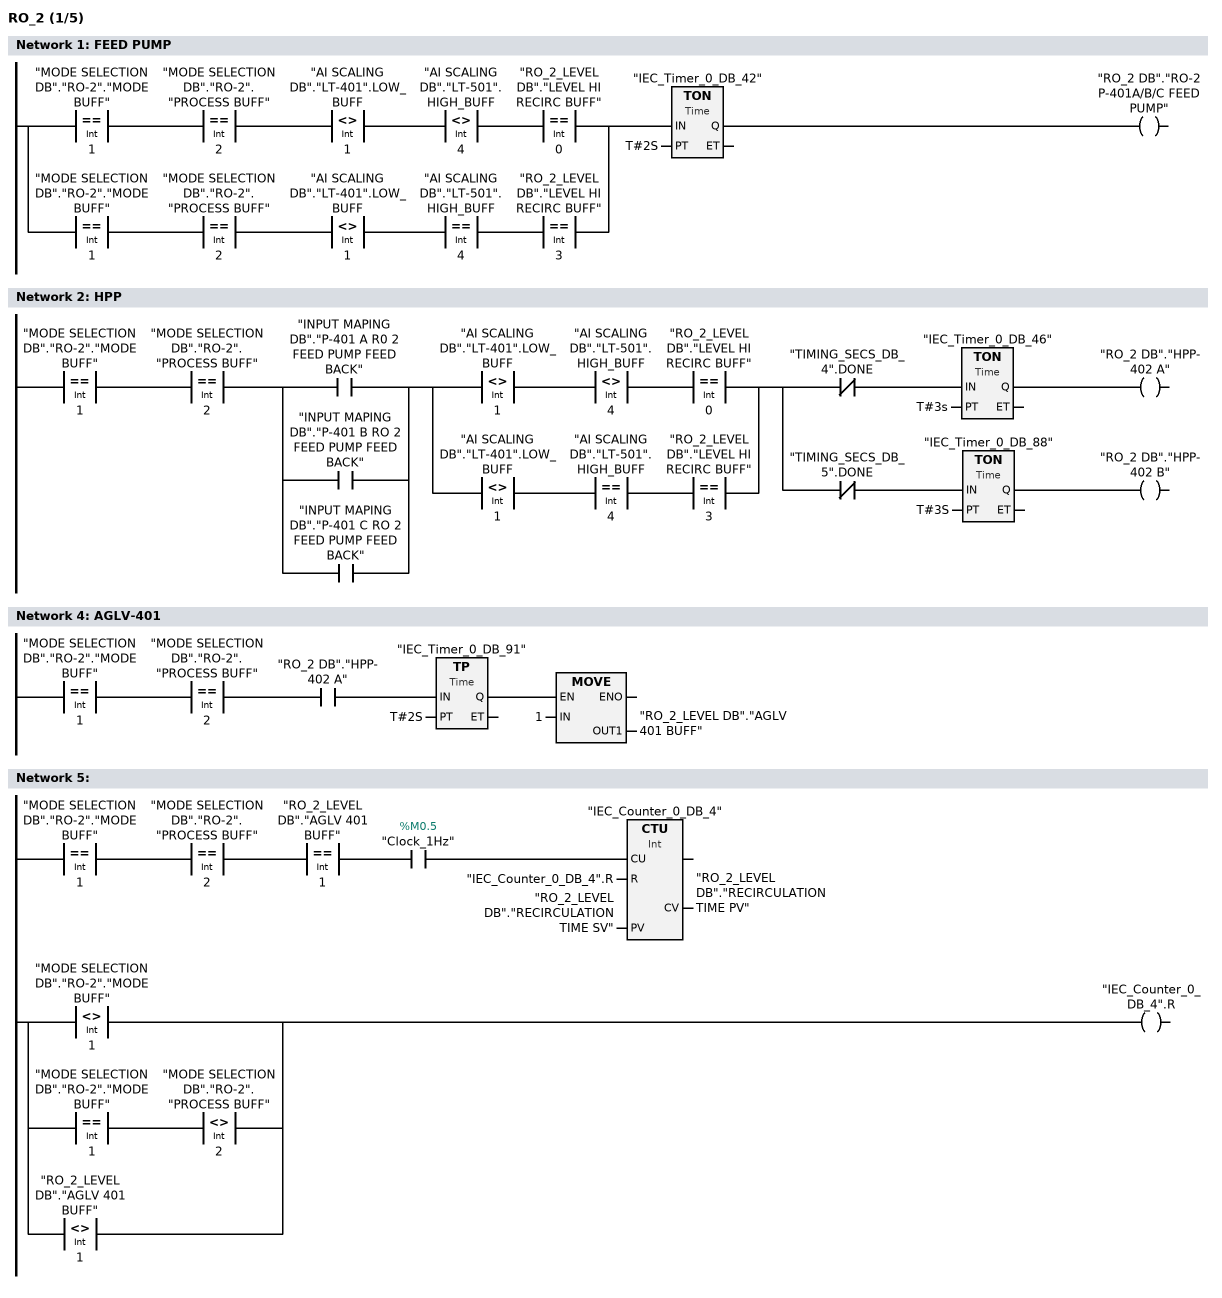
   RUNG wire#powerrail
      { S7_Templates := "SrcType := Int" } EQ_Contact(in1 := "MODE SELECTION DB"."RO-2"."MODE BUFF", in2 := 1)
      { S7_Templates := "SrcType := Int" } EQ_Contact(in1 := "MODE SELECTION DB"."RO-2"."PROCESS BUFF", in2 := 2)
      { S7_Templates := "SrcType := Int" } NE_Contact(in1 := "AI SCALING DB"."LT-401".LOW_BUFF, in2 := 1)
      { S7_Templates := "SrcType := Int" } NE_Contact(in1 := "AI SCALING DB"."LT-501".HIGH_BUFF, in2 := 4)
      { S7_Templates := "SrcType := Int" } EQ_Contact(in1 := "RO_2_LEVEL DB"."LEVEL HI RECIRC BUFF", in2 := 0)
      wire#w1
      { S7_Templates := "time_type := Time" } "IEC_Timer_0_DB_42".TON(pt := T#2S, et =>)
      Coil( "RO_2 DB"."RO-2 P-401A/B/C FEED PUMP" )
   END_RUNG
   RUNG wire#powerrail
      { S7_Templates := "SrcType := Int" } EQ_Contact(in1 := "MODE SELECTION DB"."RO-2"."MODE BUFF", in2 := 1)
      { S7_Templates := "SrcType := Int" } EQ_Contact(in1 := "MODE SELECTION DB"."RO-2"."PROCESS BUFF", in2 := 2)
      { S7_Templates := "SrcType := Int" } NE_Contact(in1 := "AI SCALING DB"."LT-401".LOW_BUFF, in2 := 1)
      { S7_Templates := "SrcType := Int" } EQ_Contact(in1 := "AI SCALING DB"."LT-501".HIGH_BUFF, in2 := 4)
      { S7_Templates := "SrcType := Int" } EQ_Contact(in1 := "RO_2_LEVEL DB"."LEVEL HI RECIRC BUFF", in2 := 3)
   END_RUNG wire#w1
   // the same network as SCL:
   "IEC_Timer_0_DB_42".TON(IN := (("MODE SELECTION DB"."RO-2"."MODE BUFF" = 1) AND ("MODE SELECTION DB"."RO-2"."PROCESS BUFF" = 2) AND ("AI SCALING DB"."LT-401".LOW_BUFF <> 1) AND ("AI SCALING DB"."LT-501".HIGH_BUFF <> 4) AND ("RO_2_LEVEL DB"."LEVEL HI RECIRC BUFF" = 0)) OR (("MODE SELECTION DB"."RO-2"."MODE BUFF" = 1) AND ("MODE SELECTION DB"."RO-2"."PROCESS BUFF" = 2) AND ("AI SCALING DB"."LT-401".LOW_BUFF <> 1) AND ("AI SCALING DB"."LT-501".HIGH_BUFF = 4) AND ("RO_2_LEVEL DB"."LEVEL HI RECIRC BUFF" = 3)),
                           PT := T#2S);
   "RO_2 DB"."RO-2 P-401A/B/C FEED PUMP" := "IEC_Timer_0_DB_42".Q;
END_REGION

REGION Network 2: HPP
   RUNG wire#powerrail
      { S7_Templates := "SrcType := Int" } EQ_Contact(in1 := "MODE SELECTION DB"."RO-2"."MODE BUFF", in2 := 1)
      { S7_Templates := "SrcType := Int" } EQ_Contact(in1 := "MODE SELECTION DB"."RO-2"."PROCESS BUFF", in2 := 2)
      wire#w1
      Contact( "INPUT MAPING DB"."P-401 A R0 2 FEED PUMP FEED BACK" )
      wire#w2
      { S7_Templates := "SrcType := Int" } NE_Contact(in1 := "AI SCALING DB"."LT-401".LOW_BUFF, in2 := 1)
      { S7_Templates := "SrcType := Int" } NE_Contact(in1 := "AI SCALING DB"."LT-501".HIGH_BUFF, in2 := 4)
      { S7_Templates := "SrcType := Int" } EQ_Contact(in1 := "RO_2_LEVEL DB"."LEVEL HI RECIRC BUFF", in2 := 0)
      wire#w3
      I_Contact( "TIMING_SECS_DB_4".DONE )
      { S7_Templates := "time_type := Time" } "IEC_Timer_0_DB_46".TON(pt := T#3s, et =>)
      Coil( "RO_2 DB"."HPP-402 A" )
   END_RUNG
   RUNG wire#w1
      Contact( "INPUT MAPING DB"."P-401 B RO 2 FEED PUMP FEED BACK" )
   END_RUNG wire#w2
   RUNG wire#w1
      Contact( "INPUT MAPING DB"."P-401 C RO 2 FEED PUMP FEED BACK" )
   END_RUNG wire#w2
   RUNG wire#w2
      { S7_Templates := "SrcType := Int" } NE_Contact(in1 := "AI SCALING DB"."LT-401".LOW_BUFF, in2 := 1)
      { S7_Templates := "SrcType := Int" } EQ_Contact(in1 := "AI SCALING DB"."LT-501".HIGH_BUFF, in2 := 4)
      { S7_Templates := "SrcType := Int" } EQ_Contact(in1 := "RO_2_LEVEL DB"."LEVEL HI RECIRC BUFF", in2 := 3)
   END_RUNG wire#w3
   RUNG wire#w3
      I_Contact( "TIMING_SECS_DB_5".DONE )
      { S7_Templates := "time_type := Time" } "IEC_Timer_0_DB_88".TON(pt := T#3S, et =>)
      Coil( "RO_2 DB"."HPP-402 B" )
   END_RUNG
   // the same network as SCL:
   #_w1 := ("MODE SELECTION DB"."RO-2"."MODE BUFF" = 1) AND ("MODE SELECTION DB"."RO-2"."PROCESS BUFF" = 2) AND ("INPUT MAPING DB"."P-401 A R0 2 FEED PUMP FEED BACK" OR "INPUT MAPING DB"."P-401 B RO 2 FEED PUMP FEED BACK" OR "INPUT MAPING DB"."P-401 C RO 2 FEED PUMP FEED BACK") AND ((("AI SCALING DB"."LT-401".LOW_BUFF <> 1) AND ("AI SCALING DB"."LT-501".HIGH_BUFF <> 4) AND ("RO_2_LEVEL DB"."LEVEL HI RECIRC BUFF" = 0)) OR (("AI SCALING DB"."LT-401".LOW_BUFF <> 1) AND ("AI SCALING DB"."LT-501".HIGH_BUFF = 4) AND ("RO_2_LEVEL DB"."LEVEL HI RECIRC BUFF" = 3)));
   "IEC_Timer_0_DB_46".TON(IN := #_w1 AND NOT "TIMING_SECS_DB_4".DONE, PT := T#3s);
   "RO_2 DB"."HPP-402 A" := "IEC_Timer_0_DB_46".Q;
   "IEC_Timer_0_DB_88".TON(IN := #_w1 AND NOT "TIMING_SECS_DB_5".DONE, PT := T#3S);
   "RO_2 DB"."HPP-402 B" := "IEC_Timer_0_DB_88".Q;
END_REGION

REGION Network 4: AGLV-401
   RUNG wire#powerrail
      { S7_Templates := "SrcType := Int" } EQ_Contact(in1 := "MODE SELECTION DB"."RO-2"."MODE BUFF", in2 := 1)
      { S7_Templates := "SrcType := Int" } EQ_Contact(in1 := "MODE SELECTION DB"."RO-2"."PROCESS BUFF", in2 := 2)
      Contact( "RO_2 DB"."HPP-402 A" )
      { S7_Templates := "time_type := Time" } "IEC_Timer_0_DB_91".TP(pt := T#2S, et =>)
      Move(in := 1, out1 => "RO_2_LEVEL DB"."AGLV 401 BUFF")
   END_RUNG
   // the same network as SCL:
   "IEC_Timer_0_DB_91".TP(IN := ("MODE SELECTION DB"."RO-2"."MODE BUFF" = 1) AND ("MODE SELECTION DB"."RO-2"."PROCESS BUFF" = 2) AND "RO_2 DB"."HPP-402 A",
                          PT := T#2S);
   IF "IEC_Timer_0_DB_91".Q THEN "RO_2_LEVEL DB"."AGLV 401 BUFF" := 1; END_IF;
END_REGION

REGION Network 5
   RUNG wire#powerrail
      { S7_Templates := "SrcType := Int" } EQ_Contact(in1 := "MODE SELECTION DB"."RO-2"."MODE BUFF", in2 := 1)
      { S7_Templates := "SrcType := Int" } EQ_Contact(in1 := "MODE SELECTION DB"."RO-2"."PROCESS BUFF", in2 := 2)
      { S7_Templates := "SrcType := Int" } EQ_Contact(in1 := "RO_2_LEVEL DB"."AGLV 401 BUFF", in2 := 1)
      Contact( "Clock_1Hz" )
      { S7_Templates := "value_type := Int" } "IEC_Counter_0_DB_4".CTU(r := "IEC_Counter_0_DB_4".R, pv := "RO_2_LEVEL DB"."RECIRCULATION TIME SV", cv => "RO_2_LEVEL DB"."RECIRCULATION TIME PV")
   END_RUNG
   RUNG wire#powerrail
      { S7_Templates := "SrcType := Int" } NE_Contact(in1 := "MODE SELECTION DB"."RO-2"."MODE BUFF", in2 := 1)
      wire#w1
      Coil( "IEC_Counter_0_DB_4".R )
   END_RUNG
   RUNG wire#powerrail
      { S7_Templates := "SrcType := Int" } EQ_Contact(in1 := "MODE SELECTION DB"."RO-2"."MODE BUFF", in2 := 1)
      { S7_Templates := "SrcType := Int" } NE_Contact(in1 := "MODE SELECTION DB"."RO-2"."PROCESS BUFF", in2 := 2)
   END_RUNG wire#w1
   RUNG wire#powerrail
      { S7_Templates := "SrcType := Int" } NE_Contact(in1 := "RO_2_LEVEL DB"."AGLV 401 BUFF", in2 := 1)
   END_RUNG wire#w1
   // the same network as SCL:
   "IEC_Counter_0_DB_4".CTU(CU := ("MODE SELECTION DB"."RO-2"."MODE BUFF" = 1) AND ("MODE SELECTION DB"."RO-2"."PROCESS BUFF" = 2) AND ("RO_2_LEVEL DB"."AGLV 401 BUFF" = 1) AND "Clock_1Hz",
                           R := "IEC_Counter_0_DB_4".R,
                           PV := "RO_2_LEVEL DB"."RECIRCULATION TIME SV",
                           CV => "RO_2_LEVEL DB"."RECIRCULATION TIME PV");
   "IEC_Counter_0_DB_4".R := ("MODE SELECTION DB"."RO-2"."MODE BUFF" <> 1) OR (("MODE SELECTION DB"."RO-2"."MODE BUFF" = 1) AND ("MODE SELECTION DB"."RO-2"."PROCESS BUFF" <> 2)) OR ("RO_2_LEVEL DB"."AGLV 401 BUFF" <> 1);
END_REGION

REGION Network 6
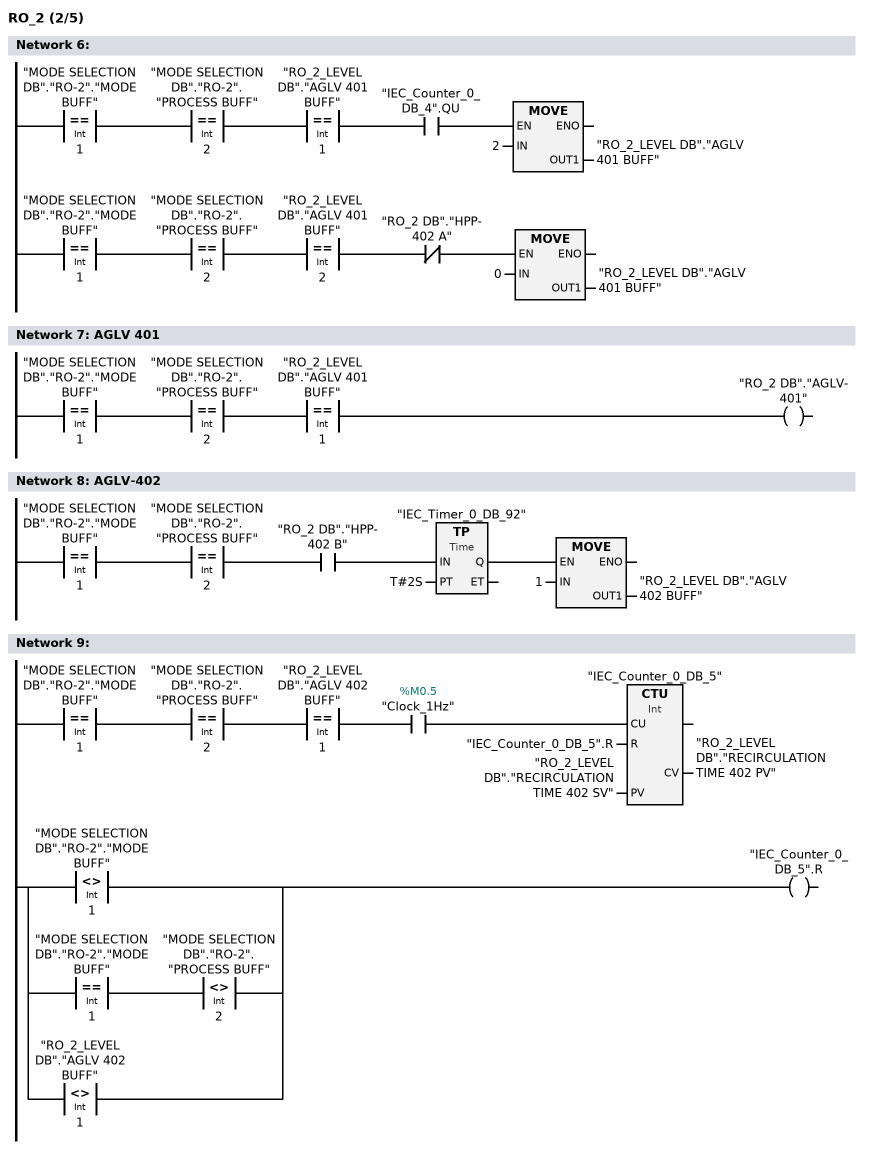
   RUNG wire#powerrail
      { S7_Templates := "SrcType := Int" } EQ_Contact(in1 := "MODE SELECTION DB"."RO-2"."MODE BUFF", in2 := 1)
      { S7_Templates := "SrcType := Int" } EQ_Contact(in1 := "MODE SELECTION DB"."RO-2"."PROCESS BUFF", in2 := 2)
      { S7_Templates := "SrcType := Int" } EQ_Contact(in1 := "RO_2_LEVEL DB"."AGLV 401 BUFF", in2 := 1)
      Contact( "IEC_Counter_0_DB_4".QU )
      Move(in := 2, out1 => "RO_2_LEVEL DB"."AGLV 401 BUFF")
   END_RUNG
   RUNG wire#powerrail
      { S7_Templates := "SrcType := Int" } EQ_Contact(in1 := "MODE SELECTION DB"."RO-2"."MODE BUFF", in2 := 1)
      { S7_Templates := "SrcType := Int" } EQ_Contact(in1 := "MODE SELECTION DB"."RO-2"."PROCESS BUFF", in2 := 2)
      { S7_Templates := "SrcType := Int" } EQ_Contact(in1 := "RO_2_LEVEL DB"."AGLV 401 BUFF", in2 := 2)
      I_Contact( "RO_2 DB"."HPP-402 A" )
      Move(in := 0, out1 => "RO_2_LEVEL DB"."AGLV 401 BUFF")
   END_RUNG
   // the same network as SCL:
   IF ("MODE SELECTION DB"."RO-2"."MODE BUFF" = 1) AND ("MODE SELECTION DB"."RO-2"."PROCESS BUFF" = 2) AND ("RO_2_LEVEL DB"."AGLV 401 BUFF" = 1) AND "IEC_Counter_0_DB_4".QU THEN
       "RO_2_LEVEL DB"."AGLV 401 BUFF" := 2;
   END_IF;
   IF ("MODE SELECTION DB"."RO-2"."MODE BUFF" = 1) AND ("MODE SELECTION DB"."RO-2"."PROCESS BUFF" = 2) AND ("RO_2_LEVEL DB"."AGLV 401 BUFF" = 2) AND NOT "RO_2 DB"."HPP-402 A" THEN
       "RO_2_LEVEL DB"."AGLV 401 BUFF" := 0;
   END_IF;
END_REGION

REGION Network 7: AGLV 401
   RUNG wire#powerrail
      { S7_Templates := "SrcType := Int" } EQ_Contact(in1 := "MODE SELECTION DB"."RO-2"."MODE BUFF", in2 := 1)
      { S7_Templates := "SrcType := Int" } EQ_Contact(in1 := "MODE SELECTION DB"."RO-2"."PROCESS BUFF", in2 := 2)
      { S7_Templates := "SrcType := Int" } EQ_Contact(in1 := "RO_2_LEVEL DB"."AGLV 401 BUFF", in2 := 1)
      Coil( "RO_2 DB"."AGLV-401" )
   END_RUNG
   // the same network as SCL:
   "RO_2 DB"."AGLV-401" := ("MODE SELECTION DB"."RO-2"."MODE BUFF" = 1) AND ("MODE SELECTION DB"."RO-2"."PROCESS BUFF" = 2) AND ("RO_2_LEVEL DB"."AGLV 401 BUFF" = 1);
END_REGION

REGION Network 8: AGLV-402
   RUNG wire#powerrail
      { S7_Templates := "SrcType := Int" } EQ_Contact(in1 := "MODE SELECTION DB"."RO-2"."MODE BUFF", in2 := 1)
      { S7_Templates := "SrcType := Int" } EQ_Contact(in1 := "MODE SELECTION DB"."RO-2"."PROCESS BUFF", in2 := 2)
      Contact( "RO_2 DB"."HPP-402 B" )
      { S7_Templates := "time_type := Time" } "IEC_Timer_0_DB_92".TP(pt := T#2S, et =>)
      Move(in := 1, out1 => "RO_2_LEVEL DB"."AGLV 402 BUFF")
   END_RUNG
   // the same network as SCL:
   "IEC_Timer_0_DB_92".TP(IN := ("MODE SELECTION DB"."RO-2"."MODE BUFF" = 1) AND ("MODE SELECTION DB"."RO-2"."PROCESS BUFF" = 2) AND "RO_2 DB"."HPP-402 B",
                          PT := T#2S);
   IF "IEC_Timer_0_DB_92".Q THEN "RO_2_LEVEL DB"."AGLV 402 BUFF" := 1; END_IF;
END_REGION

REGION Network 9
   RUNG wire#powerrail
      { S7_Templates := "SrcType := Int" } EQ_Contact(in1 := "MODE SELECTION DB"."RO-2"."MODE BUFF", in2 := 1)
      { S7_Templates := "SrcType := Int" } EQ_Contact(in1 := "MODE SELECTION DB"."RO-2"."PROCESS BUFF", in2 := 2)
      { S7_Templates := "SrcType := Int" } EQ_Contact(in1 := "RO_2_LEVEL DB"."AGLV 402 BUFF", in2 := 1)
      Contact( "Clock_1Hz" )
      { S7_Templates := "value_type := Int" } "IEC_Counter_0_DB_5".CTU(r := "IEC_Counter_0_DB_5".R, pv := "RO_2_LEVEL DB"."RECIRCULATION TIME 402 SV", cv => "RO_2_LEVEL DB"."RECIRCULATION TIME 402 PV")
   END_RUNG
   RUNG wire#powerrail
      { S7_Templates := "SrcType := Int" } NE_Contact(in1 := "MODE SELECTION DB"."RO-2"."MODE BUFF", in2 := 1)
      wire#w1
      Coil( "IEC_Counter_0_DB_5".R )
   END_RUNG
   RUNG wire#powerrail
      { S7_Templates := "SrcType := Int" } EQ_Contact(in1 := "MODE SELECTION DB"."RO-2"."MODE BUFF", in2 := 1)
      { S7_Templates := "SrcType := Int" } NE_Contact(in1 := "MODE SELECTION DB"."RO-2"."PROCESS BUFF", in2 := 2)
   END_RUNG wire#w1
   RUNG wire#powerrail
      { S7_Templates := "SrcType := Int" } NE_Contact(in1 := "RO_2_LEVEL DB"."AGLV 402 BUFF", in2 := 1)
   END_RUNG wire#w1
   // the same network as SCL:
   "IEC_Counter_0_DB_5".CTU(CU := ("MODE SELECTION DB"."RO-2"."MODE BUFF" = 1) AND ("MODE SELECTION DB"."RO-2"."PROCESS BUFF" = 2) AND ("RO_2_LEVEL DB"."AGLV 402 BUFF" = 1) AND "Clock_1Hz",
                           R := "IEC_Counter_0_DB_5".R,
                           PV := "RO_2_LEVEL DB"."RECIRCULATION TIME 402 SV",
                           CV => "RO_2_LEVEL DB"."RECIRCULATION TIME 402 PV");
   "IEC_Counter_0_DB_5".R := ("MODE SELECTION DB"."RO-2"."MODE BUFF" <> 1) OR (("MODE SELECTION DB"."RO-2"."MODE BUFF" = 1) AND ("MODE SELECTION DB"."RO-2"."PROCESS BUFF" <> 2)) OR ("RO_2_LEVEL DB"."AGLV 402 BUFF" <> 1);
END_REGION

REGION Network 10
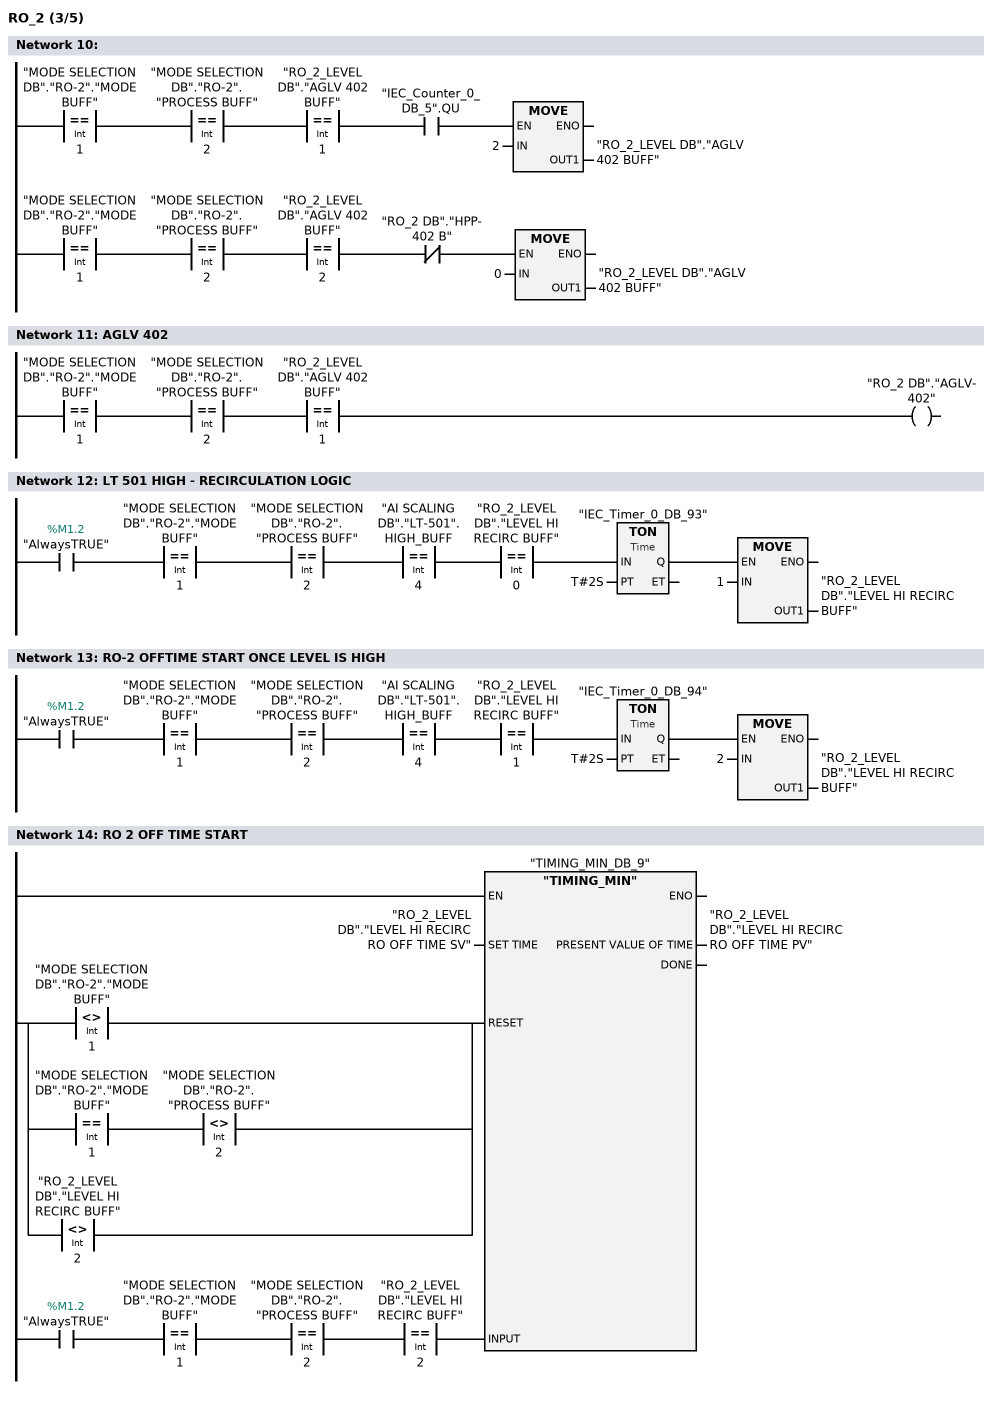
   RUNG wire#powerrail
      { S7_Templates := "SrcType := Int" } EQ_Contact(in1 := "MODE SELECTION DB"."RO-2"."MODE BUFF", in2 := 1)
      { S7_Templates := "SrcType := Int" } EQ_Contact(in1 := "MODE SELECTION DB"."RO-2"."PROCESS BUFF", in2 := 2)
      { S7_Templates := "SrcType := Int" } EQ_Contact(in1 := "RO_2_LEVEL DB"."AGLV 402 BUFF", in2 := 1)
      Contact( "IEC_Counter_0_DB_5".QU )
      Move(in := 2, out1 => "RO_2_LEVEL DB"."AGLV 402 BUFF")
   END_RUNG
   RUNG wire#powerrail
      { S7_Templates := "SrcType := Int" } EQ_Contact(in1 := "MODE SELECTION DB"."RO-2"."MODE BUFF", in2 := 1)
      { S7_Templates := "SrcType := Int" } EQ_Contact(in1 := "MODE SELECTION DB"."RO-2"."PROCESS BUFF", in2 := 2)
      { S7_Templates := "SrcType := Int" } EQ_Contact(in1 := "RO_2_LEVEL DB"."AGLV 402 BUFF", in2 := 2)
      I_Contact( "RO_2 DB"."HPP-402 B" )
      Move(in := 0, out1 => "RO_2_LEVEL DB"."AGLV 402 BUFF")
   END_RUNG
   // the same network as SCL:
   IF ("MODE SELECTION DB"."RO-2"."MODE BUFF" = 1) AND ("MODE SELECTION DB"."RO-2"."PROCESS BUFF" = 2) AND ("RO_2_LEVEL DB"."AGLV 402 BUFF" = 1) AND "IEC_Counter_0_DB_5".QU THEN
       "RO_2_LEVEL DB"."AGLV 402 BUFF" := 2;
   END_IF;
   IF ("MODE SELECTION DB"."RO-2"."MODE BUFF" = 1) AND ("MODE SELECTION DB"."RO-2"."PROCESS BUFF" = 2) AND ("RO_2_LEVEL DB"."AGLV 402 BUFF" = 2) AND NOT "RO_2 DB"."HPP-402 B" THEN
       "RO_2_LEVEL DB"."AGLV 402 BUFF" := 0;
   END_IF;
END_REGION

REGION Network 11: AGLV 402
   RUNG wire#powerrail
      { S7_Templates := "SrcType := Int" } EQ_Contact(in1 := "MODE SELECTION DB"."RO-2"."MODE BUFF", in2 := 1)
      { S7_Templates := "SrcType := Int" } EQ_Contact(in1 := "MODE SELECTION DB"."RO-2"."PROCESS BUFF", in2 := 2)
      { S7_Templates := "SrcType := Int" } EQ_Contact(in1 := "RO_2_LEVEL DB"."AGLV 402 BUFF", in2 := 1)
      Coil( "RO_2 DB"."AGLV-402" )
   END_RUNG
   // the same network as SCL:
   "RO_2 DB"."AGLV-402" := ("MODE SELECTION DB"."RO-2"."MODE BUFF" = 1) AND ("MODE SELECTION DB"."RO-2"."PROCESS BUFF" = 2) AND ("RO_2_LEVEL DB"."AGLV 402 BUFF" = 1);
END_REGION

REGION Network 12: LT 501 HIGH - RECIRCULATION LOGIC
   RUNG wire#powerrail
      Contact( "AlwaysTRUE" )
      { S7_Templates := "SrcType := Int" } EQ_Contact(in1 := "MODE SELECTION DB"."RO-2"."MODE BUFF", in2 := 1)
      { S7_Templates := "SrcType := Int" } EQ_Contact(in1 := "MODE SELECTION DB"."RO-2"."PROCESS BUFF", in2 := 2)
      { S7_Templates := "SrcType := Int" } EQ_Contact(in1 := "AI SCALING DB"."LT-501".HIGH_BUFF, in2 := 4)
      { S7_Templates := "SrcType := Int" } EQ_Contact(in1 := "RO_2_LEVEL DB"."LEVEL HI RECIRC BUFF", in2 := 0)
      { S7_Templates := "time_type := Time" } "IEC_Timer_0_DB_93".TON(pt := T#2S, et =>)
      Move(in := 1, out1 => "RO_2_LEVEL DB"."LEVEL HI RECIRC BUFF")
   END_RUNG
   // the same network as SCL:
   "IEC_Timer_0_DB_93".TON(IN := "AlwaysTRUE" AND ("MODE SELECTION DB"."RO-2"."MODE BUFF" = 1) AND ("MODE SELECTION DB"."RO-2"."PROCESS BUFF" = 2) AND ("AI SCALING DB"."LT-501".HIGH_BUFF = 4) AND ("RO_2_LEVEL DB"."LEVEL HI RECIRC BUFF" = 0),
                           PT := T#2S);
   IF "IEC_Timer_0_DB_93".Q THEN "RO_2_LEVEL DB"."LEVEL HI RECIRC BUFF" := 1; END_IF;
END_REGION

REGION Network 13: RO-2 OFFTIME START ONCE LEVEL IS HIGH
   RUNG wire#powerrail
      Contact( "AlwaysTRUE" )
      { S7_Templates := "SrcType := Int" } EQ_Contact(in1 := "MODE SELECTION DB"."RO-2"."MODE BUFF", in2 := 1)
      { S7_Templates := "SrcType := Int" } EQ_Contact(in1 := "MODE SELECTION DB"."RO-2"."PROCESS BUFF", in2 := 2)
      { S7_Templates := "SrcType := Int" } EQ_Contact(in1 := "AI SCALING DB"."LT-501".HIGH_BUFF, in2 := 4)
      { S7_Templates := "SrcType := Int" } EQ_Contact(in1 := "RO_2_LEVEL DB"."LEVEL HI RECIRC BUFF", in2 := 1)
      { S7_Templates := "time_type := Time" } "IEC_Timer_0_DB_94".TON(pt := T#2S, et =>)
      Move(in := 2, out1 => "RO_2_LEVEL DB"."LEVEL HI RECIRC BUFF")
   END_RUNG
   // the same network as SCL:
   "IEC_Timer_0_DB_94".TON(IN := "AlwaysTRUE" AND ("MODE SELECTION DB"."RO-2"."MODE BUFF" = 1) AND ("MODE SELECTION DB"."RO-2"."PROCESS BUFF" = 2) AND ("AI SCALING DB"."LT-501".HIGH_BUFF = 4) AND ("RO_2_LEVEL DB"."LEVEL HI RECIRC BUFF" = 1),
                           PT := T#2S);
   IF "IEC_Timer_0_DB_94".Q THEN "RO_2_LEVEL DB"."LEVEL HI RECIRC BUFF" := 2; END_IF;
END_REGION

REGION Network 14: RO 2 OFF TIME START
   RUNG wire#powerrail
      "TIMING_MIN_DB_9"(RESET := wire#w1, INPUT := wire#w2, "SET TIME" := "RO_2_LEVEL DB"."LEVEL HI RECIRC RO OFF TIME SV", "PRESENT VALUE OF TIME" => "RO_2_LEVEL DB"."LEVEL HI RECIRC RO OFF TIME PV", DONE =>)
   END_RUNG
   RUNG wire#powerrail
      { S7_Templates := "SrcType := Int" } NE_Contact(in1 := "MODE SELECTION DB"."RO-2"."MODE BUFF", in2 := 1)
   END_RUNG wire#w1
   RUNG wire#powerrail
      { S7_Templates := "SrcType := Int" } EQ_Contact(in1 := "MODE SELECTION DB"."RO-2"."MODE BUFF", in2 := 1)
      { S7_Templates := "SrcType := Int" } NE_Contact(in1 := "MODE SELECTION DB"."RO-2"."PROCESS BUFF", in2 := 2)
   END_RUNG wire#w1
   RUNG wire#powerrail
      { S7_Templates := "SrcType := Int" } NE_Contact(in1 := "RO_2_LEVEL DB"."LEVEL HI RECIRC BUFF", in2 := 2)
   END_RUNG wire#w1
   RUNG wire#powerrail
      Contact( "AlwaysTRUE" )
      { S7_Templates := "SrcType := Int" } EQ_Contact(in1 := "MODE SELECTION DB"."RO-2"."MODE BUFF", in2 := 1)
      { S7_Templates := "SrcType := Int" } EQ_Contact(in1 := "MODE SELECTION DB"."RO-2"."PROCESS BUFF", in2 := 2)
      { S7_Templates := "SrcType := Int" } EQ_Contact(in1 := "RO_2_LEVEL DB"."LEVEL HI RECIRC BUFF", in2 := 2)
   END_RUNG wire#w2
   // the same network as SCL:
   "TIMING_MIN_DB_9"("SET TIME" := "RO_2_LEVEL DB"."LEVEL HI RECIRC RO OFF TIME SV",   // "TIMING_MIN"
                     RESET := ("MODE SELECTION DB"."RO-2"."MODE BUFF" <> 1) OR (("MODE SELECTION DB"."RO-2"."MODE BUFF" = 1) AND ("MODE SELECTION DB"."RO-2"."PROCESS BUFF" <> 2)) OR ("RO_2_LEVEL DB"."LEVEL HI RECIRC BUFF" <> 2),
                     INPUT := "AlwaysTRUE" AND ("MODE SELECTION DB"."RO-2"."MODE BUFF" = 1) AND ("MODE SELECTION DB"."RO-2"."PROCESS BUFF" = 2) AND ("RO_2_LEVEL DB"."LEVEL HI RECIRC BUFF" = 2),
                     "PRESENT VALUE OF TIME" => "RO_2_LEVEL DB"."LEVEL HI RECIRC RO OFF TIME PV");
END_REGION

REGION Network 15: RO 2 RECIRCULATION START AFTER OFF TIME OVER
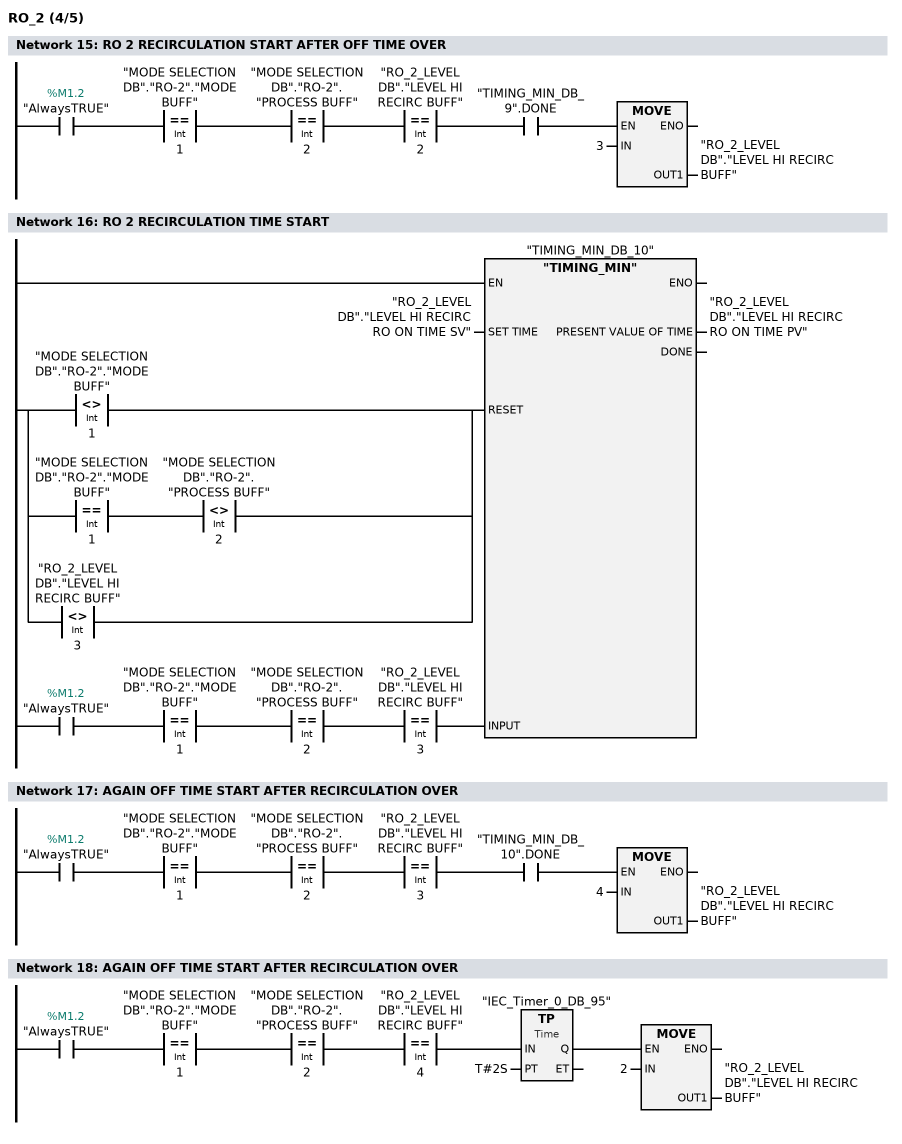
   RUNG wire#powerrail
      Contact( "AlwaysTRUE" )
      { S7_Templates := "SrcType := Int" } EQ_Contact(in1 := "MODE SELECTION DB"."RO-2"."MODE BUFF", in2 := 1)
      { S7_Templates := "SrcType := Int" } EQ_Contact(in1 := "MODE SELECTION DB"."RO-2"."PROCESS BUFF", in2 := 2)
      { S7_Templates := "SrcType := Int" } EQ_Contact(in1 := "RO_2_LEVEL DB"."LEVEL HI RECIRC BUFF", in2 := 2)
      Contact( "TIMING_MIN_DB_9".DONE )
      Move(in := 3, out1 => "RO_2_LEVEL DB"."LEVEL HI RECIRC BUFF")
   END_RUNG
   // the same network as SCL:
   IF "AlwaysTRUE" AND ("MODE SELECTION DB"."RO-2"."MODE BUFF" = 1) AND ("MODE SELECTION DB"."RO-2"."PROCESS BUFF" = 2) AND ("RO_2_LEVEL DB"."LEVEL HI RECIRC BUFF" = 2) AND "TIMING_MIN_DB_9".DONE THEN
       "RO_2_LEVEL DB"."LEVEL HI RECIRC BUFF" := 3;
   END_IF;
END_REGION

REGION Network 16: RO 2 RECIRCULATION TIME START
   RUNG wire#powerrail
      "TIMING_MIN_DB_10"(RESET := wire#w1, INPUT := wire#w2, "SET TIME" := "RO_2_LEVEL DB"."LEVEL HI RECIRC RO ON TIME SV", "PRESENT VALUE OF TIME" => "RO_2_LEVEL DB"."LEVEL HI RECIRC RO ON TIME PV", DONE =>)
   END_RUNG
   RUNG wire#powerrail
      { S7_Templates := "SrcType := Int" } NE_Contact(in1 := "MODE SELECTION DB"."RO-2"."MODE BUFF", in2 := 1)
   END_RUNG wire#w1
   RUNG wire#powerrail
      { S7_Templates := "SrcType := Int" } EQ_Contact(in1 := "MODE SELECTION DB"."RO-2"."MODE BUFF", in2 := 1)
      { S7_Templates := "SrcType := Int" } NE_Contact(in1 := "MODE SELECTION DB"."RO-2"."PROCESS BUFF", in2 := 2)
   END_RUNG wire#w1
   RUNG wire#powerrail
      { S7_Templates := "SrcType := Int" } NE_Contact(in1 := "RO_2_LEVEL DB"."LEVEL HI RECIRC BUFF", in2 := 3)
   END_RUNG wire#w1
   RUNG wire#powerrail
      Contact( "AlwaysTRUE" )
      { S7_Templates := "SrcType := Int" } EQ_Contact(in1 := "MODE SELECTION DB"."RO-2"."MODE BUFF", in2 := 1)
      { S7_Templates := "SrcType := Int" } EQ_Contact(in1 := "MODE SELECTION DB"."RO-2"."PROCESS BUFF", in2 := 2)
      { S7_Templates := "SrcType := Int" } EQ_Contact(in1 := "RO_2_LEVEL DB"."LEVEL HI RECIRC BUFF", in2 := 3)
   END_RUNG wire#w2
   // the same network as SCL:
   "TIMING_MIN_DB_10"("SET TIME" := "RO_2_LEVEL DB"."LEVEL HI RECIRC RO ON TIME SV",   // "TIMING_MIN"
                      RESET := ("MODE SELECTION DB"."RO-2"."MODE BUFF" <> 1) OR (("MODE SELECTION DB"."RO-2"."MODE BUFF" = 1) AND ("MODE SELECTION DB"."RO-2"."PROCESS BUFF" <> 2)) OR ("RO_2_LEVEL DB"."LEVEL HI RECIRC BUFF" <> 3),
                      INPUT := "AlwaysTRUE" AND ("MODE SELECTION DB"."RO-2"."MODE BUFF" = 1) AND ("MODE SELECTION DB"."RO-2"."PROCESS BUFF" = 2) AND ("RO_2_LEVEL DB"."LEVEL HI RECIRC BUFF" = 3),
                      "PRESENT VALUE OF TIME" => "RO_2_LEVEL DB"."LEVEL HI RECIRC RO ON TIME PV");
END_REGION

